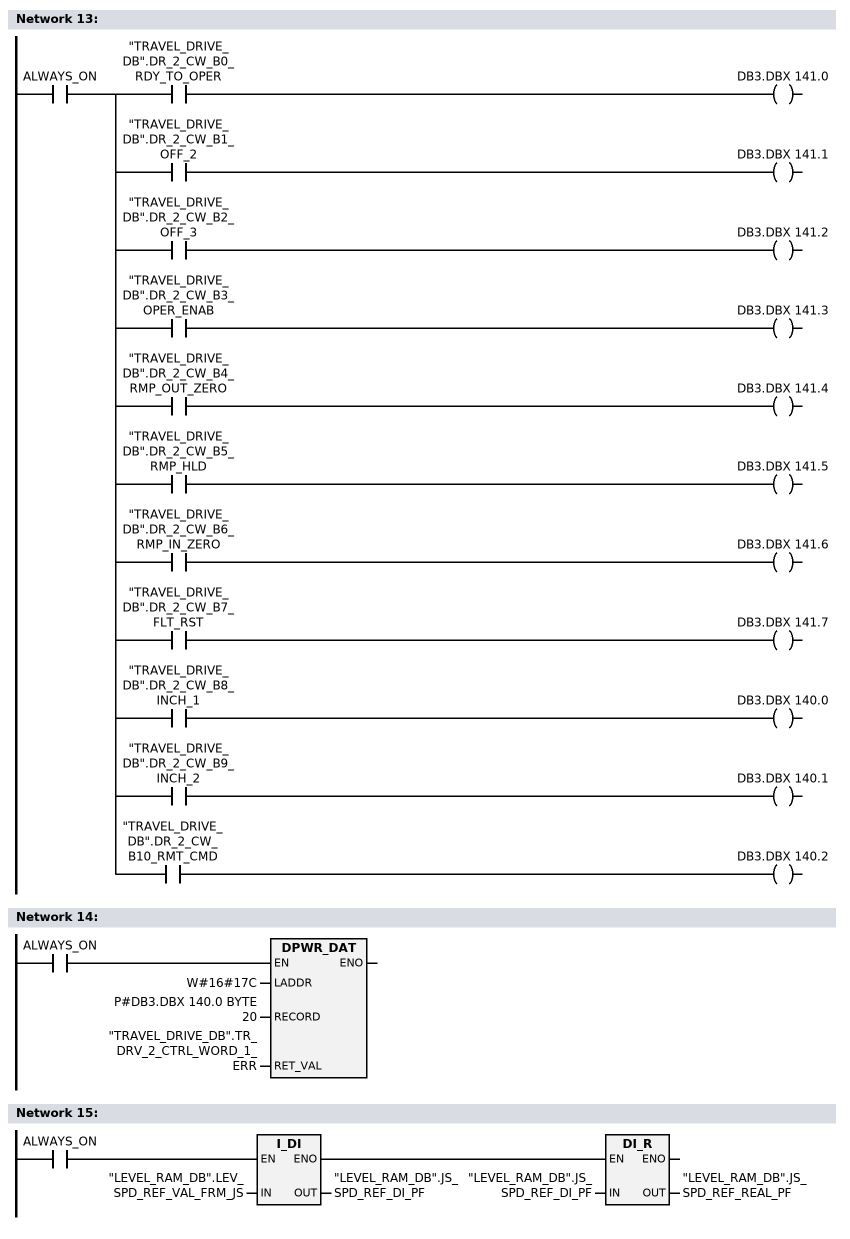
[picture p240: PROFIBUS_COMMUNICATION networks 13-15]
NETWORK
TITLE =
      A     "ALWAYS_ON";
      =     L 0.0;
      A     L 0.0;
      A     "TRAVEL_DRIVE_DB".DR_2_CW_B0_RDY_TO_OPER;
      =     DB3.DBX 141.0;
      A     L 0.0;
      A     "TRAVEL_DRIVE_DB".DR_2_CW_B1_OFF_2;
      =     DB3.DBX 141.1;
      A     L 0.0;
      A     "TRAVEL_DRIVE_DB".DR_2_CW_B2_OFF_3;
      =     DB3.DBX 141.2;
      A     L 0.0;
      A     "TRAVEL_DRIVE_DB".DR_2_CW_B3_OPER_ENAB;
      =     DB3.DBX 141.3;
      A     L 0.0;
      A     "TRAVEL_DRIVE_DB".DR_2_CW_B4_RMP_OUT_ZERO;
      =     DB3.DBX 141.4;
      A     L 0.0;
      A     "TRAVEL_DRIVE_DB".DR_2_CW_B5_RMP_HLD;
      =     DB3.DBX 141.5;
      A     L 0.0;
      A     "TRAVEL_DRIVE_DB".DR_2_CW_B6_RMP_IN_ZERO;
      =     DB3.DBX 141.6;
      A     L 0.0;
      A     "TRAVEL_DRIVE_DB".DR_2_CW_B7_FLT_RST;
      =     DB3.DBX 141.7;
      A     L 0.0;
      A     "TRAVEL_DRIVE_DB".DR_2_CW_B8_INCH_1;
      =     DB3.DBX 140.0;
      A     L 0.0;
      A     "TRAVEL_DRIVE_DB".DR_2_CW_B9_INCH_2;
      =     DB3.DBX 140.1;
      A     L 0.0;
      A     "TRAVEL_DRIVE_DB".DR_2_CW_B10_RMT_CMD;
      =     DB3.DBX 140.2;
NETWORK
TITLE =
      A     "ALWAYS_ON";
      JNB   M011;
      CALL  "DPWR_DAT" (
           LADDR                    := W#16#17C,
           RECORD                   := P#DB3.DBX 140.0 BYTE 20,
           RET_VAL                  := "TRAVEL_DRIVE_DB".TR_DRV_2_CTRL_WORD_1_ERR);
M011: NOP   0;
NETWORK
TITLE =
      A(;
      A     "ALWAYS_ON";
      JNB   M012;
      L     "LEVEL_RAM_DB".LEV_SPD_REF_VAL_FRM_JS;
      ITD;
      T     "LEVEL_RAM_DB".JS_SPD_REF_DI_PF;
      SET;
      SAVE;
      CLR;
M012: A     BR;
      );
      JNB   M013;
      L     "LEVEL_RAM_DB".JS_SPD_REF_DI_PF;
      DTR;
      T     "LEVEL_RAM_DB".JS_SPD_REF_REAL_PF;
M013: NOP   0;
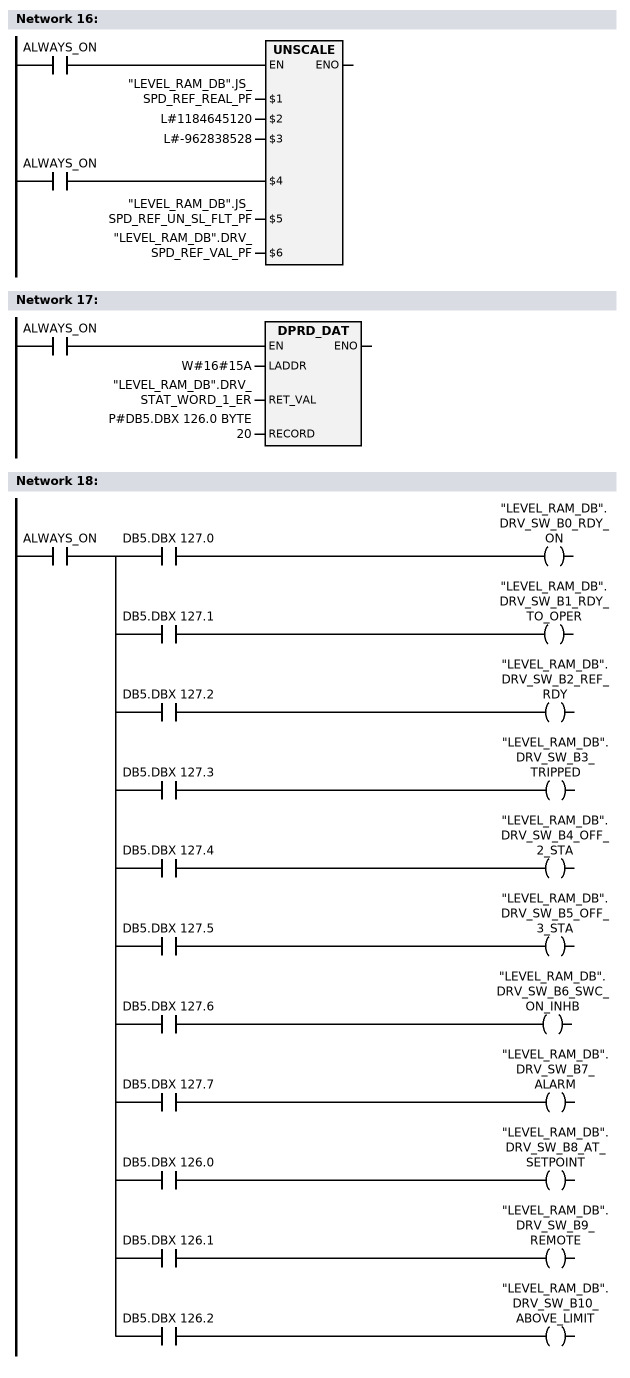
NETWORK
TITLE =
      A     "ALWAYS_ON";
      =     L 0.0;
      BLD   103;
      A     "ALWAYS_ON";
      JNB   M014;
      CALL  "UNSCALE" (
           $1                       := "LEVEL_RAM_DB".JS_SPD_REF_REAL_PF,
           $2                       := L#1184645120,
           $3                       := L#-962838528,
           $4                       := L 0.0,
           $5                       := "LEVEL_RAM_DB".JS_SPD_REF_UN_SL_FLT_PF,
           $6                       := "LEVEL_RAM_DB".DRV_SPD_REF_VAL_PF);
M014: NOP   0;
NETWORK
TITLE =
      A     "ALWAYS_ON";
      JNB   M015;
      CALL  "DPRD_DAT" (
           LADDR                    := W#16#15A,
           RET_VAL                  := "LEVEL_RAM_DB".DRV_STAT_WORD_1_ER,
           RECORD                   := P#DB5.DBX 126.0 BYTE 20);
M015: NOP   0;
NETWORK
TITLE =
      A     "ALWAYS_ON";
      =     L 0.0;
      A     L 0.0;
      A     DB5.DBX 127.0;
      =     "LEVEL_RAM_DB".DRV_SW_B0_RDY_ON;
      A     L 0.0;
      A     DB5.DBX 127.1;
      =     "LEVEL_RAM_DB".DRV_SW_B1_RDY_TO_OPER;
      A     L 0.0;
      A     DB5.DBX 127.2;
      =     "LEVEL_RAM_DB".DRV_SW_B2_REF_RDY;
      A     L 0.0;
      A     DB5.DBX 127.3;
      =     "LEVEL_RAM_DB".DRV_SW_B3_TRIPPED;
      A     L 0.0;
      A     DB5.DBX 127.4;
      =     "LEVEL_RAM_DB".DRV_SW_B4_OFF_2_STA;
      A     L 0.0;
      A     DB5.DBX 127.5;
      =     "LEVEL_RAM_DB".DRV_SW_B5_OFF_3_STA;
      A     L 0.0;
      A     DB5.DBX 127.6;
      =     "LEVEL_RAM_DB".DRV_SW_B6_SWC_ON_INHB;
      A     L 0.0;
      A     DB5.DBX 127.7;
      =     "LEVEL_RAM_DB".DRV_SW_B7_ALARM;
      A     L 0.0;
      A     DB5.DBX 126.0;
      =     "LEVEL_RAM_DB".DRV_SW_B8_AT_SETPOINT;
      A     L 0.0;
      A     DB5.DBX 126.1;
      =     "LEVEL_RAM_DB".DRV_SW_B9_REMOTE;
      A     L 0.0;
      A     DB5.DBX 126.2;
      =     "LEVEL_RAM_DB".DRV_SW_B10_ABOVE_LIMIT;
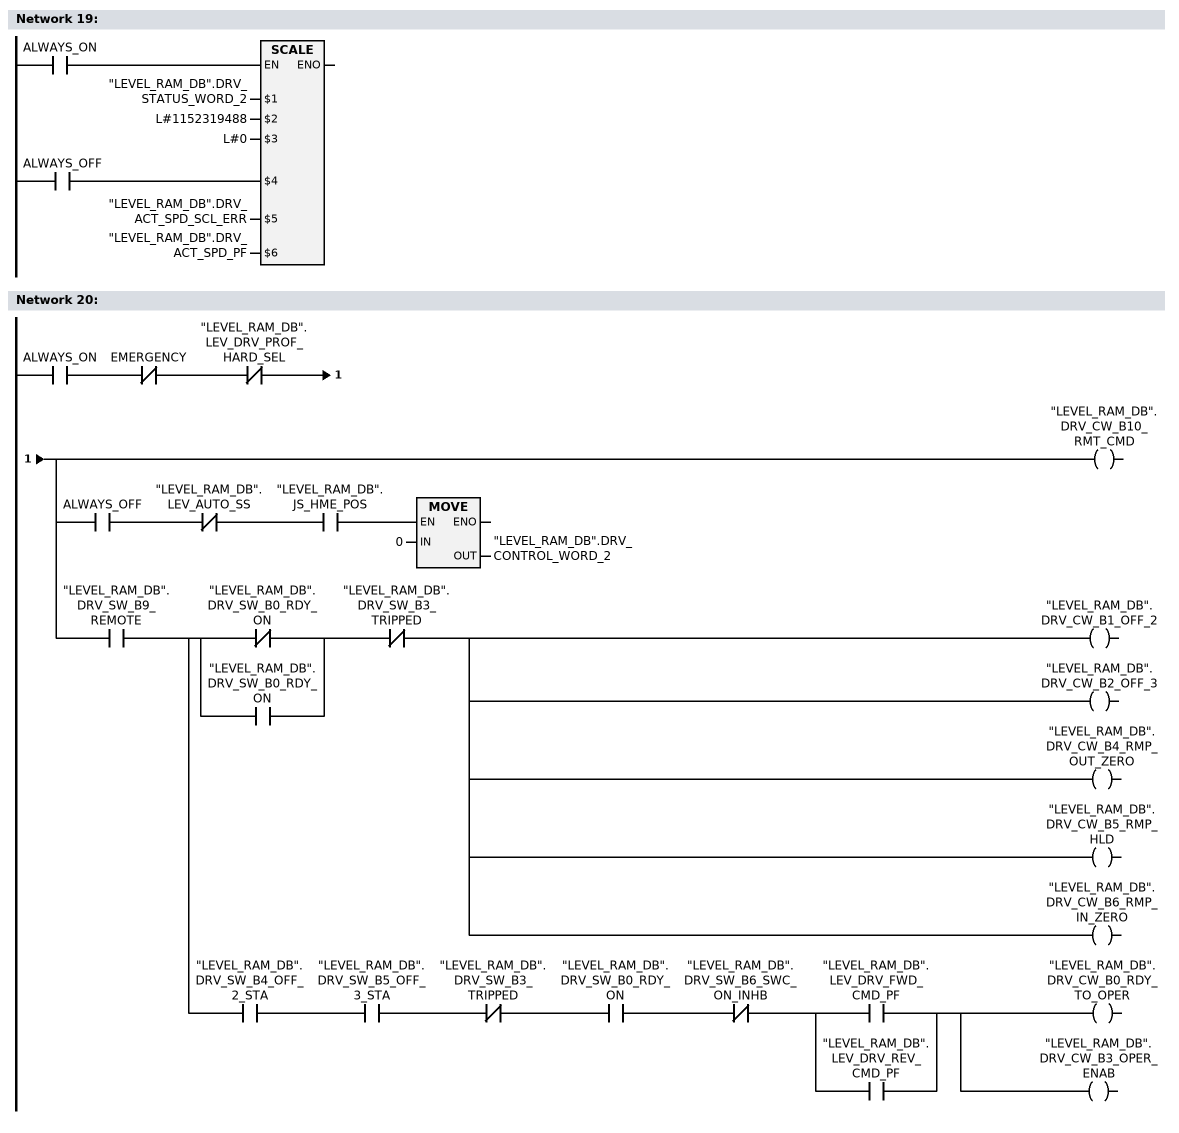
NETWORK
TITLE =
      A     "ALWAYS_OFF";
      =     L 0.0;
      BLD   103;
      A     "ALWAYS_ON";
      JNB   M016;
      CALL  "SCALE" (
           $1                       := "LEVEL_RAM_DB".DRV_STATUS_WORD_2,
           $2                       := L#1152319488,
           $3                       := L#0,
           $4                       := L 0.0,
           $5                       := "LEVEL_RAM_DB".DRV_ACT_SPD_SCL_ERR,
           $6                       := "LEVEL_RAM_DB".DRV_ACT_SPD_PF);
M016: NOP   0;
NETWORK
TITLE =
      A     "ALWAYS_ON";
      AN    "EMERGENCY";
      AN    "LEVEL_RAM_DB".LEV_DRV_PROF_HARD_SEL;
      =     L 0.0;
      A     L 0.0;
      BLD   102;
      =     "LEVEL_RAM_DB".DRV_CW_B10_RMT_CMD;
      A     L 0.0;
      A     "ALWAYS_OFF";
      AN    "LEVEL_RAM_DB".LEV_AUTO_SS;
      A     "LEVEL_RAM_DB".JS_HME_POS;
      JNB   M017;
      L     0;
      T     "LEVEL_RAM_DB".DRV_CONTROL_WORD_2;
M017: NOP   0;
      A     L 0.0;
      A     "LEVEL_RAM_DB".DRV_SW_B9_REMOTE;
      =     L 0.1;
      A     L 0.1;
      A(;
      ON    "LEVEL_RAM_DB".DRV_SW_B0_RDY_ON;
      O     "LEVEL_RAM_DB".DRV_SW_B0_RDY_ON;
      );
      AN    "LEVEL_RAM_DB".DRV_SW_B3_TRIPPED;
      =     "LEVEL_RAM_DB".DRV_CW_B1_OFF_2;
      =     "LEVEL_RAM_DB".DRV_CW_B2_OFF_3;
      =     "LEVEL_RAM_DB".DRV_CW_B4_RMP_OUT_ZERO;
      =     "LEVEL_RAM_DB".DRV_CW_B5_RMP_HLD;
      =     "LEVEL_RAM_DB".DRV_CW_B6_RMP_IN_ZERO;
      A     L 0.1;
      A     "LEVEL_RAM_DB".DRV_SW_B4_OFF_2_STA;
      A     "LEVEL_RAM_DB".DRV_SW_B5_OFF_3_STA;
      AN    "LEVEL_RAM_DB".DRV_SW_B3_TRIPPED;
      A     "LEVEL_RAM_DB".DRV_SW_B0_RDY_ON;
      AN    "LEVEL_RAM_DB".DRV_SW_B6_SWC_ON_INHB;
      A(;
      O     "LEVEL_RAM_DB".LEV_DRV_FWD_CMD_PF;
      O     "LEVEL_RAM_DB".LEV_DRV_REV_CMD_PF;
      );
      =     "LEVEL_RAM_DB".DRV_CW_B0_RDY_TO_OPER;
      =     "LEVEL_RAM_DB".DRV_CW_B3_OPER_ENAB;
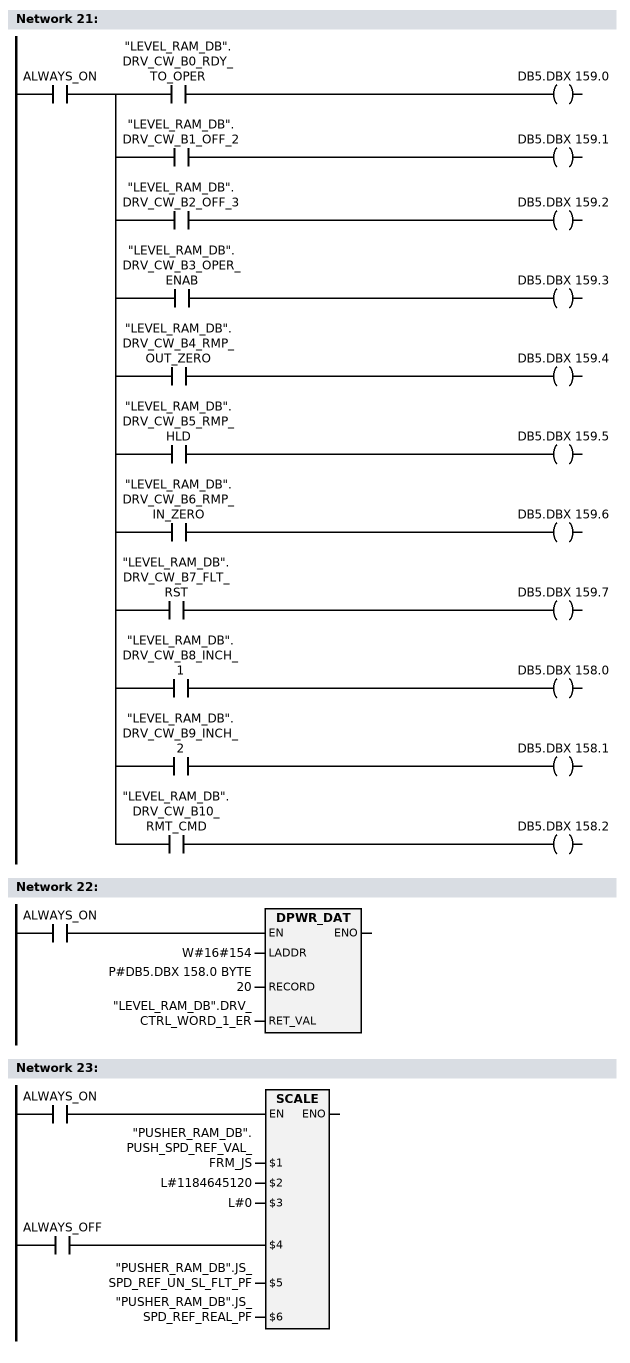
NETWORK
TITLE =
      A     "ALWAYS_ON";
      =     L 0.0;
      A     L 0.0;
      A     "LEVEL_RAM_DB".DRV_CW_B0_RDY_TO_OPER;
      =     DB5.DBX 159.0;
      A     L 0.0;
      A     "LEVEL_RAM_DB".DRV_CW_B1_OFF_2;
      =     DB5.DBX 159.1;
      A     L 0.0;
      A     "LEVEL_RAM_DB".DRV_CW_B2_OFF_3;
      =     DB5.DBX 159.2;
      A     L 0.0;
      A     "LEVEL_RAM_DB".DRV_CW_B3_OPER_ENAB;
      =     DB5.DBX 159.3;
      A     L 0.0;
      A     "LEVEL_RAM_DB".DRV_CW_B4_RMP_OUT_ZERO;
      =     DB5.DBX 159.4;
      A     L 0.0;
      A     "LEVEL_RAM_DB".DRV_CW_B5_RMP_HLD;
      =     DB5.DBX 159.5;
      A     L 0.0;
      A     "LEVEL_RAM_DB".DRV_CW_B6_RMP_IN_ZERO;
      =     DB5.DBX 159.6;
      A     L 0.0;
      A     "LEVEL_RAM_DB".DRV_CW_B7_FLT_RST;
      =     DB5.DBX 159.7;
      A     L 0.0;
      A     "LEVEL_RAM_DB".DRV_CW_B8_INCH_1;
      =     DB5.DBX 158.0;
      A     L 0.0;
      A     "LEVEL_RAM_DB".DRV_CW_B9_INCH_2;
      =     DB5.DBX 158.1;
      A     L 0.0;
      A     "LEVEL_RAM_DB".DRV_CW_B10_RMT_CMD;
      =     DB5.DBX 158.2;
NETWORK
TITLE =
      A     "ALWAYS_ON";
      JNB   M018;
      CALL  "DPWR_DAT" (
           LADDR                    := W#16#154,
           RECORD                   := P#DB5.DBX 158.0 BYTE 20,
           RET_VAL                  := "LEVEL_RAM_DB".DRV_CTRL_WORD_1_ER);
M018: NOP   0;
NETWORK
TITLE =
      A     "ALWAYS_OFF";
      =     L 0.0;
      BLD   103;
      A     "ALWAYS_ON";
      JNB   M019;
      CALL  "SCALE" (
           $1                       := "PUSHER_RAM_DB".PUSH_SPD_REF_VAL_FRM_JS,
           $2                       := L#1184645120,
           $3                       := L#0,
           $4                       := L 0.0,
           $5                       := "PUSHER_RAM_DB".JS_SPD_REF_UN_SL_FLT_PF,
           $6                       := "PUSHER_RAM_DB".JS_SPD_REF_REAL_PF);
M019: NOP   0;
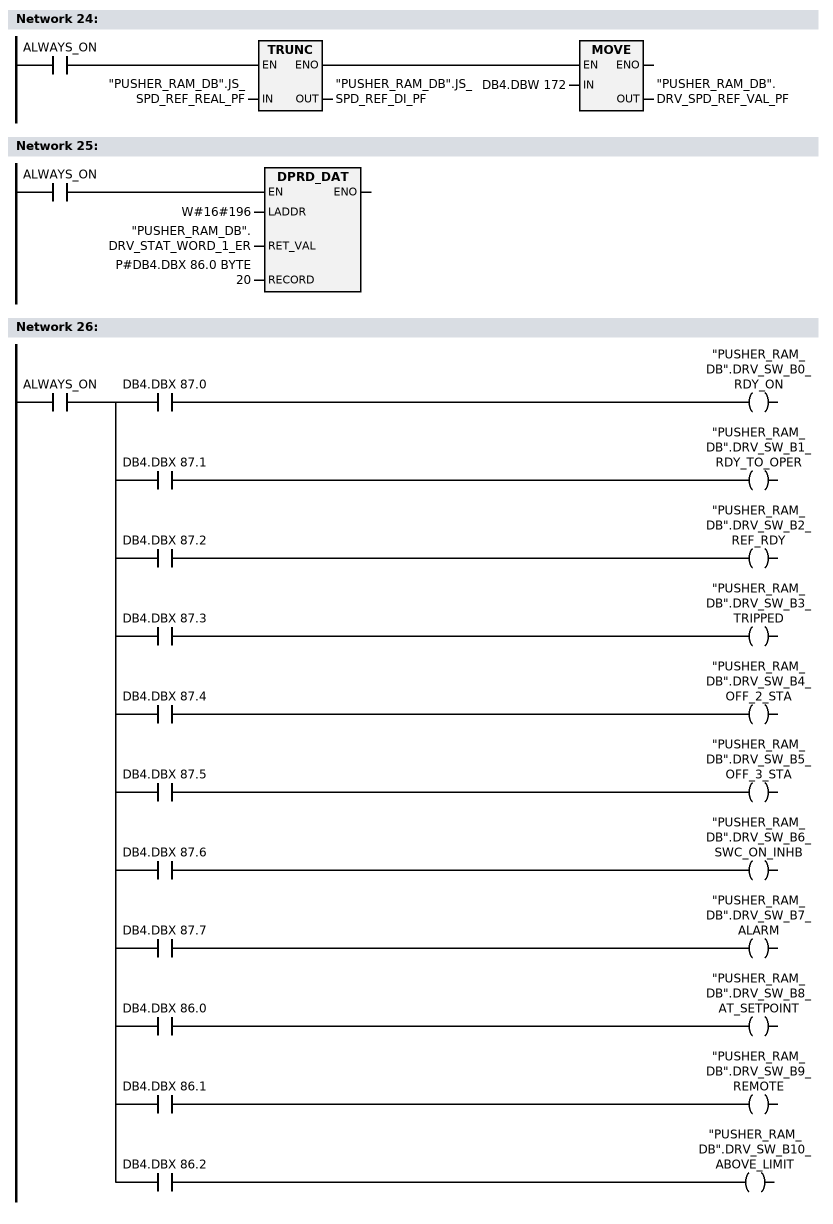
NETWORK
TITLE =
      A(;
      A     "ALWAYS_ON";
      JNB   M020;
      L     "PUSHER_RAM_DB".JS_SPD_REF_REAL_PF;
      TRUNC;
      T     "PUSHER_RAM_DB".JS_SPD_REF_DI_PF;
      AN    OV;
      SAVE;
      CLR;
M020: A     BR;
      );
      JNB   M021;
      L     DB4.DBW 172;
      T     "PUSHER_RAM_DB".DRV_SPD_REF_VAL_PF;
M021: NOP   0;
NETWORK
TITLE =
      A     "ALWAYS_ON";
      JNB   M022;
      CALL  "DPRD_DAT" (
           LADDR                    := W#16#196,
           RET_VAL                  := "PUSHER_RAM_DB".DRV_STAT_WORD_1_ER,
           RECORD                   := P#DB4.DBX 86.0 BYTE 20);
M022: NOP   0;
NETWORK
TITLE =
      A     "ALWAYS_ON";
      =     L 0.0;
      A     L 0.0;
      A     DB4.DBX 87.0;
      =     "PUSHER_RAM_DB".DRV_SW_B0_RDY_ON;
      A     L 0.0;
      A     DB4.DBX 87.1;
      =     "PUSHER_RAM_DB".DRV_SW_B1_RDY_TO_OPER;
      A     L 0.0;
      A     DB4.DBX 87.2;
      =     "PUSHER_RAM_DB".DRV_SW_B2_REF_RDY;
      A     L 0.0;
      A     DB4.DBX 87.3;
      =     "PUSHER_RAM_DB".DRV_SW_B3_TRIPPED;
      A     L 0.0;
      A     DB4.DBX 87.4;
      =     "PUSHER_RAM_DB".DRV_SW_B4_OFF_2_STA;
      A     L 0.0;
      A     DB4.DBX 87.5;
      =     "PUSHER_RAM_DB".DRV_SW_B5_OFF_3_STA;
      A     L 0.0;
      A     DB4.DBX 87.6;
      =     "PUSHER_RAM_DB".DRV_SW_B6_SWC_ON_INHB;
      A     L 0.0;
      A     DB4.DBX 87.7;
      =     "PUSHER_RAM_DB".DRV_SW_B7_ALARM;
      A     L 0.0;
      A     DB4.DBX 86.0;
      =     "PUSHER_RAM_DB".DRV_SW_B8_AT_SETPOINT;
      A     L 0.0;
      A     DB4.DBX 86.1;
      =     "PUSHER_RAM_DB".DRV_SW_B9_REMOTE;
      A     L 0.0;
      A     DB4.DBX 86.2;
      =     "PUSHER_RAM_DB".DRV_SW_B10_ABOVE_LIMIT;
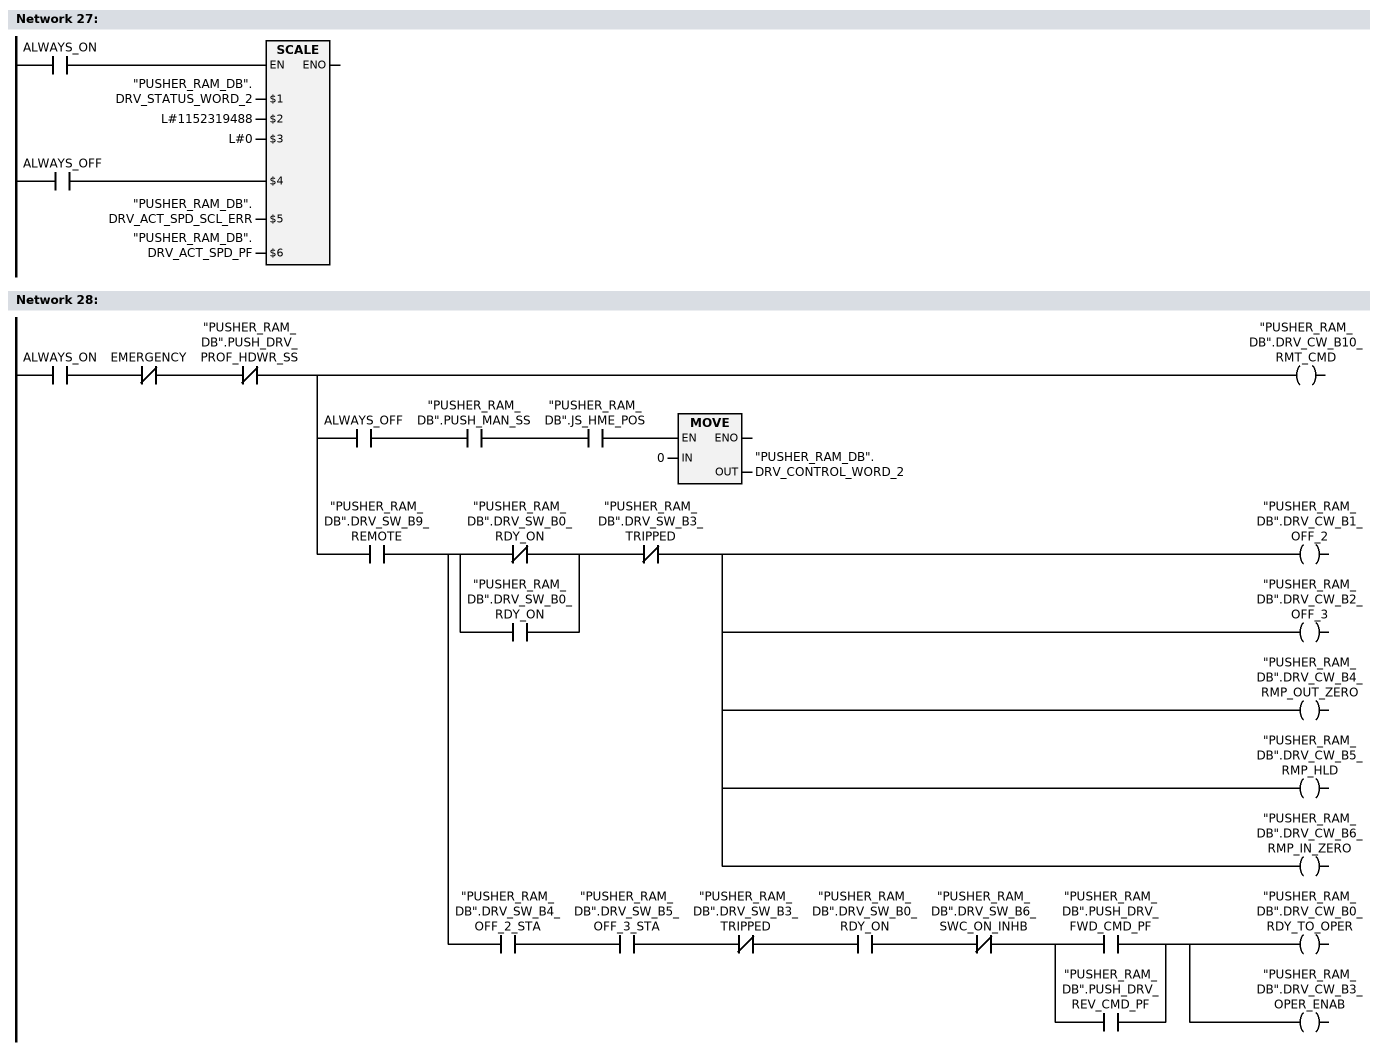
NETWORK
TITLE =
      A     "ALWAYS_OFF";
      =     L 0.0;
      BLD   103;
      A     "ALWAYS_ON";
      JNB   M023;
      CALL  "SCALE" (
           $1                       := "PUSHER_RAM_DB".DRV_STATUS_WORD_2,
           $2                       := L#1152319488,
           $3                       := L#0,
           $4                       := L 0.0,
           $5                       := "PUSHER_RAM_DB".DRV_ACT_SPD_SCL_ERR,
           $6                       := "PUSHER_RAM_DB".DRV_ACT_SPD_PF);
M023: NOP   0;
NETWORK
TITLE =
      A     "ALWAYS_ON";
      AN    "EMERGENCY";
      AN    "PUSHER_RAM_DB".PUSH_DRV_PROF_HDWR_SS;
      =     L 0.0;
      A     L 0.0;
      BLD   102;
      =     "PUSHER_RAM_DB".DRV_CW_B10_RMT_CMD;
      A     L 0.0;
      A     "ALWAYS_OFF";
      A     "PUSHER_RAM_DB".PUSH_MAN_SS;
      A     "PUSHER_RAM_DB".JS_HME_POS;
      JNB   M024;
      L     0;
      T     "PUSHER_RAM_DB".DRV_CONTROL_WORD_2;
M024: NOP   0;
      A     L 0.0;
      A     "PUSHER_RAM_DB".DRV_SW_B9_REMOTE;
      =     L 0.1;
      A     L 0.1;
      A(;
      ON    "PUSHER_RAM_DB".DRV_SW_B0_RDY_ON;
      O     "PUSHER_RAM_DB".DRV_SW_B0_RDY_ON;
      );
      AN    "PUSHER_RAM_DB".DRV_SW_B3_TRIPPED;
      =     "PUSHER_RAM_DB".DRV_CW_B1_OFF_2;
      =     "PUSHER_RAM_DB".DRV_CW_B2_OFF_3;
      =     "PUSHER_RAM_DB".DRV_CW_B4_RMP_OUT_ZERO;
      =     "PUSHER_RAM_DB".DRV_CW_B5_RMP_HLD;
      =     "PUSHER_RAM_DB".DRV_CW_B6_RMP_IN_ZERO;
      A     L 0.1;
      A     "PUSHER_RAM_DB".DRV_SW_B4_OFF_2_STA;
      A     "PUSHER_RAM_DB".DRV_SW_B5_OFF_3_STA;
      AN    "PUSHER_RAM_DB".DRV_SW_B3_TRIPPED;
      A     "PUSHER_RAM_DB".DRV_SW_B0_RDY_ON;
      AN    "PUSHER_RAM_DB".DRV_SW_B6_SWC_ON_INHB;
      A(;
      O     "PUSHER_RAM_DB".PUSH_DRV_FWD_CMD_PF;
      O     "PUSHER_RAM_DB".PUSH_DRV_REV_CMD_PF;
      );
      =     "PUSHER_RAM_DB".DRV_CW_B0_RDY_TO_OPER;
      =     "PUSHER_RAM_DB".DRV_CW_B3_OPER_ENAB;
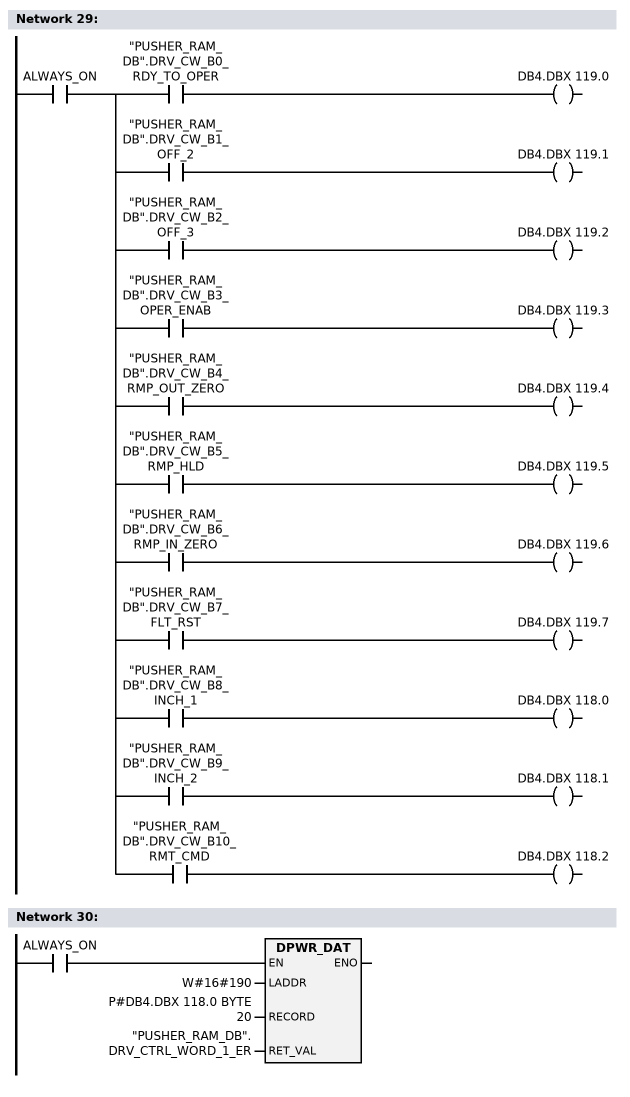
NETWORK
TITLE =
      A     "ALWAYS_ON";
      =     L 0.0;
      A     L 0.0;
      A     "PUSHER_RAM_DB".DRV_CW_B0_RDY_TO_OPER;
      =     DB4.DBX 119.0;
      A     L 0.0;
      A     "PUSHER_RAM_DB".DRV_CW_B1_OFF_2;
      =     DB4.DBX 119.1;
      A     L 0.0;
      A     "PUSHER_RAM_DB".DRV_CW_B2_OFF_3;
      =     DB4.DBX 119.2;
      A     L 0.0;
      A     "PUSHER_RAM_DB".DRV_CW_B3_OPER_ENAB;
      =     DB4.DBX 119.3;
      A     L 0.0;
      A     "PUSHER_RAM_DB".DRV_CW_B4_RMP_OUT_ZERO;
      =     DB4.DBX 119.4;
      A     L 0.0;
      A     "PUSHER_RAM_DB".DRV_CW_B5_RMP_HLD;
      =     DB4.DBX 119.5;
      A     L 0.0;
      A     "PUSHER_RAM_DB".DRV_CW_B6_RMP_IN_ZERO;
      =     DB4.DBX 119.6;
      A     L 0.0;
      A     "PUSHER_RAM_DB".DRV_CW_B7_FLT_RST;
      =     DB4.DBX 119.7;
      A     L 0.0;
      A     "PUSHER_RAM_DB".DRV_CW_B8_INCH_1;
      =     DB4.DBX 118.0;
      A     L 0.0;
      A     "PUSHER_RAM_DB".DRV_CW_B9_INCH_2;
      =     DB4.DBX 118.1;
      A     L 0.0;
      A     "PUSHER_RAM_DB".DRV_CW_B10_RMT_CMD;
      =     DB4.DBX 118.2;
NETWORK
TITLE =
      A     "ALWAYS_ON";
      JNB   M025;
      CALL  "DPWR_DAT" (
           LADDR                    := W#16#190,
           RECORD                   := P#DB4.DBX 118.0 BYTE 20,
           RET_VAL                  := "PUSHER_RAM_DB".DRV_CTRL_WORD_1_ER);
M025: NOP   0;
END_FUNCTION

FUNCTION "TATA_COMMUNICATION" : VOID	// FC 20
AUTHOR : Kamillas
VERSION : 0.1
BEGIN
// (block stored without names or comments; labels and parameter names are numbered)
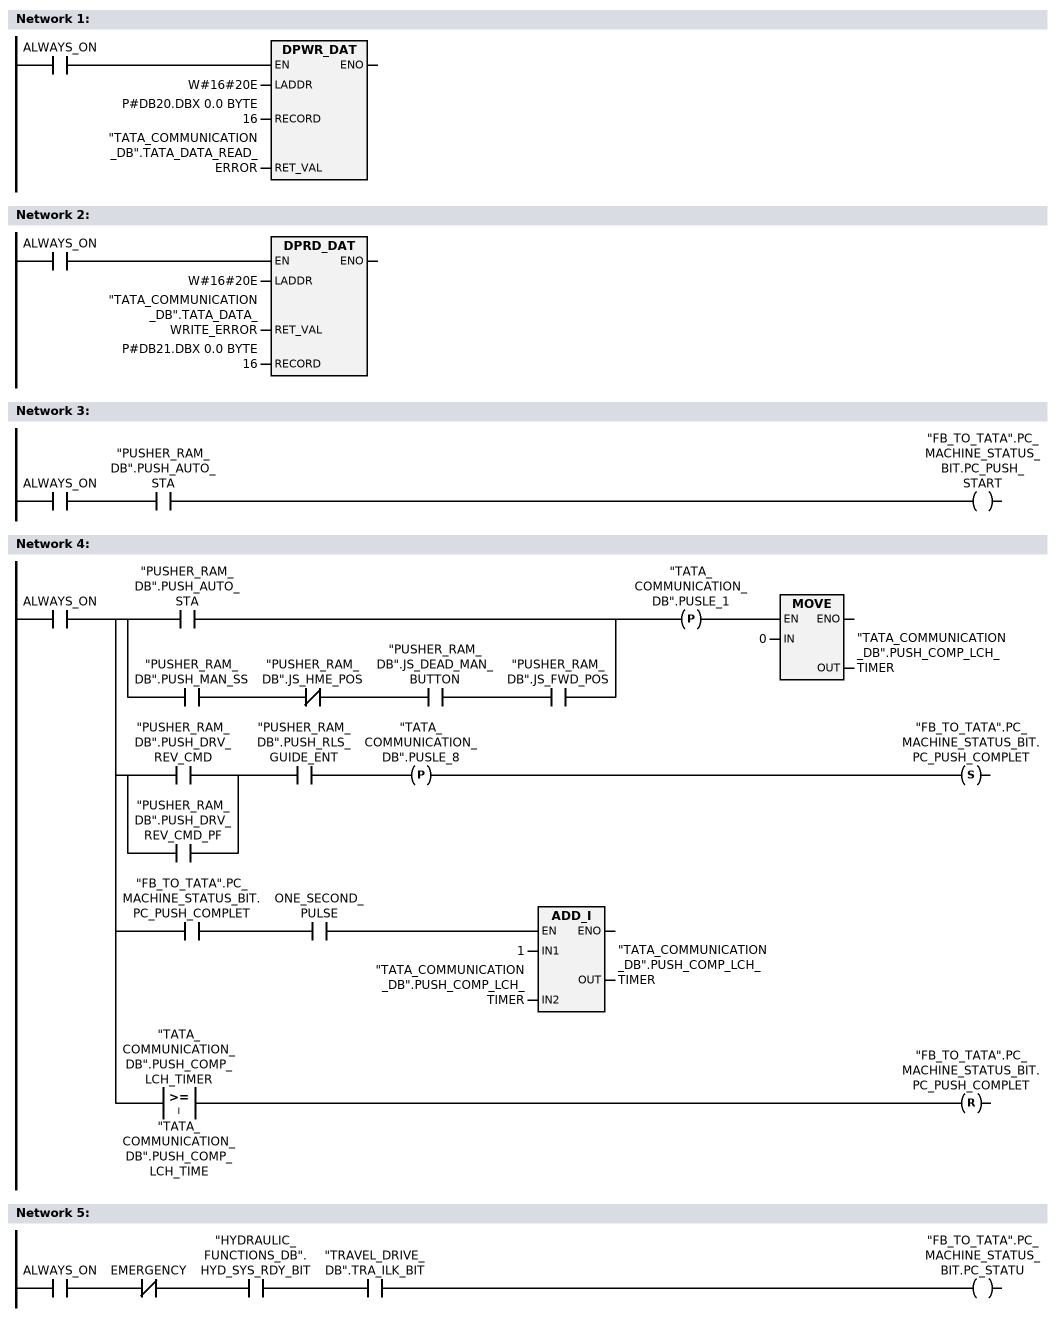
NETWORK
TITLE =
      A     "ALWAYS_ON";
      JNB   M001;
      CALL  "DPWR_DAT" (
           LADDR                    := W#16#20E,
           RECORD                   := P#DB20.DBX 0.0 BYTE 16,
           RET_VAL                  := "TATA_COMMUNICATION_DB".TATA_DATA_READ_ERROR);
M001: NOP   0;
NETWORK
TITLE =
      A     "ALWAYS_ON";
      JNB   M002;
      CALL  "DPRD_DAT" (
           LADDR                    := W#16#20E,
           RET_VAL                  := "TATA_COMMUNICATION_DB".TATA_DATA_WRITE_ERROR,
           RECORD                   := P#DB21.DBX 0.0 BYTE 16);
M002: NOP   0;
NETWORK
TITLE =
      A     "ALWAYS_ON";
      A     "PUSHER_RAM_DB".PUSH_AUTO_STA;
      =     "FB_TO_TATA".PC_MACHINE_STATUS_BIT.PC_PUSH_START;
NETWORK
TITLE =
      A     "ALWAYS_ON";
      =     L 0.0;
      A     L 0.0;
      A(;
      O     "PUSHER_RAM_DB".PUSH_AUTO_STA;
      O;
      A     "PUSHER_RAM_DB".PUSH_MAN_SS;
      AN    "PUSHER_RAM_DB".JS_HME_POS;
      A     "PUSHER_RAM_DB".JS_DEAD_MAN_BUTTON;
      A     "PUSHER_RAM_DB".JS_FWD_POS;
      );
      FP    "TATA_COMMUNICATION_DB".PUSLE_1;
      JNB   M003;
      L     0;
      T     "TATA_COMMUNICATION_DB".PUSH_COMP_LCH_TIMER;
M003: NOP   0;
      A     L 0.0;
      A(;
      O     "PUSHER_RAM_DB".PUSH_DRV_REV_CMD;
      O     "PUSHER_RAM_DB".PUSH_DRV_REV_CMD_PF;
      );
      A     "PUSHER_RAM_DB".PUSH_RLS_GUIDE_ENT;
      FP    "TATA_COMMUNICATION_DB".PUSLE_8;
      S     "FB_TO_TATA".PC_MACHINE_STATUS_BIT.PC_PUSH_COMPLET;
      A     L 0.0;
      A     "FB_TO_TATA".PC_MACHINE_STATUS_BIT.PC_PUSH_COMPLET;
      A     "ONE_SECOND_PULSE";
      JNB   M004;
      L     1;
      L     "TATA_COMMUNICATION_DB".PUSH_COMP_LCH_TIMER;
      +I;
      T     "TATA_COMMUNICATION_DB".PUSH_COMP_LCH_TIMER;
M004: NOP   0;
      A     L 0.0;
      A(;
      L     "TATA_COMMUNICATION_DB".PUSH_COMP_LCH_TIMER;
      L     "TATA_COMMUNICATION_DB".PUSH_COMP_LCH_TIME;
      >=I;
      );
      R     "FB_TO_TATA".PC_MACHINE_STATUS_BIT.PC_PUSH_COMPLET;
NETWORK
TITLE =
      A     "ALWAYS_ON";
      AN    "EMERGENCY";
      A     "HYDRAULIC_FUNCTIONS_DB".HYD_SYS_RDY_BIT;
      A     "TRAVEL_DRIVE_DB".TRA_ILK_BIT;
      =     "FB_TO_TATA".PC_MACHINE_STATUS_BIT.PC_STATU;
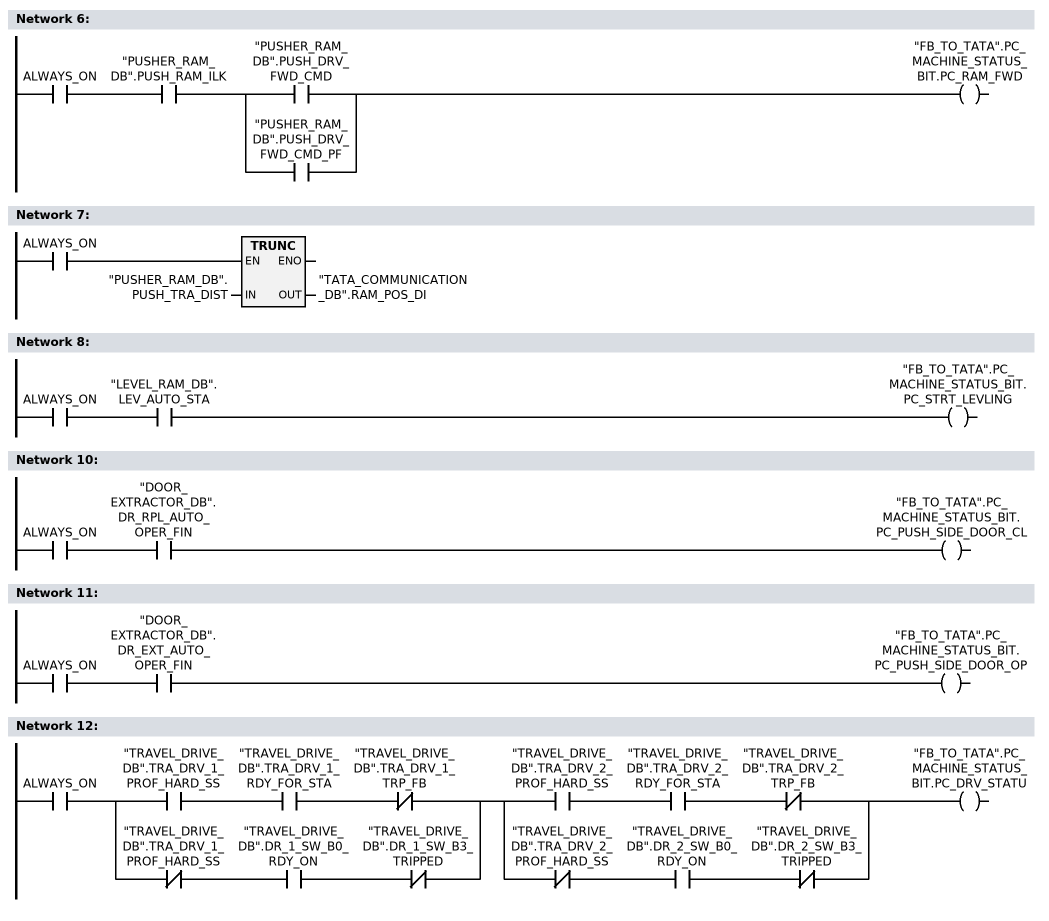
NETWORK
TITLE =
      A     "ALWAYS_ON";
      A     "PUSHER_RAM_DB".PUSH_RAM_ILK;
      A(;
      O     "PUSHER_RAM_DB".PUSH_DRV_FWD_CMD;
      O     "PUSHER_RAM_DB".PUSH_DRV_FWD_CMD_PF;
      );
      =     "FB_TO_TATA".PC_MACHINE_STATUS_BIT.PC_RAM_FWD;
NETWORK
TITLE =
      A     "ALWAYS_ON";
      JNB   M005;
      L     "PUSHER_RAM_DB".PUSH_TRA_DIST;
      TRUNC;
      T     "TATA_COMMUNICATION_DB".RAM_POS_DI;
M005: NOP   0;
NETWORK
TITLE =
      A     "ALWAYS_ON";
      A     "LEVEL_RAM_DB".LEV_AUTO_STA;
      =     "FB_TO_TATA".PC_MACHINE_STATUS_BIT.PC_STRT_LEVLING;
NETWORK
TITLE =
      A     "ALWAYS_ON";
      =     L 0.0;
      A     L 0.0;
      A(;
      O     "LEVEL_RAM_DB".LEV_AUTO_STA;
      O     "LEVEL_RAM_DB".LEV_AUTO_STP_RET;
      );
      =     L 0.1;
      A     L 0.1;
      FP    "TATA_COMMUNICATION_DB".PUSLE_3;
      JNB   M006;
      L     0;
      T     "TATA_COMMUNICATION_DB".LEV_COMP_LCH_TIMER;
M006: NOP   0;
      A(;
      A     L 0.1;
      FN    "TATA_COMMUNICATION_DB".PUSLE_4;
      );
      A     "LEVEL_RAM_DB".LEV_AUTO_SS;
      A(;
      ON    "LEVEL_RAM_DB".LEV_RLS_REV_END;
      ON    "LEVEL_RAM_DB".LEV_END_RET_LS;
      );
      S     "FB_TO_TATA".PC_MACHINE_STATUS_BIT.PC_STOP_LEVLING;
      A     L 0.0;
      A     "FB_TO_TATA".PC_MACHINE_STATUS_BIT.PC_STOP_LEVLING;
      A     "ONE_SECOND_PULSE";
      JNB   M007;
      L     1;
      L     "TATA_COMMUNICATION_DB".LEV_COMP_LCH_TIMER;
      +I;
      T     "TATA_COMMUNICATION_DB".LEV_COMP_LCH_TIMER;
M007: NOP   0;
      A     L 0.0;
      A(;
      L     "TATA_COMMUNICATION_DB".LEV_COMP_LCH_TIMER;
      L     "TATA_COMMUNICATION_DB".LEV_COMP_LCH_TIME;
      >=I;
      );
      R     "FB_TO_TATA".PC_MACHINE_STATUS_BIT.PC_STOP_LEVLING;
NETWORK
TITLE =
      A     "ALWAYS_ON";
      A     "DOOR_EXTRACTOR_DB".DR_RPL_AUTO_OPER_FIN;
      =     "FB_TO_TATA".PC_MACHINE_STATUS_BIT.PC_PUSH_SIDE_DOOR_CL;
NETWORK
TITLE =
      A     "ALWAYS_ON";
      A     "DOOR_EXTRACTOR_DB".DR_EXT_AUTO_OPER_FIN;
      =     "FB_TO_TATA".PC_MACHINE_STATUS_BIT.PC_PUSH_SIDE_DOOR_OP;
NETWORK
TITLE =
      A     "ALWAYS_ON";
      A(;
      A     "TRAVEL_DRIVE_DB".TRA_DRV_1_PROF_HARD_SS;
      A     "TRAVEL_DRIVE_DB".TRA_DRV_1_RDY_FOR_STA;
      AN    "TRAVEL_DRIVE_DB".TRA_DRV_1_TRP_FB;
      O;
      AN    "TRAVEL_DRIVE_DB".TRA_DRV_1_PROF_HARD_SS;
      A     "TRAVEL_DRIVE_DB".DR_1_SW_B0_RDY_ON;
      AN    "TRAVEL_DRIVE_DB".DR_1_SW_B3_TRIPPED;
      );
      A(;
      A     "TRAVEL_DRIVE_DB".TRA_DRV_2_PROF_HARD_SS;
      A     "TRAVEL_DRIVE_DB".TRA_DRV_2_RDY_FOR_STA;
      AN    "TRAVEL_DRIVE_DB".TRA_DRV_2_TRP_FB;
      O;
      AN    "TRAVEL_DRIVE_DB".TRA_DRV_2_PROF_HARD_SS;
      A     "TRAVEL_DRIVE_DB".DR_2_SW_B0_RDY_ON;
      AN    "TRAVEL_DRIVE_DB".DR_2_SW_B3_TRIPPED;
      );
      =     "FB_TO_TATA".PC_MACHINE_STATUS_BIT.PC_DRV_STATU;
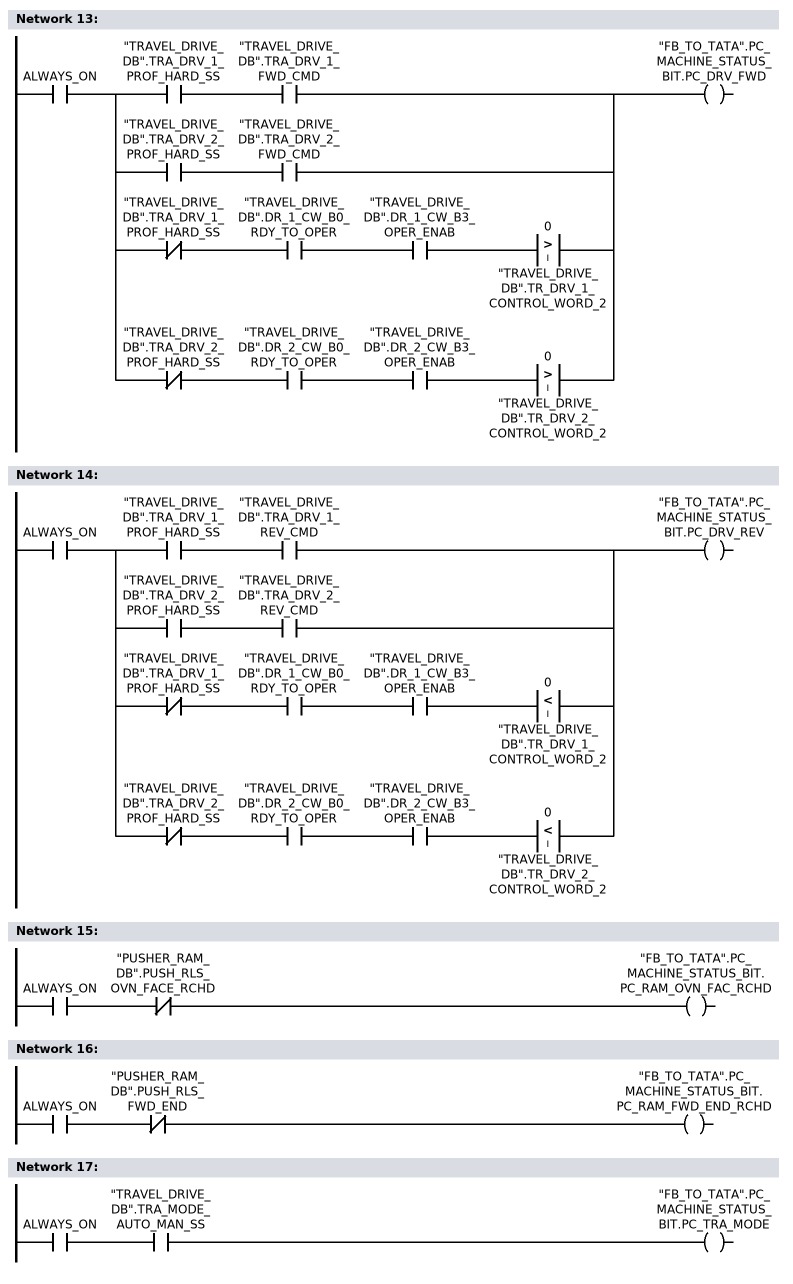
NETWORK
TITLE =
      A     "ALWAYS_ON";
      A(;
      A     "TRAVEL_DRIVE_DB".TRA_DRV_1_PROF_HARD_SS;
      A     "TRAVEL_DRIVE_DB".TRA_DRV_1_FWD_CMD;
      O;
      A     "TRAVEL_DRIVE_DB".TRA_DRV_2_PROF_HARD_SS;
      A     "TRAVEL_DRIVE_DB".TRA_DRV_2_FWD_CMD;
      O;
      AN    "TRAVEL_DRIVE_DB".TRA_DRV_1_PROF_HARD_SS;
      A     "TRAVEL_DRIVE_DB".DR_1_CW_B0_RDY_TO_OPER;
      A     "TRAVEL_DRIVE_DB".DR_1_CW_B3_OPER_ENAB;
      A(;
      L     0;
      L     "TRAVEL_DRIVE_DB".TR_DRV_1_CONTROL_WORD_2;
      >I;
      );
      O;
      AN    "TRAVEL_DRIVE_DB".TRA_DRV_2_PROF_HARD_SS;
      A     "TRAVEL_DRIVE_DB".DR_2_CW_B0_RDY_TO_OPER;
      A     "TRAVEL_DRIVE_DB".DR_2_CW_B3_OPER_ENAB;
      A(;
      L     0;
      L     "TRAVEL_DRIVE_DB".TR_DRV_2_CONTROL_WORD_2;
      >I;
      );
      );
      =     "FB_TO_TATA".PC_MACHINE_STATUS_BIT.PC_DRV_FWD;
NETWORK
TITLE =
      A     "ALWAYS_ON";
      A(;
      A     "TRAVEL_DRIVE_DB".TRA_DRV_1_PROF_HARD_SS;
      A     "TRAVEL_DRIVE_DB".TRA_DRV_1_REV_CMD;
      O;
      A     "TRAVEL_DRIVE_DB".TRA_DRV_2_PROF_HARD_SS;
      A     "TRAVEL_DRIVE_DB".TRA_DRV_2_REV_CMD;
      O;
      AN    "TRAVEL_DRIVE_DB".TRA_DRV_1_PROF_HARD_SS;
      A     "TRAVEL_DRIVE_DB".DR_1_CW_B0_RDY_TO_OPER;
      A     "TRAVEL_DRIVE_DB".DR_1_CW_B3_OPER_ENAB;
      A(;
      L     0;
      L     "TRAVEL_DRIVE_DB".TR_DRV_1_CONTROL_WORD_2;
      <I;
      );
      O;
      AN    "TRAVEL_DRIVE_DB".TRA_DRV_2_PROF_HARD_SS;
      A     "TRAVEL_DRIVE_DB".DR_2_CW_B0_RDY_TO_OPER;
      A     "TRAVEL_DRIVE_DB".DR_2_CW_B3_OPER_ENAB;
      A(;
      L     0;
      L     "TRAVEL_DRIVE_DB".TR_DRV_2_CONTROL_WORD_2;
      <I;
      );
      );
      =     "FB_TO_TATA".PC_MACHINE_STATUS_BIT.PC_DRV_REV;
NETWORK
TITLE =
      A     "ALWAYS_ON";
      AN    "PUSHER_RAM_DB".PUSH_RLS_OVN_FACE_RCHD;
      =     "FB_TO_TATA".PC_MACHINE_STATUS_BIT.PC_RAM_OVN_FAC_RCHD;
NETWORK
TITLE =
      A     "ALWAYS_ON";
      AN    "PUSHER_RAM_DB".PUSH_RLS_FWD_END;
      =     "FB_TO_TATA".PC_MACHINE_STATUS_BIT.PC_RAM_FWD_END_RCHD;
NETWORK
TITLE =
      A     "ALWAYS_ON";
      A     "TRAVEL_DRIVE_DB".TRA_MODE_AUTO_MAN_SS;
      =     "FB_TO_TATA".PC_MACHINE_STATUS_BIT.PC_TRA_MODE;
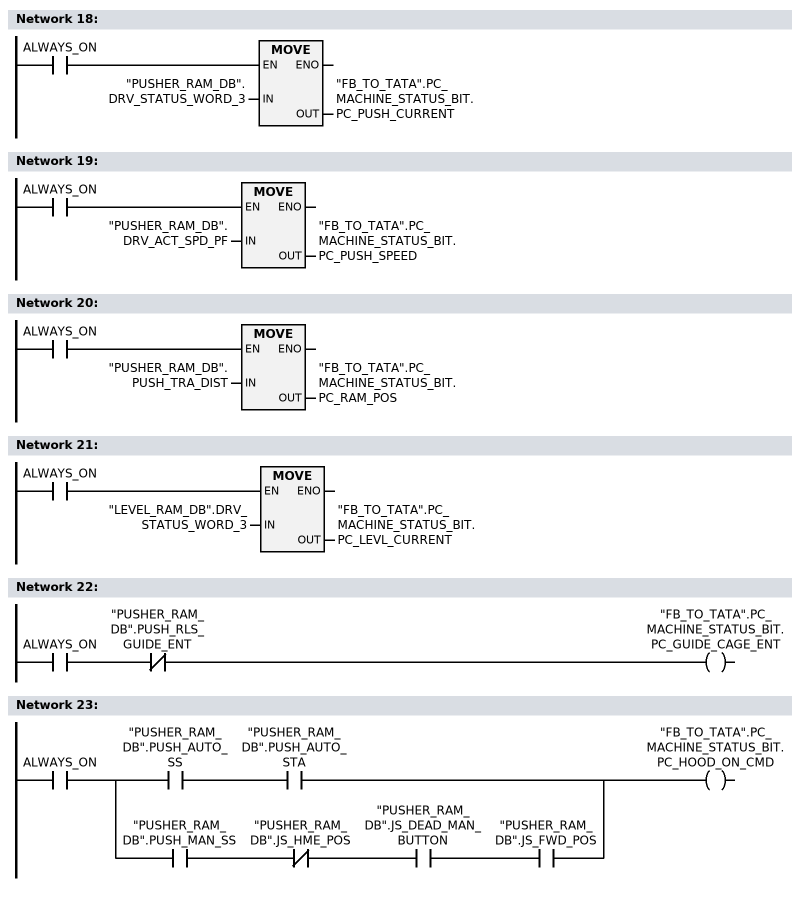
NETWORK
TITLE =
      A     "ALWAYS_ON";
      JNB   M008;
      L     "PUSHER_RAM_DB".DRV_STATUS_WORD_3;
      T     "FB_TO_TATA".PC_MACHINE_STATUS_BIT.PC_PUSH_CURRENT;
M008: NOP   0;
NETWORK
TITLE =
      A     "ALWAYS_ON";
      JNB   M009;
      L     "PUSHER_RAM_DB".DRV_ACT_SPD_PF;
      T     "FB_TO_TATA".PC_MACHINE_STATUS_BIT.PC_PUSH_SPEED;
M009: NOP   0;
NETWORK
TITLE =
      A     "ALWAYS_ON";
      JNB   M010;
      L     "PUSHER_RAM_DB".PUSH_TRA_DIST;
      T     "FB_TO_TATA".PC_MACHINE_STATUS_BIT.PC_RAM_POS;
M010: NOP   0;
NETWORK
TITLE =
      A     "ALWAYS_ON";
      JNB   M011;
      L     "LEVEL_RAM_DB".DRV_STATUS_WORD_3;
      T     "FB_TO_TATA".PC_MACHINE_STATUS_BIT.PC_LEVL_CURRENT;
M011: NOP   0;
NETWORK
TITLE =
      A     "ALWAYS_ON";
      AN    "PUSHER_RAM_DB".PUSH_RLS_GUIDE_ENT;
      =     "FB_TO_TATA".PC_MACHINE_STATUS_BIT.PC_GUIDE_CAGE_ENT;
NETWORK
TITLE =
      A     "ALWAYS_ON";
      A(;
      A     "PUSHER_RAM_DB".PUSH_AUTO_SS;
      A     "PUSHER_RAM_DB".PUSH_AUTO_STA;
      O;
      A     "PUSHER_RAM_DB".PUSH_MAN_SS;
      AN    "PUSHER_RAM_DB".JS_HME_POS;
      A     "PUSHER_RAM_DB".JS_DEAD_MAN_BUTTON;
      A     "PUSHER_RAM_DB".JS_FWD_POS;
      );
      =     "FB_TO_TATA".PC_MACHINE_STATUS_BIT.PC_HOOD_ON_CMD;
END_FUNCTION

FUNCTION FC 21 : VOID
VERSION : 0.1
BEGIN
// (block stored without names or comments; labels and parameter names are numbered)
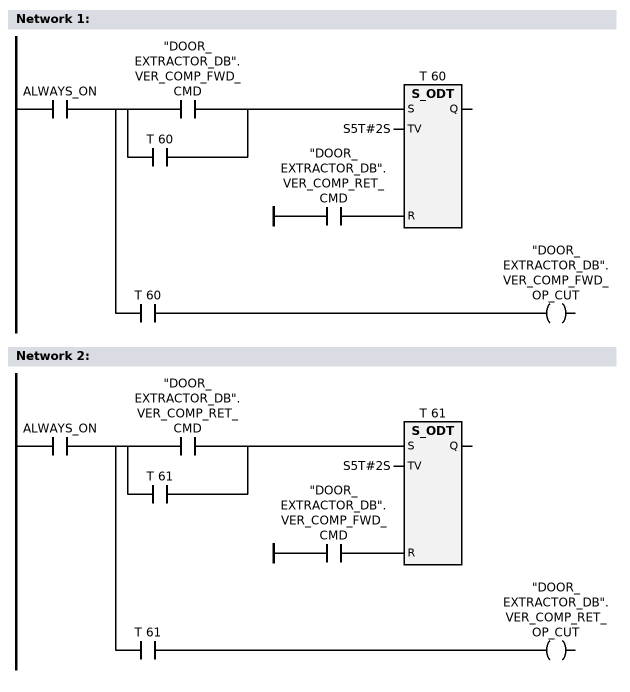
NETWORK
TITLE =
      A     "ALWAYS_ON";
      =     L 0.0;
      A     L 0.0;
      A(;
      O     "DOOR_EXTRACTOR_DB".VER_COMP_FWD_CMD;
      O     T 60;
      );
      L     S5T#2S;
      SD    T 60;
      A     "DOOR_EXTRACTOR_DB".VER_COMP_RET_CMD;
      R     T 60;
      NOP   0;
      NOP   0;
      NOP   0;
      A     L 0.0;
      A     T 60;
      =     "DOOR_EXTRACTOR_DB".VER_COMP_FWD_OP_CUT;
NETWORK
TITLE =
      A     "ALWAYS_ON";
      =     L 0.0;
      A     L 0.0;
      A(;
      O     "DOOR_EXTRACTOR_DB".VER_COMP_RET_CMD;
      O     T 61;
      );
      L     S5T#2S;
      SD    T 61;
      A     "DOOR_EXTRACTOR_DB".VER_COMP_FWD_CMD;
      R     T 61;
      NOP   0;
      NOP   0;
      NOP   0;
      A     L 0.0;
      A     T 61;
      =     "DOOR_EXTRACTOR_DB".VER_COMP_RET_OP_CUT;
END_FUNCTION

// FC 105: know-how protected block, not included

// FC 106: know-how protected block, not included

DATA_BLOCK "MAIN_POWER_DB"	// DB 1
AUTHOR : Kamillas
VERSION : 0.1
  STRUCT
   MAIN_PWR_RDY_FOR_ON : BOOL ;	//MAIN POWER READY FOR ON
   MAIN_PWR_ON_FB : BOOL ;	//MAIN POWER ON FEED BACK
   CTRL_PWR_ON_FB : BOOL ;	//CONTROL POWER ON FEEDBACK
   MAIN_PWR_ON_PB : BOOL ;	//MAIN POWER ON PUSH BUTTON
   MAIN_PWR_OFF_PB : BOOL ;	//MAIN POWER OFF PUSH BUTTON
   LAMP_TEST_PB : BOOL ;	//LAMP TEST PUSH BUTTON
   ALARM_ACK_PB : BOOL ;	//ALARM ACKNOWLEDGE PUSH BUTTON
   MAIN_PWR_ON_CMD : BOOL ;	//MAIN POWER ON COMMAND
   MAIN_PWR_ON_IND : BOOL ;	//MAIN POWER ON INDICATOR
   CTRL_PWR_ON_IND : BOOL ;	//CONTROL POWER ON INDICATOR
   CTRL_SELECTION_CD : BOOL ;	//CONTROL SELECTRION CD
   MAIN_PWR_FLT : BOOL ;	//MAIN POWER FAULT
   CTRL_PWR_FLT : BOOL ;	//CTRL POWER FAULT
   MAIN_PWR_HEALTHY : BOOL ;	//MAIN POWER HEALTHY
   MAIN_PWR_FLT_TIMR : INT ;	//MAIN POWER FAULT TIMER
   MAIN_PWR_FLT_GEN_TIME : INT  := 3;	//MAIN POWER FAULT GENERATION TIME
   PULSE_1 : BOOL ;	//PULSE 1
   PULSE_2 : BOOL ;	//PULSE 2
   CTRL_PWR_FLT_TIMR : INT ;	//CONTROL POWER FAULT TIMER
   CTRL_PWR_FLT_GEN_TIME : INT  := 3;	//CONTROL POWER FAULT GENERATION TIME
  END_STRUCT ;	
BEGIN
   CTRL_PWR_FLT_GEN_TIME := 3;
END_DATA_BLOCK

DATA_BLOCK "HYDRAULIC_FUNCTIONS_DB"	// DB 2
AUTHOR : Kamillas
VERSION : 0.1
  STRUCT
   PUMP_1_RDY_FOR_STA : BOOL ;	//PUMP 1 READY FOR START
   PUMP_1_RUN_FB : BOOL ;	//PUMP 1 RUNNING FEEDBACK
   PUMP_1_OVR_LD_TRIP : BOOL ;	//PUMP 1 OVER LOAD TRIPPED
   PUMP_2_RDY_FOR_STA : BOOL ;	//PUMP 2 READY FOR START
   PUMP_2_RUN_FB : BOOL ;	//PUMP 2 RUNNING FEEDBACK
   PUMP_2_OVR_LD_TRIP : BOOL ;	//PUMP 2 OVER LOAD TRIPPED
   CIR_PUMP_RDY_FOR_STA : BOOL ;	//CIRCULATION PUMP READY FOR START
   CIR_PUMP_RUN_FB : BOOL ;	//CIRCULATION PUMP RUNNING FEEDBACK
   CIR_PUMP_OVR_LD_TRIP : BOOL ;	//CIRCULATION PUMP OVER LOAD TRIPPED
   COLR_FAN_RDY_FOR_STA : BOOL ;	//COOLER FAN READY FOR START
   COLR_FAN_RUN_FB : BOOL ;	//COOLER FAN RUNNING FEEDBACK
   COLR_FAN_OVR_LD_TRIP : BOOL ;	//COOLER FAN OVER LOAD TRIPPED
   CD_LCS_SS : BOOL ;	//CONTROL DESK / LOCAL CONTROL SELECTOR SWITCH
   PUMP_1_2_SS : BOOL ;	//PUMP 1 OR 2 SELECTOR SWITCH
   PUMP_1_STA_PB : BOOL ;	//PUMP 1 START PUSH BUTTON
   PUMP_1_STP_PB : BOOL ;	//PUMP 1 STOP PUSH BUTTON
   PUMP_2_STA_PB : BOOL ;	//PUMP 2 START PUSH BUTTON
   PUMP_2_STP_PB : BOOL ;	//PUMP 2 STOP PUSH BUTTON
   EMERGENCY_STOP_PB : BOOL ;	//EMERGENCY STOP PUSH BUTTON
   PUMP_1_2_SS_LCS : BOOL ;	//PUMP 1 OR 2 SELECTOR SWITCH LCS
   PUMP_1_STA_PB_LCS : BOOL ;	//PUMP 1 START PUSH BUTTON LCS
   PUMP_1_STP_PB_LCS : BOOL ;	//PUMP 1 STOP PUSH BUTTON LCS
   PUMP_2_STA_PB_LCS : BOOL ;	//PUMP 2 START PUSH BUTTON LCS
   PUMP_2_STP_PB_LCS : BOOL ;	//PUMP 2 STOP PUSH BUTTON LCS
   CIR_PUMP_STA_PB_LCS : BOOL ;	//CIRCULATION PUMP START PUSH BUTTON LCS
   CIR_PUMP_STP_PB_LCS : BOOL ;	//CIRCULATION PUMP STOP PUSH BUTTON LCS
   COLR_FAN_STA_PB_LCS : BOOL ;	//COOLER FAN START PUSH BUTTON LCS
   COLR_FAN_STP_PB_LCS : BOOL ;	//COOLER FAN STOP PUSH BUTTON LCS
   LAMP_TEST_PB_LCS_41 : BOOL ;	//LAMP TEST PUSH BUTTON LCS
   EMG_ACCM_STA_PB_LCS : BOOL ;	//EMERGENCY ACCUMULATOR START PB LCS
   EMG_ACCM_STP_PB_LCS : BOOL ;	//EMERGENCY ACCUMULATOR STOP PB LCS
   HTR_STA_PB_LCS : BOOL ;	//HEATER START PUSH BUTTON LCS
   HTR_STP_PB_LCS : BOOL ;	//HEATER STOP PUSH BUTTON LCS
   SHT_OF_VLV_LIN_1_FUL_OPN : BOOL ;	//SHUT OFF VALVE IN LINE 1 - FULLY OPEN
   SHT_OF_VLV_LIN_2_FUL_OPN : BOOL ;	//SHUT OFF VALVE IN LINE 2 - FULLY OPEN
   LOW_OIL_TEMP : BOOL ;	//LOW OIL TEMPERATURE - THERMOSTAT
   HIGH_OIL_TEMP : BOOL ;	//HIGH OIL TEMPERATURE - THERMOSTAT
   MAX_OIL_TEMP : BOOL ;	//MAXIMUM OIL TEMPERATURE - THERMOSTAT
   LOW_OIL_LEVEL : BOOL ;	//LOW OIL LEVEL - FLOAT SWITCH
   MIN_OIL_LEVEL : BOOL ;	//MINIMUM OIL LEVEL - FLOAT SWITCH
   RET_LIN_FLTR_CKD : BOOL ;	//RETURN LINE FILTER CHOKED
   LOW_OIL_PRESS : BOOL ;	//LOW OIL PRESSURE - PRESSURE SWITCH
   HIGH_OIL_PRESS : BOOL ;	//HIGH OIL PRESSURE - PRESSURE SWITCH
   PUMP_1_ON_CMD : BOOL ;	//PUMP 1 ON COMMAND
   PUMP_2_ON_CMD : BOOL ;	//PUMP 2 ON COMMAND
   CIR_PUMP_ON_CMD : BOOL ;	//CIRCULATION PUMP ON COMMAND
   CLR_FAN_ON_CMD : BOOL ;	//COOLER FAN ON COMMAND
   SYSTEM_RDY_IND : BOOL ;	//SYSTEM READY INDICATOR
   PUMP_1_ON_IND : BOOL ;	//PUMP 1 ON INDICATOR
   PUMP_2_ON_IND : BOOL ;	//PUMP 2 ON INDICATOR
   LCS_41_ON_IND_LCS : BOOL ;	//LCS 41 ON INDICATOR
   PUMP_1_ON_IND_LCS : BOOL ;	//PUMP 1 ON INDICATOR LCS
   PUMP_2_ON_IND_LCS : BOOL ;	//PUMP 2 ON INDICATOR LCS
   CIR_PUMP_ON_IND_LCS : BOOL ;	//CIRCULATION PUMP ON INDICATOR LCS
   CLR_FAN_ON_IND_LCS : BOOL ;	//COOLER FAN ON INDICATOR LCS
   HIGH_OIL_TEMP_IND_LCS : BOOL ;	//HIGH OIL TEMPERATURE INDICATOR LCS
   LOW_OIL_LEVEL_IND_LCS : BOOL ;	//LOW OIL LEVEL INDICATOR LCS
   LOW_OIL_TEMP_IND_LCS : BOOL ;	//LOW OIL TEMPERATURE INDICATOR LCS
   HTR_ON_IND_LCS : BOOL ;	//HEATER ON INDICATOR LCS
   FLTR_CHK_IND_LCS : BOOL ;	//FILTER CHOKE INDICATOR LCS
   ACCM_IN_OPER_IND_LCS : BOOL ;	//ACCUMULATOR IN OPERATION INDICATOR
   PRESS_REL_VLV_1_ON_CMD : BOOL ;	//PRESSURE RELIEF VALVE 1 ON COMMAND
   PRESS_REL_VLV_2_ON_CMD : BOOL ;	//PRESSURE RELIEF VALVE 2 ON COMMAND
   EMG_ACCM_ON_CMD : BOOL ;	//EMERGENCY ACCUMULLATOR ON COMMAND
   HYD_SYS_HEALTHY : BOOL ;	//HYDRAULIC SYSTEMS HEALTHY BIT
   PULSE_1 : BOOL ;	//PULSE 1
   PULSE_2 : BOOL ;	//PULSE 2
   PULSE_3 : BOOL ;	//PULSE 3
   PULSE_4 : BOOL ;	//PULSE 4
   PULSE_5 : BOOL ;	//PULSE 5
   PULSE_6 : BOOL ;	//PULSE 6
   HYD_PUMP_1_FLT : BOOL ;	//HYDRAULIC PUMP 1 FAULT
   HYD_PUMP_2_FLT : BOOL ;	//HYDRAULIC PUMP 2 FAULT
   HYD_PUMP_1_FLT_TMR : INT ;	//HYDRAULIC PUMP 1 FAULT TIMER
   HYD_PUMP_1_FLT_GEN_TIME : INT  := 3;	//HYDRAULIC PUMP 1 FAULT GEMERATION TIME
   HYD_PUMP_2_FLT_TMR : INT ;	//HYDRAULIC PUMP 2 FAULT TIMER
   HYD_PUMP_2_FLT_GEN_TIME2 : INT  := 3;	//HYDRAULIC PUMP 2 FAULT GEMERATION TIME
   PRS_REL_VLV_1_OPN_TMR : INT ;	//PRESSURE RELEIF VALVE 1 OPEN TIMER
   PRS_REL_VLV_1_OPN_ST_TIM : INT  := 8;	//PRESSURE RELEIF VALVE 1 OPEN SET TIME
   PRS_REL_VLV_2_OPN_TMR : INT ;	//PRESSURE RELEIF VALVE 2 OPEN TIMER
   PRS_REL_VLV_2_OPN_ST_TIM : INT  := 8;	//PRESSURE RELEIF VALVE 2 OPEN SET TIME
   CIR_PUMP_FLT : BOOL ;	//CIRCULATION PUMP 1 FAULT
   CLR_FAN_FLT : BOOL ;	//COOLER FAN FAULT
   CIR_PUMP_FLT_TMR : INT ;	//CIRCULATION PUMP FAULT TIMER
   CIR_PUMP_FLT_GEN_TIME : INT  := 3;	//CIRCULATION PUMP FAULT GEMERATION TIME
   CLR_FAN_FLT_TMR : INT ;	//HYDRAULIC PUMP 2 FAULT TIMER
   CLR_FAN_FLT_GEN_TIME : INT  := 3;	//COOLER FAN FAULT GEMERATION TIME
   HYD_SYS_RDY_BIT : BOOL ;	//HYDRAULIC SYSTEM READY BIT
   LOW_OIL_LEV_FOR_HMI : BOOL ;	//LOW OIL LEVEL LEVEL CREATED TO DISPLAY IN HMI
  END_STRUCT ;	
BEGIN
   HYD_PUMP_1_FLT_GEN_TIME := 3;
   HYD_PUMP_2_FLT_GEN_TIME2 := 3;
   PRS_REL_VLV_1_OPN_ST_TIM := 3;
   PRS_REL_VLV_2_OPN_ST_TIM := 8;
   CIR_PUMP_FLT_GEN_TIME := 3;
   CLR_FAN_FLT_GEN_TIME := 3;
END_DATA_BLOCK

DATA_BLOCK "TRAVEL_DRIVE_DB"	// DB 3
AUTHOR : Kamillas
VERSION : 0.1
  STRUCT
   TRA_GRP_1_RDY_FOR_STA : BOOL ;	//TRAVEL GROUP 1 READY FOR START
   TRA_GRP_1_RUN_FB : BOOL ;	//TRAVEL GROUP 1 RUNNING FEEDBACK
   TRA_MTR_1_OVLD_TRIP : BOOL ;	//TRAVEL MOTOR 1 OVER LOAD TRIP
   TRA_MTR_2_OVLD_TRIP : BOOL ;	//TRAVEL MOTOR 2 OVER LOAD TRIP
   TRA_MTR_1_ISO_ON_FB : BOOL ;	//TRAVEL MOTOR 1 ISOLATOR ON FEEDBACK
   TRA_MTR_2_ISO_ON_FB : BOOL ;	//TRAVEL MOTOR 2 ISOLATOR ON FEEDBACK
   TRA_GRP_2_RDY_FOR_STA : BOOL ;	//TRAVEL GROUP 2 READY FOR START
   TRA_GRP_2_RUN_FB : BOOL ;	//TRAVEL GROUP 2 RUNNING FEEDBACK
   TRA_MTR_3_OVLD_TRIP : BOOL ;	//TRAVEL MOTOR 3 OVER LOAD TRIP
   TRA_MTR_4_OVLD_TRIP : BOOL ;	//TRAVEL MOTOR 4 OVER LOAD TRIP
   TRA_MTR_3_ISO_ON_FB : BOOL ;	//TRAVEL MOTOR 3 ISOLATOR ON FEEDBACK
   TRA_MTR_4_ISO_ON_FB : BOOL ;	//TRAVEL MOTOR 4 ISOLATOR ON FEEDBACK
   TRA_GRP_1_BRK_RDY_FOR_ST : BOOL ;	//TRAVEL GROUP 1 BREAK READY FOR START
   TRA_GRP_1_BRK_ON_FB : BOOL ;	//TRAVEL GROUP 1 BREAK ON FEEDBACK
   SIR_RDY_FOR_STA : BOOL ;	//SIREN READY FOR START
   SIR_ON_FB : BOOL ;	//SIREN ON FEED BACK
   TRA_GRP_2_BRK_RDY_FOR_ST : BOOL ;	//TRAVEL GROUP 2 BREAK READY FOR START
   TRA_GRP_2_BRK_ON_FB : BOOL ;	//TRAVEL GROUP 2 BREAK ON FEEDBACK
   SIR_OLR_TRIP : BOOL ;	//SIREN ON OVER LOAD TRIP
   TRA_JOY_STK_HME_POS : BOOL ;	//TRAVEL JOY STICK HOME POSITION
   TRA_JOY_STK_DED_MAN_BTN : BOOL ;	//TRAVEL JOY DEAD MAN BUTTON
   TRA_MODE_AUTO_MAN_SS : BOOL ;	//TRAVEL MODE AUTO/MANUAL BUTTON
   AUTO_POS_ACK : BOOL ;	//AUTO POSITION ACKNOWLEDGE
   TRA_DRV_1_PROF_HARD_SS : BOOL ;	//TRAVEL DRIVE 1 PROFIBUS/HARD WIRE SELECTRO SWITCH
   TRA_DRV_1_ON_FB : BOOL ;	//TRAVEL DRIVE 1 ON FEEDBACK
   TRA_DRV_1_RDY_FOR_STA : BOOL ;	//TRAVEL DRIVE 1 READY FOR START
   TRA_DRV_1_TRP_FB : BOOL ;	//TRAVEL DRIVE 1 TRIP FEEDBACK
   TRA_DRV_2_PROF_HARD_SS : BOOL ;	//TRAVEL DRIVE 2 PROFIBUS/HARD WIRE SELECTRO SWITCH
   TRA_DRV_2_ON_FB : BOOL ;	//TRAVEL DRIVE 2 ON FEEDBACK
   TRA_DRV_2_RDY_FOR_STA : BOOL ;	//TRAVEL DRIVE 2 READY FOR START
   TRA_DRV_2_TRP_FB : BOOL ;	//TRAVEL DRIVE 2 TRIP FEEDBACK
   LIMIT_SW_END_FWD_FB : BOOL ;	//LIMIT SWITCH END FORWARD FEEDBACK
   LIMIT_SW_END_REV_FB : BOOL ;	//LIMIT SWITCH END REVERSE FEEDBACK
   TRA_GRP_1_ON_CMD : BOOL ;	//TRAVEL GROUP 1 ON COMMAND
   TRA_GRP_2_ON_CMD : BOOL ;	//TRAVEL GROUP 2 ON COMMAND
   TRA_GRP_1_BRK_ON_CMD : BOOL ;	//TRAVEL GROUP 1 BRAKE ON COMMAND
   SIREN_ON_CMD : BOOL ;	//SIREN ON COMMAND
   TRA_GRP_2_BRK_ON_CMD : BOOL ;	//TRAVEL GROUP 2 BRAKE ON COMMAND
   FLASHER_ON_CMD : BOOL ;	//FLASHER ON COMMAND
   TRA_PER_IND : BOOL ;	//TRAVEL PERMISSION INDICATOR
   AUTO_POS_ON : BOOL ;	//AUTO POSITION ON
   TRA_DRV_1_FWD_CMD : BOOL ;	//TRAVEL DRIVE 1 FORWARD COMMAND
   TRA_DRV_1_REV_CMD : BOOL ;	//TRAVEL DRIVE 1 REVERSE COMMAND
   TRA_DRV_2_FWD_CMD : BOOL ;	//TRAVEL DRIVE 2 FORWARD COMMAND
   TRA_DRV_2_REV_CMD : BOOL ;	//TRAVEL DRIVE 2 REVERSE COMMAND
   TRA_ILK_BIT : BOOL ;	//TRAVEL OPERATIONS INTERLOCK BIT
   TRA_JOY_STK_FWD_POS : BOOL ;	//TRAVEL JOY STICK FOWRWARD POSITION
   TRA_JOY_STK_REV_POS : BOOL ;	//TRAVEL JOY DEAD REVERSE POSITION
   TRA_ILK_INM_BIT_1 : BOOL ;	//TRAVEL INTERLOCK INTERMEDIATE BIT 1
   TRA_ILK_INM_BIT_2 : BOOL ;	//TRAVEL INTERLOCK INTERMEDIATE BIT 2
   TRA_ILK_INM_BIT_3 : BOOL ;	//TRAVEL INTERLOCK INTERMEDIATE BIT 3
   TRA_DRV_1_2_BRK_FLT : BOOL ;	//TRAVEL DRIVE BREAK 1 AND 2 FAULT
   TRA_DRV_1_2_BRK_FLT_TMR : INT ;	//TRAVEL DRIVE BREAK 1 AND 2 FAULT TIMER
   JS_SPD_REF_DI : DINT ;	//JOY STICK SPEED REFERENCE IN DOUBLE INTEGER
   JS_SPD_REF_NEG_RMD : INT ;	//JOY STICK SPEED REFERENCE CONVERTERD TO POSITIVE VALUE
   JS_SPD_REF_REAL : REAL ;	//JOY STICK SPEED REFERENCE IN REAL(FLOATING POINT)
   JS_SPD_REF_UN_SL_FLT : WORD ;	//JOY STICK SPEED REFERENCE UNSCALLING FAULT
   TRA_SPD_REF_VAL : INT ;	//TRAVEL SPEED REFERENCE VALUE
   TRA_SPD_REF_VAL_FRM_JS : INT ;	//TRAVEL SPEED REFERENCE VALUW FROM JOYSTICK
   PULSE_1 : BOOL ;	//PULSE 1
   PULSE_2 : BOOL ;	//PULSE 2
   PULSE_3 : BOOL ;	//PULSE 3
   PULSE_4 : BOOL ;	//PULSE 4
   TR_DRV_1_STATUS_WORD_1 : INT ;	//TRAVEL DRIVE 1 PROFIBUS STATUS WORD 1
   TR_DRV_1_STATUS_WORD_2 : INT ;	//TRAVEL DRIVE 1 PROFIBUS STATUS WORD 2
   TR_DRV_1_STATUS_WORD_3 : INT ;	//TRAVEL DRIVE 1 PROFIBUS STATUS WORD 3
   TR_DRV_1_STATUS_WORD_4 : INT ;	//TRAVEL DRIVE 1 PROFIBUS STATUS WORD 4
   TR_DRV_1_STATUS_WORD_5 : INT ;	//TRAVEL DRIVE 1 PROFIBUS STATUS WORD 5
   TR_DRV_1_STATUS_WORD_6 : INT ;	//TRAVEL DRIVE 1 PROFIBUS STATUS WORD 6
   TR_DRV_1_STATUS_WORD_7 : INT ;	//TRAVEL DRIVE 1 PROFIBUS STATUS WORD 7
   TR_DRV_1_STATUS_WORD_8 : INT ;	//TRAVEL DRIVE 1 PROFIBUS STATUS WORD 8
   TR_DRV_1_STATUS_WORD_9 : INT ;	//TRAVEL DRIVE 1 PROFIBUS STATUS WORD 9
   TR_DRV_1_STATUS_WORD_10 : INT ;	//TRAVEL DRIVE 1 PROFIBUS STATUS WORD 10
   TR_DRV_1_STATUS_WORD_11 : INT ;	//TRAVEL DRIVE 1 PROFIBUS STATUS WORD 11
   TR_DRV_1_STATUS_WORD_12 : INT ;	//TRAVEL DRIVE 1 PROFIBUS STATUS WORD 12
   TR_DRV_1_STATUS_WORD_13 : INT ;	//TRAVEL DRIVE 1 PROFIBUS STATUS WORD 13
   TR_DRV_1_STATUS_WORD_14 : INT ;	//TRAVEL DRIVE 1 PROFIBUS STATUS WORD 14
   TR_DRV_1_STATUS_WORD_15 : INT ;	//TRAVEL DRIVE 1 PROFIBUS STATUS WORD 15
   TR_DRV_1_STATUS_WORD_16 : INT ;	//TRAVEL DRIVE 1 PROFIBUS STATUS WORD 16
   TR_DRV_1_CONTROL_WORD_1 : INT ;	//TRAVEL DRIVE 1 PROFIBUS CONTROL WORD 1
   TR_DRV_1_CONTROL_WORD_2 : INT ;	//TRAVEL DRIVE 1 PROFIBUS CONTROL WORD 2
   TR_DRV_1_CONTROL_WORD_3 : INT ;	//TRAVEL DRIVE 1 PROFIBUS CONTROL WORD 3
   TR_DRV_1_CONTROL_WORD_4 : INT ;	//TRAVEL DRIVE 1 PROFIBUS CONTROL WORD 4
   TR_DRV_1_CONTROL_WORD_5 : INT ;	//TRAVEL DRIVE 1 PROFIBUS CONTROL WORD 5
   TR_DRV_1_CONTROL_WORD_6 : INT ;	//TRAVEL DRIVE 1 PROFIBUS CONTROL WORD 6
   TR_DRV_1_CONTROL_WORD_7 : INT ;	//TRAVEL DRIVE 1 PROFIBUS CONTROL WORD 7
   TR_DRV_1_CONTROL_WORD_8 : INT ;	//TRAVEL DRIVE 1 PROFIBUS CONTROL WORD 8
   TR_DRV_1_CONTROL_WORD_9 : INT ;	//TRAVEL DRIVE 1 PROFIBUS CONTROL WORD 9
   TR_DRV_1_CONTROL_WORD_10 : INT ;	//TRAVEL DRIVE 1 PROFIBUS CONTROL WORD 10
   TR_DRV_1_CONTROL_WORD_11 : INT ;	//TRAVEL DRIVE 1 PROFIBUS CONTROL WORD 11
   TR_DRV_1_CONTROL_WORD_12 : INT ;	//TRAVEL DRIVE 1 PROFIBUS CONTROL WORD 12
   TR_DRV_1_CONTROL_WORD_13 : INT ;	//TRAVEL DRIVE 1 PROFIBUS CONTROL WORD 13
   TR_DRV_1_CONTROL_WORD_14 : INT ;	//TRAVEL DRIVE 1 PROFIBUS CONTROL WORD 14
   TR_DRV_1_CONTROL_WORD_15 : INT ;	//TRAVEL DRIVE 1 PROFIBUS CONTROL WORD 15
   TR_DRV_1_CONTROL_WORD_16 : INT ;	//TRAVEL DRIVE 1 PROFIBUS CONTROL WORD 16
   TR_DRV_1_STAT_WORD_1_ERR : INT ;	//TRAVEL DRIVE 1 DRIVE STATUS WORD 1 READ ERROR
   TR_DRV_1_STAT_WORD_2_ERR : INT ;	//TRAVEL DRIVE 1 DRIVE STATUS WORD 2 READ ERROR
   TR_DRV_1_STAT_WORD_3_ERR : INT ;	//TRAVEL DRIVE 1 DRIVE STATUS WORD 3 READ ERROR
   TR_DRV_1_STAT_WORD_4_ERR : INT ;	//TRAVEL DRIVE 1 DRIVE STATUS WORD 4 READ ERROR
   TR_DRV_1_CTRL_WORD_1_ERR : INT ;	//TRAVEL DRIVE 1 DRIVE CONTROL WORD 1 WRITE ERROR
   TR_DRV_1_CTRL_WORD_2_ERR : INT ;	//TRAVEL DRIVE 1 DRIVE CONTROL WORD 2 WRITE ERROR
   TR_DRV_1_CTRL_WORD_3_ERR : INT ;	//TRAVEL DRIVE 1 DRIVE CONTROL WORD 3 WRITE ERROR
   TR_DRV_1_CTRL_WORD_4_ERR : INT ;	//TRAVEL DRIVE 1 DRIVE CONTROL WORD 4 WRITE ERROR
   TR_DRV_2_STATUS_WORD_1 : INT ;	//TRAVEL DRIVE 2 PROFIBUS STATUS WORD 1
   TR_DRV_2_STATUS_WORD_2 : INT ;	//TRAVEL DRIVE 2 PROFIBUS STATUS WORD 2
   TR_DRV_2_STATUS_WORD_3 : INT ;	//TRAVEL DRIVE 2 PROFIBUS STATUS WORD 3
   TR_DRV_2_STATUS_WORD_4 : INT ;	//TRAVEL DRIVE 2 PROFIBUS STATUS WORD 4
   TR_DRV_2_STATUS_WORD_5 : INT ;	//TRAVEL DRIVE 2 PROFIBUS STATUS WORD 5
   TR_DRV_2_STATUS_WORD_6 : INT ;	//TRAVEL DRIVE 2 PROFIBUS STATUS WORD 6
   TR_DRV_2_STATUS_WORD_7 : INT ;	//TRAVEL DRIVE 2 PROFIBUS STATUS WORD 7
   TR_DRV_2_STATUS_WORD_8 : INT ;	//TRAVEL DRIVE 2 PROFIBUS STATUS WORD 8
   TR_DRV_2_STATUS_WORD_9 : INT ;	//TRAVEL DRIVE 2 PROFIBUS STATUS WORD 9
   TR_DRV_2_STATUS_WORD_10 : INT ;	//TRAVEL DRIVE 2 PROFIBUS STATUS WORD 10
   TR_DRV_2_STATUS_WORD_11 : INT ;	//TRAVEL DRIVE 2 PROFIBUS STATUS WORD 11
   TR_DRV_2_STATUS_WORD_12 : INT ;	//TRAVEL DRIVE 2 PROFIBUS STATUS WORD 12
   TR_DRV_2_STATUS_WORD_13 : INT ;	//TRAVEL DRIVE 2 PROFIBUS STATUS WORD 13
   TR_DRV_2_STATUS_WORD_14 : INT ;	//TRAVEL DRIVE 2 PROFIBUS STATUS WORD 14
   TR_DRV_2_STATUS_WORD_15 : INT ;	//TRAVEL DRIVE 2 PROFIBUS STATUS WORD 15
   TR_DRV_2_STATUS_WORD_16 : INT ;	//TRAVEL DRIVE 2 PROFIBUS STATUS WORD 16
   TR_DRV_2_CONTROL_WORD_1 : INT ;	//TRAVEL DRIVE 2 PROFIBUS CONTROL WORD 1
   TR_DRV_2_CONTROL_WORD_2 : INT ;	//TRAVEL DRIVE 2 PROFIBUS CONTROL WORD 2
   TR_DRV_2_CONTROL_WORD_3 : INT ;	//TRAVEL DRIVE 2 PROFIBUS CONTROL WORD 3
   TR_DRV_2_CONTROL_WORD_4 : INT ;	//TRAVEL DRIVE 2 PROFIBUS CONTROL WORD 4
   TR_DRV_2_CONTROL_WORD_5 : INT ;	//TRAVEL DRIVE 2 PROFIBUS CONTROL WORD 5
   TR_DRV_2_CONTROL_WORD_6 : INT ;	//TRAVEL DRIVE 2 PROFIBUS CONTROL WORD 6
   TR_DRV_2_CONTROL_WORD_7 : INT ;	//TRAVEL DRIVE 2 PROFIBUS CONTROL WORD 7
   TR_DRV_2_CONTROL_WORD_8 : INT ;	//TRAVEL DRIVE 2 PROFIBUS CONTROL WORD 8
   TR_DRV_2_CONTROL_WORD_9 : INT ;	//TRAVEL DRIVE 2 PROFIBUS CONTROL WORD 9
   TR_DRV_2_CONTROL_WORD_10 : INT ;	//TRAVEL DRIVE 2 PROFIBUS CONTROL WORD 10
   TR_DRV_2_CONTROL_WORD_11 : INT ;	//TRAVEL DRIVE 2 PROFIBUS CONTROL WORD 11
   TR_DRV_2_CONTROL_WORD_12 : INT ;	//TRAVEL DRIVE 2 PROFIBUS CONTROL WORD 12
   TR_DRV_2_CONTROL_WORD_13 : INT ;	//TRAVEL DRIVE 2 PROFIBUS CONTROL WORD 13
   TR_DRV_2_CONTROL_WORD_14 : INT ;	//TRAVEL DRIVE 2 PROFIBUS CONTROL WORD 14
   TR_DRV_2_CONTROL_WORD_15 : INT ;	//TRAVEL DRIVE 2 PROFIBUS CONTROL WORD 15
   TR_DRV_2_CONTROL_WORD_16 : INT ;	//TRAVEL DRIVE 2 PROFIBUS CONTROL WORD 16
   TR_DRV_2_STAT_WORD_1_ERR : INT ;	//TRAVEL DRIVE 2 DRIVE STATUS WORD 1 READ ERROR
   TR_DRV_2_STAT_WORD_2_ERR : INT ;	//TRAVEL DRIVE 2 DRIVE STATUS WORD 2 READ ERROR
   TR_DRV_2_STAT_WORD_3_ERR : INT ;	//TRAVEL DRIVE 2 DRIVE STATUS WORD 3 READ ERROR
   TR_DRV_2_STAT_WORD_4_ERR : INT ;	//TRAVEL DRIVE 2 DRIVE STATUS WORD 4 READ ERROR
   TR_DRV_2_CTRL_WORD_1_ERR : INT ;	//TRAVEL DRIVE 2 DRIVE CONTROL WORD 1 WRITE ERROR
   TR_DRV_2_CTRL_WORD_2_ERR : INT ;	//TRAVEL DRIVE 2 DRIVE CONTROL WORD 2 WRITE ERROR
   TR_DRV_2_CTRL_WORD_3_ERR : INT ;	//TRAVEL DRIVE 2 DRIVE CONTROL WORD 3 WRITE ERROR
   TR_DRV_2_CTRL_WORD_4_ERR : INT ;	//TRAVEL DRIVE 2 DRIVE CONTROL WORD 4 WRITE ERROR
   DR_1_CW_B0_RDY_TO_OPER : BOOL ;	//TRAVEL DRIVE 1 CONTROL WORD BIT 0 - READY TO OPERATE - OFF1 - PROFIBUS
   DR_1_CW_B1_OFF_2 : BOOL ;	//TRAVEL DRIVE 1 CONTROL WORD BIT 1 - OFF2 - PROFIBUS
   DR_1_CW_B2_OFF_3 : BOOL ;	//TRAVEL DRIVE 1 CONTROL WORD BIT 2 - OFF3 - PROFIBUS
   DR_1_CW_B3_OPER_ENAB : BOOL ;	//TRAVEL DRIVE 1 CONTROL WORD BIT 3 - OPERATION ENABLE - PROFIBUS
   DR_1_CW_B4_RMP_OUT_ZERO : BOOL ;	//TRAVEL DRIVE 1 CONTROL WORD BIT 4 - RAMP OUT ZERO - PROFIBUS
   DR_1_CW_B5_RMP_HLD : BOOL ;	//TRAVEL DRIVE 1 CONTROL WORD BIT 5 - RAMP HOLD - PROFIBUS
   DR_1_CW_B6_RMP_IN_ZERO : BOOL ;	//TRAVEL DRIVE 1 CONTROL WORD BIT 6 - RAMP IN ZERO - PROFIBUS
   DR_1_CW_B7_FLT_RST : BOOL ;	//TRAVEL DRIVE 1 CONTROL WORD BIT 7 - FAULT RESET - PROFIBUS
   DR_1_CW_B8_INCH_1 : BOOL ;	//TRAVEL DRIVE 1 CONTROL WORD BIT 8 - INCHING 1 - PROFIBUS
   DR_1_CW_B9_INCH_2 : BOOL ;	//TRAVEL DRIVE 1 CONTROL WORD BIT 9 - INCHING 2 - PROFIBUS
   DR_1_CW_B10_RMT_CMD : BOOL ;	//TRAVEL DRIVE 1 CONTROL WORD BIT 10 - REMOTE COMMAND - PROFIBUS
   DR_1_CW_B11 : BOOL ;	//TRAVEL DRIVE 1 CONTROL WORD BIT 11 - DRIVE SPECIFIC - PROFOBUS
   DR_1_CW_B12 : BOOL ;	//TRAVEL DRIVE 1 CONTROL WORD BIT 12 - DRIVE SPECIFIC - PROFOBUS
   DR_1_CW_B13 : BOOL ;	//TRAVEL DRIVE 1 CONTROL WORD BIT 13 - DRIVE SPECIFIC - PROFOBUS
   DR_1_CW_B14 : BOOL ;	//TRAVEL DRIVE 1 CONTROL WORD BIT 14 - DRIVE SPECIFIC - PROFOBUS
   DR_1_CW_B15 : BOOL ;	//TRAVEL DRIVE 1 CONTROL WORD BIT 15 - DRIVE SPECIFIC - PROFOBUS
   DR_1_SW_B0_RDY_ON : BOOL ;	//TRAVEL DRIVE 1 STATUS WORD BIT 0 - READY TO OPERATE - OFF1 - PROFIBUS
   DR_1_SW_B1_RDY_TO_OPER : BOOL ;	//TRAVEL DRIVE 1 STATUS WORD BIT 1 - REDY TO OPERATE - PROFIBUS
   DR_1_SW_B2_REF_RDY : BOOL ;	//TRAVEL DRIVE 1 STATUS WORD BIT 2 - ENABEL OPERATION - PROFIBUS
   DR_1_SW_B3_TRIPPED : BOOL ;	//TRAVEL DRIVE 1 STATUS WORD BIT 3 - FAULT - PROFIBUS
   DR_1_SW_B4_OFF_2_STA : BOOL ;	//TRAVEL DRIVE 1 STATUS WORD BIT 4 - OFF 2 STATUS - PROFIBUS
   DR_1_SW_B5_OFF_3_STA : BOOL ;	//TRAVEL DRIVE 1 STATUS WORD BIT 5 - OFF 3 STATUS - PROFIBUS
   DR_1_SW_B6_SWC_ON_INHB : BOOL ;	//TRAVEL DRIVE 1 STATUS WORD BIT 6 - SWITCH ON INHIBIT - PROFIBUS
   DR_1_SW_B7_ALARM : BOOL ;	//TRAVEL DRIVE 1 STATUS WORD BIT 7 - WARNING/ALARM - PROFIBUS
   DR_1_SW_B8_AT_SETPOINT : BOOL ;	//TRAVEL DRIVE 1 STATUS WORD BIT 8 - OPERATING - PROFIBUS
   DR_1_SW_B9_REMOTE : BOOL ;	//TRAVEL DRIVE 1 STATUS WORD BIT 9 - DRIVE CONTROL REMOTE\LOCAL - PROFIBUS
   DR_1_SW_B10_ABOVE_LIMIT : BOOL ;	//TRAVEL DRIVE 1 STATUS WORD BIT 10 - SPEED ABOVE LIMIT - PROFIBUS
   DR_1_SW_B11 : BOOL ;	//TRAVEL DRIVE 1 STATUS WORD BIT 11 - DRIVE SPECIFIC - PROFOBUS
   DR_1_SW_B12 : BOOL ;	//TRAVEL DRIVE 1 STATUS WORD BIT 12 - DRIVE SPECIFIC - PROFOBUS
   DR_1_SW_B13 : BOOL ;	//TRAVEL DRIVE 1 STATUS WORD BIT 13 - DRIVE SPECIFIC - PROFOBUS
   DR_1_SW_B14 : BOOL ;	//TRAVEL DRIVE 1 STATUS WORD BIT 14 - DRIVE SPECIFIC - PROFOBUS
   DR_1_SW_B15 : BOOL ;	//TRAVEL DRIVE 1 STATUS WORD BIT 15 - DRIVE SPECIFIC - PROFOBUS
   JS_SPD_REF_DI_PF : DINT ;	//JOY STICK SPEED REFERENCE IN DOUBLE INTEGER
   JS_SPD_REF_REAL_PF : REAL ;	//JOY STICK SPEED REFERENCE IN REAL(FLOATING POINT)
   JS_SPD_REF_UN_SL_FLT_PF : WORD ;	//JOY STICK SPEED REFERENCE UNSCALLING FAULT
   TRA_SPD_REF_VAL_PF : INT ;	//TRAVEL SPEED REFERENCE VALUE
   DR_2_CW_B0_RDY_TO_OPER : BOOL ;	//TRAVEL DRIVE 2 CONTROL WORD BIT 0 - READY TO OPERATE - OFF1 - PROFIBUS
   DR_2_CW_B1_OFF_2 : BOOL ;	//TRAVEL DRIVE 2 CONTROL WORD BIT 1 - OFF2 - PROFIBUS
   DR_2_CW_B2_OFF_3 : BOOL ;	//TRAVEL DRIVE 2 CONTROL WORD BIT 2 - OFF3 - PROFIBUS
   DR_2_CW_B3_OPER_ENAB : BOOL ;	//TRAVEL DRIVE 2 CONTROL WORD BIT 3 - OPERATION ENABLE - PROFIBUS
   DR_2_CW_B4_RMP_OUT_ZERO : BOOL ;	//TRAVEL DRIVE 2 CONTROL WORD BIT 4 - RAMP OUT ZERO - PROFIBUS
   DR_2_CW_B5_RMP_HLD : BOOL ;	//TRAVEL DRIVE 2 CONTROL WORD BIT 5 - RAMP HOLD - PROFIBUS
   DR_2_CW_B6_RMP_IN_ZERO : BOOL ;	//TRAVEL DRIVE 2 CONTROL WORD BIT 6 - RAMP IN ZERO - PROFIBUS
   DR_2_CW_B7_FLT_RST : BOOL ;	//TRAVEL DRIVE 2 CONTROL WORD BIT 7 - FAULT RESET - PROFIBUS
   DR_2_CW_B8_INCH_1 : BOOL ;	//TRAVEL DRIVE 2 CONTROL WORD BIT 8 - INCHING 1 - PROFIBUS
   DR_2_CW_B9_INCH_2 : BOOL ;	//TRAVEL DRIVE 2 CONTROL WORD BIT 9 - INCHING 2 - PROFIBUS
   DR_2_CW_B10_RMT_CMD : BOOL ;	//TRAVEL DRIVE 2 CONTROL WORD BIT 10 - REMOTE COMMAND - PROFIBUS
   DR_2_CW_B11 : BOOL ;	//TRAVEL DRIVE 2 CONTROL WORD BIT 11 - DRIVE SPECIFIC - PROFOBUS
   DR_2_CW_B12 : BOOL ;	//TRAVEL DRIVE 2 CONTROL WORD BIT 12 - DRIVE SPECIFIC - PROFOBUS
   DR_2_CW_B13 : BOOL ;	//TRAVEL DRIVE 2 CONTROL WORD BIT 13 - DRIVE SPECIFIC - PROFOBUS
   DR_2_CW_B14 : BOOL ;	//TRAVEL DRIVE 2 CONTROL WORD BIT 14 - DRIVE SPECIFIC - PROFOBUS
   DR_2_CW_B15 : BOOL ;	//TRAVEL DRIVE 2 CONTROL WORD BIT 15 - DRIVE SPECIFIC - PROFOBUS
   DR_2_SW_B0_RDY_ON : BOOL ;	//TRAVEL DRIVE 2 STATUS WORD BIT 0 - READY TO OPERATE - OFF1 - PROFIBUS
   DR_2_SW_B1_RDY_TO_OPER : BOOL ;	//TRAVEL DRIVE 2 STATUS WORD BIT 1 - REDY TO OPERATE - PROFIBUS
   DR_2_SW_B2_REF_RDY : BOOL ;	//TRAVEL DRIVE 2 STATUS WORD BIT 2 - ENABEL OPERATION - PROFIBUS
   DR_2_SW_B3_TRIPPED : BOOL ;	//TRAVEL DRIVE 2 STATUS WORD BIT 3 - FAULT - PROFIBUS
   DR_2_SW_B4_OFF_2_STA : BOOL ;	//TRAVEL DRIVE 2 STATUS WORD BIT 4 - OFF 2 STATUS - PROFIBUS
   DR_2_SW_B5_OFF_3_STA : BOOL ;	//TRAVEL DRIVE 2 STATUS WORD BIT 5 - OFF 3 STATUS - PROFIBUS
   DR_2_SW_B6_SWC_ON_INHB : BOOL ;	//TRAVEL DRIVE 2 STATUS WORD BIT 6 - SWITCH ON INHIBIT - PROFIBUS
   DR_2_SW_B7_ALARM : BOOL ;	//TRAVEL DRIVE 2 STATUS WORD BIT 7 - WARNING/ALARM - PROFIBUS
   DR_2_SW_B8_AT_SETPOINT : BOOL ;	//TRAVEL DRIVE 2 STATUS WORD BIT 8 - OPERATING - PROFIBUS
   DR_2_SW_B9_REMOTE : BOOL ;	//TRAVEL DRIVE 2 STATUS WORD BIT 9 - DRIVE CONTROL REMOTE\LOCAL - PROFIBUS
   DR_2_SW_B10_ABOVE_LIMIT : BOOL ;	//TRAVEL DRIVE 2 STATUS WORD BIT 10 - SPEED ABOVE LIMIT - PROFIBUS
   DR_2_SW_B11 : BOOL ;	//TRAVEL DRIVE 2 STATUS WORD BIT 11 - DRIVE SPECIFIC - PROFOBUS
   DR_2_SW_B12 : BOOL ;	//TRAVEL DRIVE 2 STATUS WORD BIT 12 - DRIVE SPECIFIC - PROFOBUS
   DR_2_SW_B13 : BOOL ;	//TRAVEL DRIVE 2 STATUS WORD BIT 13 - DRIVE SPECIFIC - PROFOBUS
   DR_2_SW_B14 : BOOL ;	//TRAVEL DRIVE 2 STATUS WORD BIT 14 - DRIVE SPECIFIC - PROFOBUS
   DR_2_SW_B15 : BOOL ;	//TRAVEL DRIVE 2 STATUS WORD BIT 15 - DRIVE SPECIFIC - PROFOBUS
   DR_1_ACT_SPD_PF : REAL ;	//TRAVEL DRIVE 1 ACTUAL SPEED - PROFIBUS
   DR_1_ACT_SPD_SCL_ERR : WORD ;	//TRAVEL DRIVE 1 ACTUAL SPEED SCALING ERROR - PROFIBUS
   DR_2_ACT_SPD_PF : REAL ;	//TRAVEL DRIVE 2 ACTUAL SPEED - PROFIBUS
   DR_2_ACT_SPD_SCL_ERR : WORD ;	//TRAVEL DRIVE 2 ACTUAL SPEED SCALING ERROR - PROFIBUS
   TRA_DRV_1_FWD_CMD_PF : BOOL ;	//TRAVEL DRIVE 1 FORWARD COMMAND THROUGH PROFIBUS
   TRA_DRV_1_REV_CMD_PF : BOOL ;	//TRAVEL DRIVE 1 REVERSE COMMAND THROUGH PROFIBUS
   TRA_DRV_2_FWD_CMD_PF : BOOL ;	//TRAVEL DRIVE 2 FORWARD COMMAND THROUGH PROFIBUS
   TRA_DRV_2_REV_CMD_PF : BOOL ;	//TRAVEL DRIVE 2 REVERSE COMMAND THROUGH PROFIBUS
   TRA_FWD_CHNG_OVR_DEL : BOOL ;	//TRAVEL DRIVE FORWARD CHANGE OVER DELAY
   TRA_REV_CHNG_OVR_DEL : BOOL ;	//TRAVEL DRIVE REVERSE CHANGE OVER DELAY
   TRA_DRV_MAN_JS_ANA_IN : INT ;	//TRAVEL DRIVE MANUAL MODE JOYSTICK ANALOG INPPUT
   TRA_DRV_ATUO_PF_ANA_IN : INT ;	//TRAVEL DRIVE AUTO MODE ANALOG INPUT THROUGH PROFIBUS FROM TATA PLC
   TRA_DRV_SPD_REF_HW_OUT : INT ;	//TRAVEL DRIVE SPEED REFERENCE THROUGH ANALOG OUTPUT
   TRA_DRV_SPD_REF_PF_OUT : INT ;	//TRAVEL DRIVE SPEED REFERENCE THROUGH PROFIBUS OUTPUT
   TRA_AUTO_POS_ACK_SET : BOOL ;	//TRAVEL AUTO POSITIONING ACKNOWLEDGE
   TRA_SIREN_ON_PB : BOOL ;	//TRAVEL SIREN PUSH BUTTON
   TRA_SIREN_ON_COMMAND : BOOL ;	//TRAVEL SIREN ON COMMAND
  END_STRUCT ;	
BEGIN
END_DATA_BLOCK

DATA_BLOCK "PUSHER_RAM_DB"	// DB 4
AUTHOR : Kamillas
VERSION : 0.1
  STRUCT
   PUSH_BRK_RDY_FOR_STA : BOOL ;	//PUSHER BRAKE READY FOR START
   PUSH_MTR_BRK_ON_FB : BOOL ;	//PUSHER MOTOR BRAKE ON FEEDBCAK
   PUSH_RAM_STP_PB : BOOL ;	//PUSHER RAM STOP PUSH BUTTON
   PUSH_MAN_SS : BOOL ;	//PUSHER MANUAL SELECTOR SWTICH
   PUSH_AUTO_SS : BOOL ;	//PUSHER AUTO SELECTOR SWITCH
   PUSH_DRV_PROF_HDWR_SS : BOOL ;	//PUSHER DRIVE PROFIBUS/HARDWIRE SELECTOR SWITCH
   PUSH_DRV_ON_FB : BOOL ;	//PUSHER DRIVE ON FEED BACK
   PUSH_DRV_RDY_FOR_STA : BOOL ;	//PUSHER DRIVE READY FOR START
   PUSH_DRV_TRP_FB : BOOL ;	//PUSHER DRIVE TRIP FEED BACK
   PUSH_RLS_OVN_FACE_RCHD : BOOL ;	//PUSHER RLS OVEN FACE REACHED
   PUSH_RLS_GUIDE_ENT : BOOL ;	//PUSHER RLS GUIDE ENTRY
   PUSH_RLS_FWD_END : BOOL ;	//PUSHER RLS FORWARD END
   PUSH_RLS_STND_PIPE : BOOL ;	//PUSHER RLS STAND PIPE
   PUSH_RLS_REV_END : BOOL ;	//PUSHER RLS REVERSE END
   PUSH_EM_DRV_ENG : BOOL ;	//PUSHER EMERGENCY DRIVE ENGAGE
   PUSH_EM_DRV_DIS_ENG : BOOL ;	//PUSHER EMERGENCY DRIVE DISENGAGE
   EMERGENCY_PB_LCS_15 : BOOL ;	//EMERGENCY PUSH BUTTON
   RAM_EMG_DRV_DIS_ENG : BOOL ;	//RAM EMERGENCY DRIVE DISENGAGE
   RAM_END_FWD_LS : BOOL ;	//RAM END FORWARD LIMIT SWITCH
   RAM_END_RET_LS : BOOL ;	//RAM END RETRACT LIMIT SWITCH
   PUSH_RAM_BRK_ON_CMD : BOOL ;	//PUSHER RAM BREAK ON COMMAND
   PREP_FOR_PUSH_IND : BOOL ;	//PREPARE FOR PUSHING INDICATOR
   PUSH_DRV_FWD_CMD : BOOL ;	//PUSHER DRIVE FORWARD COMMAND
   PUSH_DRV_REV_CMD : BOOL ;	//PUSHER DRIVE REVERSE COMMAND
   LOCAL_SEL_IND_LCS_15 : BOOL ;	//LOCAL SELECTION INDICATOR LCS-15
   PUSH_RAM_ILK_1 : BOOL ;	//PUSHER RAM INTERLOCK BIT 1
   PUSH_RAM_ILK : BOOL ;	//PUSHER RAM INTERLOCK BIT
   JS_HME_POS : BOOL ;	//JOYSTICK HOME POSITION
   JS_FWD_POS : BOOL ;	//JOYSTICK FORWARD POSITION
   JS_REV_POS : BOOL ;	//JOYSTICK REVERSE POSITION
   JS_DEAD_MAN_BUTTON : BOOL ;	//JOYSTICK DEAD MAN BUTTON
   JS_SPD_REF_DI : DINT ;	//JOY STICK SPEED REFERENCE IN DOUBLE INTEGER
   JS_SPD_REF_NEG_RMD : INT ;	//JOY STICK SPEED REFERENCE CONVERTERD TO POSITIVE VALUE
   JS_SPD_REF_REAL : REAL ;	//JOY STICK SPEED REFERENCE IN REAL(FLOATING POINT)
   JS_SPD_REF_UN_SL_FLT : WORD ;	//JOY STICK SPEED REFERENCE UNSCALLING FAULT
   PUSH_SPD_REF_VAL : INT ;	//PUSHER SPEED REFERENCE VALUE
   PUSH_DRV_BRK_FLT : BOOL ;	//PUSHER DRIVE BREAK FAULT
   PUSH_DRV_BRK_FLT_TMR : INT ;	//PUSHER DRIVE BREAK FAULT TIMER
   PUSH_ILK_BYPASS : BOOL ;	//PUSHER RAM INTERLOCK BYPASS INPUT
   PUSH_RAM_REV_END_IND : BOOL ;	//PUSHER RAM REVERSE END INDICATOR
   PUSH_PERM_IND : BOOL ;	//PUSHER PERMISION INDICATION
   PUSH_DRV_STATUS_WORD_1 : INT ;	//PUSHER PROFIBUS STATUS WORD 1
   PUSH_DRV_STATUS_WORD_2 : INT ;	//PUSHER PROFIBUS STATUS WORD 2
   PUSH_DRV_STATUS_WORD_3 : INT ;	//PUSHER PROFIBUS STATUS WORD 3
   PUSH_DRV_STATUS_WORD_4 : INT ;	//PUSHER PROFIBUS STATUS WORD 4
   PUSH_DRV_CONTROL_WORD_1 : INT ;	//PUSHER PROFIBUS CONTROL WORD 1
   PUSH_DRV_CONTROL_WORD_2 : INT ;	//PUSHER PROFIBUS CONTROL WORD 2
   PUSH_DRV_CONTROL_WORD_3 : INT ;	//PUSHER PROFIBUS CONTROL WORD 3
   PUSH_DRV_CONTROL_WORD_4 : INT ;	//PUSHER PROFIBUS CONTROL WORD 4
   PUSH_DRV_STAT_WORD_1_ERR : INT ;	//PUSHER DRIVE STATUS WORD 1 READ ERROR
   PUSH_DRV_STAT_WORD_2_ERR : INT ;	//PUSHER DRIVE STATUS WORD 2 READ ERROR
   PUSH_DRV_STAT_WORD_3_ERR : INT ;	//PUSHER DRIVE STATUS WORD 3 READ ERROR
   PUSH_DRV_STAT_WORD_4_ERR : INT ;	//PUSHER DRIVE STATUS WORD 4 READ ERROR
   PUSH_DRV_CTRL_WORD_1_ERR : INT ;	//PUSHER DRIVE CONTROL WORD 1 WRITE ERROR
   PUSH_DRV_CTRL_WORD_2_ERR : INT ;	//PUSHER DRIVE CONTROL WORD 2 WRITE ERROR
   PUSH_DRV_CTRL_WORD_3_ERR : INT ;	//PUSHER DRIVE CONTROL WORD 3 WRITE ERROR
   PUSH_DRV_CTRL_WORD_4_ERR : INT ;	//PUSHER DRIVE CONTROL WORD 4 WRITE ERROR
   PUSH_FWD_REV_COUNT : INT ;	//PUSHER FORWARD REVERSE COUNT
   PUSH_FWD_REV_COUNT_SET : INT  := 3;	//PUSHER FORWARD REVERSE COUNT SET POINT
   PUSH_AUTO_CNT_RCHD : BOOL ;	//PUSHER AUTO COUNT REACHED
   PUSH_FST_TIM_FWD_END_RCH : BOOL ;	//PUSHER REACHED THE FORWARD END FOR FIRST TIME
   PUSH_AUTO_STA_PB : BOOL ;	//PUSHER AUTO START PUSH BUTTON
   PUSH_AUTO_STP_RET_PB : BOOL ;	//PUSHER AUTO STOP AND RETRACT PUSH BUTTON
   PUSH_AUTO_STA : BOOL ;	//PUSHER AUTO START
   PUSH_AUTO_STP_RET : BOOL ;	//PUSHER AUTO STOP AND RETRACT
   PULSE_1 : BOOL ;	//PULSE 1
   PULSE_2 : BOOL ;	//PULSE 2
   PULSE_3 : BOOL ;	//PULSE 3
   PULSE_4 : BOOL ;	//PULSE 4
   STA_PUSH_IND : BOOL ;	//START PUSHING INDICATION IN AUTO MODE
   PUSH_SPD_REF_VAL_FRM_JS : INT ;	//PUSHER SPEED REFERENCE VALUW FROM JOYSTICK
   PUSH_DE_CARB_VLV : BOOL ;	//PUSHER RAM DECARBONISING VALVE
   PUSH_RACK_TEETH_VLV : BOOL ;	//PSUHER RAM RACK TEETH VALVE
   PUSH_TRA_DIST : REAL ;	//PUSHER TRAVELED DISTANCE
   PUSH_ENC_VAL : INT ;	//PUSHER ENCODER VALUE THROUGH PROFIBUS
   PUSH_ENC_VAL_DI : DINT ;	//PUSHER ENCODER VALUE IN DOUBLE INT FORMAR
   PUSH_ENC_VAL_REAL : REAL ;	//PUSHER ENCODER VALUE IN REAL FORMAT
   PUSH_ENC_NO_OF_REV : REAL ;	//PUSHER ENCODER NO OF REVOLUTIONS
   PUSH_ENC_VAL_RST : BOOL ;	//PUSHER ENCODER VALUE RESET
   DRV_STATUS_WORD_1 : INT ;	//PUSHER DRIVE PROFIBUS STATUS WORD 1
   DRV_STATUS_WORD_2 : INT ;	//PUSHER DRIVE PROFIBUS STATUS WORD 2
   DRV_STATUS_WORD_3 : INT ;	//PUSHER DRIVE PROFIBUS STATUS WORD 3
   DRV_STATUS_WORD_4 : INT ;	//PUSHER DRIVE PROFIBUS STATUS WORD 4
   DRV_STATUS_WORD_5 : INT ;	//PUSHER DRIVE PROFIBUS STATUS WORD 5
   DRV_STATUS_WORD_6 : INT ;	//PUSHER DRIVE PROFIBUS STATUS WORD 6
   DRV_STATUS_WORD_7 : INT ;	//PUSHER DRIVE PROFIBUS STATUS WORD 7
   DRV_STATUS_WORD_8 : INT ;	//PUSHER DRIVE PROFIBUS STATUS WORD 8
   DRV_STATUS_WORD_9 : INT ;	//PUSHER DRIVE PROFIBUS STATUS WORD 9
   DRV_STATUS_WORD_10 : INT ;	//PUSHER DRIVE PROFIBUS STATUS WORD 10
   DRV_STATUS_WORD_11 : INT ;	//PUSHER DRIVE PROFIBUS STATUS WORD 11
   DRV_STATUS_WORD_12 : INT ;	//PUSHER DRIVE PROFIBUS STATUS WORD 12
   DRV_STATUS_WORD_13 : INT ;	//PUSHER DRIVE PROFIBUS STATUS WORD 13
   DRV_STATUS_WORD_14 : INT ;	//PUSHER DRIVE PROFIBUS STATUS WORD 14
   DRV_STATUS_WORD_15 : INT ;	//PUSHER DRIVE PROFIBUS STATUS WORD 15
   DRV_STATUS_WORD_16 : INT ;	//PUSHER DRIVE PROFIBUS STATUS WORD 16
   DRV_CONTROL_WORD_1 : INT ;	//PUSHER DRIVE PROFIBUS CONTROL WORD 1
   DRV_CONTROL_WORD_2 : INT ;	//PUSHER DRIVE PROFIBUS CONTROL WORD 2
   DRV_CONTROL_WORD_3 : INT ;	//PUSHER DRIVE PROFIBUS CONTROL WORD 3
   DRV_CONTROL_WORD_4 : INT ;	//PUSHER DRIVE PROFIBUS CONTROL WORD 4
   DRV_CONTROL_WORD_5 : INT ;	//PUSHER DRIVE PROFIBUS CONTROL WORD 5
   DRV_CONTROL_WORD_6 : INT ;	//PUSHER DRIVE PROFIBUS CONTROL WORD 6
   DRV_CONTROL_WORD_7 : INT ;	//PUSHER DRIVE PROFIBUS CONTROL WORD 7
   DRV_CONTROL_WORD_8 : INT ;	//PUSHER DRIVE PROFIBUS CONTROL WORD 8
   DRV_CONTROL_WORD_9 : INT ;	//PUSHER DRIVE PROFIBUS CONTROL WORD 9
   DRV_CONTROL_WORD_10 : INT ;	//PUSHER DRIVE PROFIBUS CONTROL WORD 10
   DRV_CONTROL_WORD_11 : INT ;	//PUSHER DRIVE PROFIBUS CONTROL WORD 11
   DRV_CONTROL_WORD_12 : INT ;	//PUSHER DRIVE PROFIBUS CONTROL WORD 12
   DRV_CONTROL_WORD_13 : INT ;	//PUSHER DRIVE PROFIBUS CONTROL WORD 13
   DRV_CONTROL_WORD_14 : INT ;	//PUSHER DRIVE PROFIBUS CONTROL WORD 14
   DRV_CONTROL_WORD_15 : INT ;	//PUSHER DRIVE PROFIBUS CONTROL WORD 15
   DRV_CONTROL_WORD_16 : INT ;	//PUSHER DRIVE PROFIBUS CONTROL WORD 16
   DRV_STAT_WORD_1_ER : INT ;	//PUSHER DRIVE DRIVE STATUS WORD 1 READ ERROR
   DRV_STAT_WORD_2_ER : INT ;	//PUSHER DRIVE DRIVE STATUS WORD 2 READ ERROR
   DRV_STAT_WORD_3_ER : INT ;	//PUSHER DRIVE DRIVE STATUS WORD 3 READ ERROR
   DRV_STAT_WORD_4_ER : INT ;	//PUSHER DRIVE DRIVE STATUS WORD 4 READ ERROR
   DRV_CTRL_WORD_1_ER : INT ;	//PUSHER DRIVE DRIVE CONTROL WORD 1 WRITE ERROR
   DRV_CTRL_WORD_2_ER : INT ;	//PUSHER DRIVE DRIVE CONTROL WORD 2 WRITE ERROR
   DRV_CTRL_WORD_3_ER : INT ;	//PUSHER DRIVE DRIVE CONTROL WORD 3 WRITE ERROR
   DRV_CTRL_WORD_4_ER : INT ;	//PUSHER DRIVE DRIVE CONTROL WORD 4 WRITE ERROR
   DRV_CW_B0_RDY_TO_OPER : BOOL ;	//PUSHER DRIVE CONTROL WORD BIT 0 - READY TO OPERATE - OFF1 - PROFIBUS
   DRV_CW_B1_OFF_2 : BOOL ;	//PUSHER DRIVE CONTROL WORD BIT 1 - OFF2 - PROFIBUS
   DRV_CW_B2_OFF_3 : BOOL ;	//PUSHER DRIVE CONTROL WORD BIT 2 - OFF3 - PROFIBUS
   DRV_CW_B3_OPER_ENAB : BOOL ;	//PUSHER DRIVE CONTROL WORD BIT 3 - OPERATION ENABLE - PROFIBUS
   DRV_CW_B4_RMP_OUT_ZERO : BOOL ;	//PUSHER DRIVE CONTROL WORD BIT 4 - RAMP OUT ZERO - PROFIBUS
   DRV_CW_B5_RMP_HLD : BOOL ;	//PUSHER DRIVE CONTROL WORD BIT 5 - RAMP HOLD - PROFIBUS
   DRV_CW_B6_RMP_IN_ZERO : BOOL ;	//PUSHER DRIVE CONTROL WORD BIT 6 - RAMP IN ZERO - PROFIBUS
   DRV_CW_B7_FLT_RST : BOOL ;	//PUSHER DRIVE CONTROL WORD BIT 7 - FAULT RESET - PROFIBUS
   DRV_CW_B8_INCH_1 : BOOL ;	//PUSHER DRIVE CONTROL WORD BIT 8 - INCHING 1 - PROFIBUS
   DRV_CW_B9_INCH_2 : BOOL ;	//PUSHER DRIVE CONTROL WORD BIT 9 - INCHING 2 - PROFIBUS
   DRV_CW_B10_RMT_CMD : BOOL ;	//PUSHER DRIVE CONTROL WORD BIT 10 - REMOTE COMMAND - PROFIBUS
   DRV_CW_B11 : BOOL ;	//PUSHER DRIVE CONTROL WORD BIT 11 - DRIVE SPECIFIC - PROFOBUS
   DRV_CW_B12 : BOOL ;	//PUSHER DRIVE CONTROL WORD BIT 12 - DRIVE SPECIFIC - PROFOBUS
   DRV_CW_B13 : BOOL ;	//PUSHER DRIVE CONTROL WORD BIT 13 - DRIVE SPECIFIC - PROFOBUS
   DRV_CW_B14 : BOOL ;	//PUSHER DRIVE CONTROL WORD BIT 14 - DRIVE SPECIFIC - PROFOBUS
   DRV_CW_B15 : BOOL ;	//PUSHER DRIVE CONTROL WORD BIT 15 - DRIVE SPECIFIC - PROFOBUS
   DRV_SW_B0_RDY_ON : BOOL ;	//PUSHER DRIVE STATUS WORD BIT 0 - READY TO OPERATE - OFF1 - PROFIBUS
   DRV_SW_B1_RDY_TO_OPER : BOOL ;	//PUSHER DRIVE STATUS WORD BIT 1 - REDY TO OPERATE - PROFIBUS
   DRV_SW_B2_REF_RDY : BOOL ;	//PUSHER DRIVE STATUS WORD BIT 2 - ENABEL OPERATION - PROFIBUS
   DRV_SW_B3_TRIPPED : BOOL ;	//PUSHER DRIVE STATUS WORD BIT 3 - FAULT - PROFIBUS
   DRV_SW_B4_OFF_2_STA : BOOL ;	//PUSHER DRIVE STATUS WORD BIT 4 - OFF 2 STATUS - PROFIBUS
   DRV_SW_B5_OFF_3_STA : BOOL ;	//PUSHER DRIVE STATUS WORD BIT 5 - OFF 3 STATUS - PROFIBUS
   DRV_SW_B6_SWC_ON_INHB : BOOL ;	//PUSHER DRIVE STATUS WORD BIT 6 - SWITCH ON INHIBIT - PROFIBUS
   DRV_SW_B7_ALARM : BOOL ;	//PUSHER DRIVE STATUS WORD BIT 7 - WARNING/ALARM - PROFIBUS
   DRV_SW_B8_AT_SETPOINT : BOOL ;	//PUSHER DRIVE STATUS WORD BIT 8 - OPERATING - PROFIBUS
   DRV_SW_B9_REMOTE : BOOL ;	//PUSHER DRIVE STATUS WORD BIT 9 - DRIVE CONTROL REMOTE\LOCAL - PROFIBUS
   DRV_SW_B10_ABOVE_LIMIT : BOOL ;	//PUSHER DRIVE STATUS WORD BIT 10 - SPEED ABOVE LIMIT - PROFIBUS
   DRV_SW_B11 : BOOL ;	//PUSHER DRIVE STATUS WORD BIT 11 - DRIVE SPECIFIC - PROFOBUS
   DRV_SW_B12 : BOOL ;	//PUSHER DRIVE STATUS WORD BIT 12 - DRIVE SPECIFIC - PROFOBUS
   DRV_SW_B13 : BOOL ;	//PUSHER DRIVE STATUS WORD BIT 13 - DRIVE SPECIFIC - PROFOBUS
   DRV_SW_B14 : BOOL ;	//PUSHER DRIVE STATUS WORD BIT 14 - DRIVE SPECIFIC - PROFOBUS
   DRV_SW_B15 : BOOL ;	//PUSHER DRIVE STATUS WORD BIT 15 - DRIVE SPECIFIC - PROFOBUS
   JS_SPD_REF_DI_PF : DINT ;	//JOY STICK SPEED REFERENCE IN DOUBLE INTEGER
   JS_SPD_REF_REAL_PF : REAL ;	//JOY STICK SPEED REFERENCE IN REAL(FLOATING POINT)
   JS_SPD_REF_UN_SL_FLT_PF : WORD ;	//JOY STICK SPEED REFERENCE UNSCALLING FAULT
   DRV_SPD_REF_VAL_PF : INT ;	//PUSHER DRIVE SPEED REFERENCE VALUE
   DRV_ACT_SPD_PF : REAL ;	//PUSHER DRIVE ACTUAL SPEED - PROFIBUS
   DRV_ACT_SPD_SCL_ERR : WORD ;	//PUSHER DRIVE ACTUAL SPEED SCALING ERROR - PROFIBUS
   PUSH_DRV_FWD_CMD_PF : BOOL ;	//PUSHER DRIVE FORWARD COMMAND OVER PROFIBUS
   PUSH_DRV_REV_CMD_PF : BOOL ;	//PUSHER DRIVE REVERSE COMMAND OVER PROFIBUS
   PUSH_FWD_CHNG_OVR_DEL : BOOL ;	//PUSHER DRIVE FORWARD CHANGE OVER DELAY
   PUSH_REV_CHNG_OVR_DEL : BOOL ;	//PUSHER DRIVE REVERSE CHANGE OVER DELAY
   PUSH_RAM_AUTO_FWD_STOP : BOOL ;	//PUSHER DRIVE AUTO FORWARD STOP
   PUSH_RAM_AUTO_RET_STOP : BOOL ;	//PUSHER DRIVE AUTO RETRACT STOP
   PULSE_5 : BOOL ;	//PULSE 5
   PULSE_6 : BOOL ;	//PULSE 6
   PULSE_7 : BOOL ;	//PULSE 7
   PULSE_8 : BOOL ;	//PULSE 8
   PULSE_9 : BOOL ;	//PULSE 9
   PULSE_10 : BOOL ;	//PULSE 10
   PULSE_11 : BOOL ;	//PULSE 11
   PULSE_12 : BOOL ;	//PULSE 12
   PUSH_AUTO_FWD_OVR : BOOL ;	//PUSHER AUTO FORWARD OVER
   PUSH_RAM_HOOT : BOOL ;	//PUSHER RAM HOOTER
  END_STRUCT ;	
BEGIN
   PUSH_FWD_REV_COUNT_SET := 3;
END_DATA_BLOCK

DATA_BLOCK "LEVEL_RAM_DB"	// DB 5
AUTHOR : Kamillas
VERSION : 0.1
  STRUCT
   LEV_BRK_RDY_FOR_STA : BOOL ;	//LEVELER BRAKE READY FOR START
   LEV_BRK_ON_FB : BOOL ;	//MOTOR BRAKE ON FEED BACK
   LEV_STP_PB : BOOL ;	//LEVELER STOP PUSH BUTTON
   LEV_MANUAL_SS : BOOL ;	//MANUAL SELECTOR SWITCH
   LEV_AUTO_SS : BOOL ;	//AUTOMATIC SELECTOR SWITCH
   JS_HME_POS : BOOL ;	//JOYSTICK HOME POSITION
   JS_FWD_POS : BOOL ;	//JOYSTICK FORWARD POSITION
   JS_REV_POS : BOOL ;	//JOYSTICK REVERSE POSITION
   JS_DEAD_MAN_BUTTON : BOOL ;	//JOYSTICK DEAD MAN BUTTON
   LEV_DRV_PROF_HARD_SEL : BOOL ;	//LEVELER DRIVE PROFIBUS / HARD WIRE CONNECTION
   LEV_DRV_ON_FB : BOOL ;	//LEVELER DRIVE ON FEED BACK
   LEV_DRV_RDY_FOR_STA : BOOL ;	//LEVELER DRIVE READY FOR START
   LEV_DRV_TRP_FB : BOOL ;	//LEVELER DRIVE TRIP FEED BACK
   LEV_RLS_OVN_FAC_RCHD : BOOL ;	//LEVELER RLS OVEN FACE REACHED
   LEV_RLS_FWD_END : BOOL ;	//LEVELER RLS FORWARD END
   LEV_RLS_REV_STK_FB : BOOL ;	//LEVELER RLS REVERSE STROKE FEED BACK
   LEV_RLS_REV_END : BOOL ;	//LEVELER RLS REVERSE END
   EMG_PB_LCS_16 : BOOL ;	//EMERGENCY PUSH BUTTON LCS 16
   LEV_EM_DRV_ENG_LCS : BOOL ;	//LEVELER EMERGENCY DRIVE ENGAGE LCS
   LEV_EM_DRV_DIS_ENG_LCS : BOOL ;	//LEVELER EMERGENCY DRIVE DISENGAGE LCS
   LEV_EM_DRV_DIS_ENG : BOOL ;	//LEVELER EMERGENCY DRIVE DISENGAGE
   LEV_END_FWD_LS : BOOL ;	//LEVELER END FORWARD LIMIT SWITCH
   LEV_END_RET_LS : BOOL ;	//LEVELER END RETRACT LIMIT SWITCH
   LEV_RAM_BRK_ON_CMD : BOOL ;	//LEVELER RAM BRAKE ON COMMAND
   PREP_FOR_LEV_IND : BOOL ;	//PREPARE FOR LEVELING INDICATION
   LEV_DRV_FWD_CMD : BOOL ;	//LEVELER DRIVE FORWARD COMMAND
   LEV_DRV_REV_CMD : BOOL ;	//LEVELER DRIVE REVERSE COMMAND
   LEV_DRV_ENG_IND : BOOL ;	//LEVELER DRIVE ENGAGE INDICATION
   LEV_RAM_ILK_1 : BOOL ;	//LEVELER RAM INTERLOCK BIT 1
   LEV_RAM_ILK : BOOL ;	//LEVELER RAM INTERLOCK BIT
   JS_SPD_REF_DI : DINT ;	//JOY STICK SPEED REFERENCE IN DOUBLE INTEGER
   JS_SPD_REF_NEG_RMD : INT ;	//JOY STICK SPEED REFERENCE CONVERTERD TO POSITIVE VALUE
   JS_SPD_REF_REAL : REAL ;	//JOY STICK SPEED REFERENCE IN REAL(FLOATING POINT)
   JS_SPD_REF_UN_SL_FLT : WORD ;	//JOY STICK SPEED REFERENCE UNSCALLING FAULT
   LEV_SPD_REF_VAL : INT ;	//LEVELER SPEED REFERENCE VALUE
   LEV_DRV_BRK_FLT : BOOL ;	//LEVELER DRIVE BREAK FAULT
   LEV_DRV_BRK_FLT_TMR : INT ;	//LEVELER DRIVE BREAK FAULT TIMER
   LEV_ILK_BYPASS : BOOL ;	//LEVELER RAM INTERLOCK BYPASS INPUT
   LEV_RAM_REV_END_IND : BOOL ;	//LEVELER RAM REVERSE END INDICATOR
   LEV_PERM_IND : BOOL ;	//LEVELER PERMISION INDICATION
   LEV_DRV_STATUS_WORD_1 : INT ;	//LEVELER PROFIBUS STATUS WORD 1
   LEV_DRV_STATUS_WORD_2 : INT ;	//LEVELER PROFIBUS STATUS WORD 2
   LEV_DRV_STATUS_WORD_3 : INT ;	//LEVELER PROFIBUS STATUS WORD 3
   LEV_DRV_STATUS_WORD_4 : INT ;	//LEVELER PROFIBUS STATUS WORD 4
   LEV_DRV_CONTROL_WORD_1 : INT ;	//LEVELER PROFIBUS CONTROL WORD 1
   LEV_DRV_CONTROL_WORD_2 : INT ;	//LEVELER PROFIBUS CONTROL WORD 2
   LEV_DRV_CONTROL_WORD_3 : INT ;	//LEVELER PROFIBUS CONTROL WORD 3
   LEV_DRV_CONTROL_WORD_4 : INT ;	//LEVELER PROFIBUS CONTROL WORD 4
   LEV_DRV_STAT_WORD_1_ERR : INT ;	//LEVELER DRIVE STATUS WORD 1 READ ERROR
   LEV_DRV_STAT_WORD_2_ERR : INT ;	//LEVELER DRIVE STATUS WORD 2 READ ERROR
   LEV_DRV_STAT_WORD_3_ERR : INT ;	//LEVELER DRIVE STATUS WORD 3 READ ERROR
   LEV_DRV_STAT_WORD_4_ERR : INT ;	//LEVELER DRIVE STATUS WORD 4 READ ERROR
   LEV_DRV_CTRL_WORD_1_ERR : INT ;	//LEVELER DRIVE CONTROL WORD 1 WRITE ERROR
   LEV_DRV_CTRL_WORD_2_ERR : INT ;	//LEVELER DRIVE CONTROL WORD 2 WRITE ERROR
   LEV_DRV_CTRL_WORD_3_ERR : INT ;	//LEVELER DRIVE CONTROL WORD 3 WRITE ERROR
   LEV_DRV_CTRL_WORD_4_ERR : INT ;	//LEVELER DRIVE CONTROL WORD 4 WRITE ERROR
   LEV_FWD_REV_COUNT : INT ;	//LEVELER FORWARD REVERSE COUNT
   LEV_FWD_REV_COUNT_SET : INT ;	//LEVELER FORWARD REVERSE COUNT SET POINT
   LEV_AUTO_CNT_RCHD : BOOL ;	//LEVELER AUTO COUNT REACHED
   LEV_FST_TIM_FWD_END_RCHD : BOOL ;	//LEVELER REACHED THE FORWARD END FOR FIRST TIME
   LEV_AUTO_STA_PB : BOOL ;	//LEVELER AUTO START PUSH BUTTON
   LEV_AUTO_STP_RET_PB : BOOL ;	//LEVELER AUTO STOP AND RETRACT PUSH BUTTON
   LEV_AUTO_STA : BOOL ;	//LEVELER AUTO START
   LEV_AUTO_STP_RET : BOOL ;	//LEVELER AUTO STOP AND RETRACT
   PULSE_1 : BOOL ;	//PULSE 1
   PULSE_2 : BOOL ;	//PULSE 2
   PULSE_3 : BOOL ;	//PULSE 3
   PULSE_4 : BOOL ;	//PULSE 4
   STA_LEV_IND : BOOL ;	//START LEVELING INDIACTION IN AUTO MODE
   LEV_MAN_STOP : BOOL ;	//LEVELER MANUAL STOP
   PULSE_5 : BOOL ;	//PULSE 5
   PULSE_6 : BOOL ;	//PULSE 6
   PULSE_7 : BOOL ;	//PULSE 7
   PULSE_8 : BOOL ;	//PULSE 8
   LEV_MAN_STP_PB : BOOL ;	//LEVELER MANUAL STOP PUSH BUTTON
   LEV_SPD_REF_VAL_FRM_JS : INT ;	//LEVELER SPEED REFERENCE VALUW FROM JOYSTICK
   LEV_DRV_STATUS_WORD_5 : INT ;	//LEVELER PROFIBUS STATUS WORD 5
   LEV_DRV_STATUS_WORD_6 : INT ;	//LEVELER PROFIBUS STATUS WORD 6
   LEV_DRV_STATUS_WORD_7 : INT ;	//LEVELER PROFIBUS STATUS WORD 7
   LEV_DRV_STATUS_WORD_8 : INT ;	//LEVELER PROFIBUS STATUS WORD 8
   LEV_DRV_STATUS_WORD_9 : INT ;	//LEVELER PROFIBUS STATUS WORD 9
   LEV_DRV_STATUS_WORD_10 : INT ;	//LEVELER PROFIBUS STATUS WORD 10
   LEV_DRV_STATUS_WORD_11 : INT ;	//LEVELER PROFIBUS STATUS WORD 11
   LEV_DRV_STATUS_WORD_12 : INT ;	//LEVELER PROFIBUS STATUS WORD 12
   LEV_DRV_STATUS_WORD_13 : INT ;	//LEVELER PROFIBUS STATUS WORD 13
   LEV_DRV_STATUS_WORD_14 : INT ;	//LEVELER PROFIBUS STATUS WORD 14
   LEV_DRV_CONTROL_WORD_5 : INT ;	//LEVELER PROFIBUS CONTROL WORD 5
   LEV_DRV_CONTROL_WORD_6 : INT ;	//LEVELER PROFIBUS CONTROL WORD 6
   LEV_DRV_CONTROL_WORD_7 : INT ;	//LEVELER PROFIBUS CONTROL WORD 7
   LEV_DRV_CONTROL_WORD_8 : INT ;	//LEVELER PROFIBUS CONTROL WORD 8
   LEV_DRV_CONTROL_WORD_9 : INT ;	//LEVELER PROFIBUS CONTROL WORD 9
   LEV_DRV_CONTROL_WORD_10 : INT ;	//LEVELER PROFIBUS CONTROL WORD 10
   LEV_DRV_CONTROL_WORD_11 : INT ;	//LEVELER PROFIBUS CONTROL WORD 11
   LEV_DRV_CONTROL_WORD_12 : INT ;	//LEVELER PROFIBUS CONTROL WORD 12
   LEV_DRV_CONTROL_WORD_13 : INT ;	//LEVELER PROFIBUS CONTROL WORD 13
   LEV_DRV_CONTROL_WORD_14 : INT ;	//LEVELER PROFIBUS CONTROL WORD 14
   LEV_TRA_DIST : REAL ;	//LEVELER TRAVELED DISTANCE
   LEV_ENC_VAL : INT ;	//LEVELER ENCODER VALUE THROUGH PROFIBUS
   LEV_ENC_VAL_DI : DINT ;	//LEVELER ENCODER VALUE IN DOUBLE INT FORMAR
   LEV_ENC_VAL_REAL : REAL ;	//LEVELER ENCODER VALUE IN REAL FORMAT
   LEV_ENC_NO_OF_REV : REAL ;	//LEVELER ENCODER NO OF REVOLUTIONS
   LEV_ENC_VAL_RST : BOOL ;	//LEVELER ENCODER VALUE RESET
   DRV_STATUS_WORD_1 : INT ;	//LEVELER DRIVE PROFIBUS STATUS WORD 1
   DRV_STATUS_WORD_2 : INT ;	//LEVELER DRIVE PROFIBUS STATUS WORD 2
   DRV_STATUS_WORD_3 : INT ;	//LEVELER DRIVE PROFIBUS STATUS WORD 3
   DRV_STATUS_WORD_4 : INT ;	//LEVELER DRIVE PROFIBUS STATUS WORD 4 (Fault WORD 1)
   DRV_STATUS_WORD_5 : INT ;	//LEVELER DRIVE PROFIBUS STATUS WORD 5 (Fault WORD 2)
   DRV_STATUS_WORD_6 : INT ;	//LEVELER DRIVE PROFIBUS STATUS WORD 6 (Fault WORD 4)
   DRV_STATUS_WORD_7 : INT ;	//LEVELER DRIVE PROFIBUS STATUS WORD 7 (LAST FAULT)
   DRV_STATUS_WORD_8 : INT ;	//LEVELER DRIVE PROFIBUS STATUS WORD 8
   DRV_STATUS_WORD_9 : INT ;	//LEVELER DRIVE PROFIBUS STATUS WORD 9
   DRV_STATUS_WORD_10 : INT ;	//LEVELER DRIVE PROFIBUS STATUS WORD 10
   DRV_STATUS_WORD_11 : INT ;	//LEVELER DRIVE PROFIBUS STATUS WORD 11
   DRV_STATUS_WORD_12 : INT ;	//LEVELER DRIVE PROFIBUS STATUS WORD 12
   DRV_STATUS_WORD_13 : INT ;	//LEVELER DRIVE PROFIBUS STATUS WORD 13
   DRV_STATUS_WORD_14 : INT ;	//LEVELER DRIVE PROFIBUS STATUS WORD 14
   DRV_STATUS_WORD_15 : INT ;	//LEVELER DRIVE PROFIBUS STATUS WORD 15
   DRV_STATUS_WORD_16 : INT ;	//LEVELER DRIVE PROFIBUS STATUS WORD 16
   DRV_CONTROL_WORD_1 : INT ;	//LEVELER DRIVE PROFIBUS CONTROL WORD 1
   DRV_CONTROL_WORD_2 : INT ;	//LEVELER DRIVE PROFIBUS CONTROL WORD 2
   DRV_CONTROL_WORD_3 : INT ;	//LEVELER DRIVE PROFIBUS CONTROL WORD 3
   DRV_CONTROL_WORD_4 : INT ;	//LEVELER DRIVE PROFIBUS CONTROL WORD 4
   DRV_CONTROL_WORD_5 : INT ;	//LEVELER DRIVE PROFIBUS CONTROL WORD 5
   DRV_CONTROL_WORD_6 : INT ;	//LEVELER DRIVE PROFIBUS CONTROL WORD 6
   DRV_CONTROL_WORD_7 : INT ;	//LEVELER DRIVE PROFIBUS CONTROL WORD 7
   DRV_CONTROL_WORD_8 : INT ;	//LEVELER DRIVE PROFIBUS CONTROL WORD 8
   DRV_CONTROL_WORD_9 : INT ;	//LEVELER DRIVE PROFIBUS CONTROL WORD 9
   DRV_CONTROL_WORD_10 : INT ;	//LEVELER DRIVE PROFIBUS CONTROL WORD 10
   DRV_CONTROL_WORD_11 : INT ;	//LEVELER DRIVE PROFIBUS CONTROL WORD 11
   DRV_CONTROL_WORD_12 : INT ;	//LEVELER DRIVE PROFIBUS CONTROL WORD 12
   DRV_CONTROL_WORD_13 : INT ;	//LEVELER DRIVE PROFIBUS CONTROL WORD 13
   DRV_CONTROL_WORD_14 : INT ;	//LEVELER DRIVE PROFIBUS CONTROL WORD 14
   DRV_CONTROL_WORD_15 : INT ;	//LEVELER DRIVE PROFIBUS CONTROL WORD 15
   DRV_CONTROL_WORD_16 : INT ;	//LEVELER DRIVE PROFIBUS CONTROL WORD 16
   DRV_STAT_WORD_1_ER : INT ;	//LEVELER DRIVE DRIVE STATUS WORD 1 READ ERROR
   DRV_STAT_WORD_2_ER : INT ;	//LEVELER DRIVE DRIVE STATUS WORD 2 READ ERROR
   DRV_STAT_WORD_3_ER : INT ;	//LEVELER DRIVE DRIVE STATUS WORD 3 READ ERROR
   DRV_STAT_WORD_4_ER : INT ;	//LEVELER DRIVE DRIVE STATUS WORD 4 READ ERROR
   DRV_CTRL_WORD_1_ER : INT ;	//LEVELER DRIVE DRIVE CONTROL WORD 1 WRITE ERROR
   DRV_CTRL_WORD_2_ER : INT ;	//LEVELER DRIVE DRIVE CONTROL WORD 2 WRITE ERROR
   DRV_CTRL_WORD_3_ER : INT ;	//LEVELER DRIVE DRIVE CONTROL WORD 3 WRITE ERROR
   DRV_CTRL_WORD_4_ER : INT ;	//LEVELER DRIVE DRIVE CONTROL WORD 4 WRITE ERROR
   DRV_CW_B0_RDY_TO_OPER : BOOL ;	//LEVELER DRIVE CONTROL WORD BIT 0 - READY TO OPERATE - OFF1 - PROFIBUS
   DRV_CW_B1_OFF_2 : BOOL ;	//LEVELER DRIVE CONTROL WORD BIT 1 - OFF2 - PROFIBUS
   DRV_CW_B2_OFF_3 : BOOL ;	//LEVELER DRIVE CONTROL WORD BIT 2 - OFF3 - PROFIBUS
   DRV_CW_B3_OPER_ENAB : BOOL ;	//LEVELER DRIVE CONTROL WORD BIT 3 - OPERATION ENABLE - PROFIBUS
   DRV_CW_B4_RMP_OUT_ZERO : BOOL ;	//LEVELER DRIVE CONTROL WORD BIT 4 - RAMP OUT ZERO - PROFIBUS
   DRV_CW_B5_RMP_HLD : BOOL ;	//LEVELER DRIVE CONTROL WORD BIT 5 - RAMP HOLD - PROFIBUS
   DRV_CW_B6_RMP_IN_ZERO : BOOL ;	//LEVELER DRIVE CONTROL WORD BIT 6 - RAMP IN ZERO - PROFIBUS
   DRV_CW_B7_FLT_RST : BOOL ;	//LEVELER DRIVE CONTROL WORD BIT 7 - FAULT RESET - PROFIBUS
   DRV_CW_B8_INCH_1 : BOOL ;	//LEVELER DRIVE CONTROL WORD BIT 8 - INCHING 1 - PROFIBUS
   DRV_CW_B9_INCH_2 : BOOL ;	//LEVELER DRIVE CONTROL WORD BIT 9 - INCHING 2 - PROFIBUS
   DRV_CW_B10_RMT_CMD : BOOL ;	//LEVELER DRIVE CONTROL WORD BIT 10 - REMOTE COMMAND - PROFIBUS
   DRV_CW_B11 : BOOL ;	//LEVELER DRIVE CONTROL WORD BIT 11 - DRIVE SPECIFIC - PROFOBUS
   DRV_CW_B12 : BOOL ;	//LEVELER DRIVE CONTROL WORD BIT 12 - DRIVE SPECIFIC - PROFOBUS
   DRV_CW_B13 : BOOL ;	//LEVELER DRIVE CONTROL WORD BIT 13 - DRIVE SPECIFIC - PROFOBUS
   DRV_CW_B14 : BOOL ;	//LEVELER DRIVE CONTROL WORD BIT 14 - DRIVE SPECIFIC - PROFOBUS
   DRV_CW_B15 : BOOL ;	//LEVELER DRIVE CONTROL WORD BIT 15 - DRIVE SPECIFIC - PROFOBUS
   DRV_SW_B0_RDY_ON : BOOL ;	//LEVELER DRIVE STATUS WORD BIT 0 - READY TO OPERATE - OFF1 - PROFIBUS
   DRV_SW_B1_RDY_TO_OPER : BOOL ;	//LEVELER DRIVE STATUS WORD BIT 1 - REDY TO OPERATE - PROFIBUS
   DRV_SW_B2_REF_RDY : BOOL ;	//LEVELER DRIVE STATUS WORD BIT 2 - ENABEL OPERATION - PROFIBUS
   DRV_SW_B3_TRIPPED : BOOL ;	//LEVELER DRIVE STATUS WORD BIT 3 - FAULT - PROFIBUS
   DRV_SW_B4_OFF_2_STA : BOOL ;	//LEVELER DRIVE STATUS WORD BIT 4 - OFF 2 STATUS - PROFIBUS
   DRV_SW_B5_OFF_3_STA : BOOL ;	//LEVELER DRIVE STATUS WORD BIT 5 - OFF 3 STATUS - PROFIBUS
   DRV_SW_B6_SWC_ON_INHB : BOOL ;	//LEVELER DRIVE STATUS WORD BIT 6 - SWITCH ON INHIBIT - PROFIBUS
   DRV_SW_B7_ALARM : BOOL ;	//LEVELER DRIVE STATUS WORD BIT 7 - WARNING/ALARM - PROFIBUS
   DRV_SW_B8_AT_SETPOINT : BOOL ;	//LEVELER DRIVE STATUS WORD BIT 8 - OPERATING - PROFIBUS
   DRV_SW_B9_REMOTE : BOOL ;	//LEVELER DRIVE STATUS WORD BIT 9 - DRIVE CONTROL REMOTE\LOCAL - PROFIBUS
   DRV_SW_B10_ABOVE_LIMIT : BOOL ;	//LEVELER DRIVE STATUS WORD BIT 10 - SPEED ABOVE LIMIT - PROFIBUS
   DRV_SW_B11 : BOOL ;	//LEVELER DRIVE STATUS WORD BIT 11 - DRIVE SPECIFIC - PROFOBUS
   DRV_SW_B12 : BOOL ;	//LEVELER DRIVE STATUS WORD BIT 12 - DRIVE SPECIFIC - PROFOBUS
   DRV_SW_B13 : BOOL ;	//LEVELER DRIVE STATUS WORD BIT 13 - DRIVE SPECIFIC - PROFOBUS
   DRV_SW_B14 : BOOL ;	//LEVELER DRIVE STATUS WORD BIT 14 - DRIVE SPECIFIC - PROFOBUS
   DRV_SW_B15 : BOOL ;	//LEVELER DRIVE STATUS WORD BIT 15 - DRIVE SPECIFIC - PROFOBUS
   JS_SPD_REF_DI_PF : DINT ;	//JOY STICK SPEED REFERENCE IN DOUBLE INTEGER
   JS_SPD_REF_REAL_PF : REAL ;	//JOY STICK SPEED REFERENCE IN REAL(FLOATING POINT)
   JS_SPD_REF_UN_SL_FLT_PF : WORD ;	//JOY STICK SPEED REFERENCE UNSCALLING FAULT
   DRV_SPD_REF_VAL_PF : INT ;	//LEVELER DRIVE SPEED REFERENCE VALUE
   DRV_ACT_SPD_PF : REAL ;	//LEVELER DRIVE ACTUAL SPEED - PROFIBUS
   DRV_ACT_SPD_SCL_ERR : WORD ;	//LEVELER DRIVE ACTUAL SPEED SCALING ERROR - PROFIBUS
   LEV_DRV_FWD_CMD_PF : BOOL ;	//LEVELER DRIVE FORWARD COMMAND OVER PROFIBUS
   LEV_DRV_REV_CMD_PF : BOOL ;	//LEVELER DRIVE REVERSE COMMAND OVER PROFIBUS
   LEV_FWD_CHNG_OVR_DEL : BOOL ;	//LEVELER DRIVE FORWARD CHANGE OVER DELAY
   LEV_REV_CHNG_OVR_DEL : BOOL ;	//LEVELER DRIVE REVERSE CHANGE OVER DELAY
  END_STRUCT ;	
BEGIN
   LEV_FWD_REV_COUNT_SET := 4;
END_DATA_BLOCK

DATA_BLOCK "AIR_COMPRESSOR_DB"	// DB 6
AUTHOR : Kamillas
VERSION : 0.1
  STRUCT
   MRT_1_RDY_FOR_STA : BOOL ;	//MOTOR 1 READY FOR START
   MTR_1_RUN_FB : BOOL ;	//MOTOR 1 RUN FEEDBACK
   MTR_1_OLR_TRP : BOOL ;	//MOTOR 1 OVER LOAD TRIP
   MRT_2_RDY_FOR_STA : BOOL ;	//MOTOR 2 READY FOR START
   MTR_2_RUN_FB : BOOL ;	//MOTOR 2 RUN FEEDBACK
   MTR_2_OLR_TRP : BOOL ;	//MOTOR 2 OVER LOAD TRIP
   CD_LCS_SS : BOOL ;	//CONTROL DESK/LOCAL CONTROL SELECTOR SWITCH
   MTR_1_2_SS : BOOL ;	//MOTOR 1/2 SELECTION
   MTR_1_STA_PB : BOOL ;	//MOTOR 1 START PUSH BUTTON
   MTR_1_STP_PB : BOOL ;	//MOTOR 1 STOP PUSH BUTTON
   MTR_2_STA_PB : BOOL ;	//MOTOR 2 START PUSH BUTTON
   MTR_2_STP_PB : BOOL ;	//MOTOR 2 STOP PUSH BUTTON
   MTR_1_2_SS_LCS : BOOL ;	//MOTOR 1/2 SELECTION LCS
   MTR_1_STA_PB_LCS : BOOL ;	//MOTOR 1 START PUSH BUTTON LCS
   MTR_1_STP_PB_LCS : BOOL ;	//MOTOR 1 STOP PUSH BUTTON LCS
   MTR_2_STA_PB_LCS : BOOL ;	//MOTOR 2 START PUSH BUTTON LCS
   MTR_2_STP_PB_LCS : BOOL ;	//MOTOR 2 STOP PUSH BUTTON LCS
   LCS_24_EMERGENCY_STOP_PB : BOOL ;	//LCS-24 EMERGENCY STOP PUSH BUTTON
   PRESSURE_SW_FB : BOOL ;	//PRESSURE SWITCH FEEDBACK
   MTR_1_ON_CMD : BOOL ;	//MOTOR 1 ON COMMAND
   MTR_2_ON_CMD : BOOL ;	//MOTOR 2 ON COMMAND
   MTR_1_ON_IND : BOOL ;	//MOTOR 1 ON INDICATOR
   MTR_2_ON_IND : BOOL ;	//MOTOR 2 ON INDICATOR
   MTR_1_ON_IND_LCS : BOOL ;	//MOTOR 1 ON INDICATOR LCS
   MTR_2_ON_IND_LCS : BOOL ;	//MOTOR 2 ON INDICATOR LCS
   LCS_24_ON_IND_LCS : BOOL ;	//LCS-24 ON INDICATOR LCS
   MTR_1_FLT : BOOL ;	//AIR COMPRESEOR MOTOR 1 FAULT
   MTR_1_FLT_TMR : INT ;	//AIR COMPRESEOR MOTOR 1 FAULT TIMER
   MTR_1_FLT_GEN_TIME : INT  := 3;	//AIR COMPRESEOR MOTOR 1 FAULT GEMERATION TIME
   MTR_2_FLT : BOOL ;	//AIR COMPRESEOR MOTOR 2 FAULT
   MTR_2_FLT_TMR : INT ;	//AIR COMPRESEOR MOTOR 2 FAULT TIMER
   MTR_2_FLT_GEN_TIME : INT  := 3;	//AIR COMPRESEOR MOTOR 2 FAULT GEMERATION TIME
   PULSE_1 : BOOL ;	//PULSE 1
   PULSE_2 : BOOL ;	//PULSE 2
   PULSE_3 : BOOL ;	//PULSE 3
   PULSE_4 : BOOL ;	//PULSE 4
   PULSE_5 : BOOL ;	//PULSE 5
   PULSE_6 : BOOL ;	//PULSE 6
   PULSE_7 : BOOL ;	//PULSE 7
   PULSE_8 : BOOL ;	//PULSE 8
   MTR_1_ON_CMD_BIT : BOOL ;	//AIR COMPRESSOR MOTOR 1 ON COMMAND WITHOUT PRESSURE SWITCH INTERLOCK
   MTR_2_ON_CMD_BIT : BOOL ;	//AIR COMPRESSOR MOTOR 2 ON COMMAND WITHOUT PRESSURE SWITCH INTERLOCK
  END_STRUCT ;	
BEGIN
   MTR_1_FLT_GEN_TIME := 3;
   MTR_2_FLT_GEN_TIME := 3;
END_DATA_BLOCK

DATA_BLOCK "DOOR_AND_JAMB_DB"	// DB 7
AUTHOR : Kamillas
VERSION : 0.1
  STRUCT
   VIB_DOR_CLNR_RDY_FOR_STA : BOOL ;	//VIBRATOR - DOOR CLEANER READY FOR START
   VIB_DOR_CLNR_RUN_FB : BOOL ;	//VIBRATOR - DOOR CLEANER RUN FEEDBACK
   VIB_DOR_CLNR_OLR_TRP : BOOL ;	//VIBRATOR - DOOR CLEANER OVERLOAD TRIP
   VIB_JMB_CLNR_RDY_FOR_STA : BOOL ;	//VIBRATOR - JAMB CLEANER READY FOR START
   VIB_JMB_CLNR_RUN_FB : BOOL ;	//VIBRATOR - JAMB CLEANER RUN FEEDBACK
   VIB_JMB_CLNR_OLR_TRP : BOOL ;	//VIBRATOR - JAMB CLEANER OVERLOAD TRIP
   VIB_DOR_CLNR_STA_PB : BOOL ;	//VIBRATOR - DOOR CLEANER START PUSH BUTTON
   VIB_DOR_CLNR_STP_PB : BOOL ;	//VIBRATOR - DOOR CLEANER STOP PUSH BUTTON
   VIB_JMB_CLNR_STA_PB : BOOL ;	//VIBRATOR - JAMB CLEANER START PUSH BUTTON
   VIB_JMB_CLNR_STP_PB : BOOL ;	//VIBRATOR - JAMB CLEANER STOP PUSH BUTTON
   VIB_DOR_CLNR_STA_PB_LCS : BOOL ;	//VIBRATOR - DOOR CLEANER START PUSH BUTTON LCS
   VIB_DOR_CLNR_STP_PB_LCS : BOOL ;	//VIBRATOR - DOOR CLEANER STOP PUSH BUTTON LCS
   VIB_JMB_CLNR_STA_PB_LCS : BOOL ;	//VIBRATOR - JAMB CLEANER START PUSH BUTTON LCS
   VIB_JMB_CLNR_STP_PB_LCS : BOOL ;	//VIBRATOR - JAMB CLEANER STOP PUSH BUTTON LCS
   VIB_DOR_CLNR_ON_CMD : BOOL ;	//VIBRATOR - DOOR CLEANER ON COMMAND
   VIB_JMB_CLNR_ON_CMD : BOOL ;	//VIBRATOR - JAMB CLEANER ON COMMAND
   VIB_DOR_CLNR_ON_IND : BOOL ;	//VIBRATOR - DOOR CLEANER ON INDICATOR
   VIB_JMB_CLNR_ON_IND : BOOL ;	//VIBRATOR - JAMB CLEANER ON INDICATOR
   VIB_DOR_CLNR_ON_IND_LCS : BOOL ;	//VIBRATOR - DOOR CLEANER ON INDICATOR LCS
   VIB_JMB_CLNR_ON_IND_LCS : BOOL ;	//VIBRATOR - JAMB CLEANER ON INDICATOR LCS
   PULSE_1 : BOOL ;	//PULSE 1
   PULSE_2 : BOOL ;	//PULSE 2
   PULSE_3 : BOOL ;	//PULSE 3
   PULSE_4 : BOOL ;	//PULSE 4
   PULSE_5 : BOOL ;	//PULSE 5
   PULSE_6 : BOOL ;	//PULSE 6
   PULSE_7 : BOOL ;	//PULSE 7
   PULSE_8 : BOOL ;	//PULSE 8
   VIB_DOR_CLNR_FLT : BOOL ;	//VIBRATOR - DOOR CLEANER FAULT
   VIB_DOR_CLNR_FLT_TMR : INT ;	//VIBRATOR - DOOR CLEANER FAULT TIMER
   VIB_DOR_CLN_FLT_GEN_TIME : INT  := 3;	//VIBRATOR - DOOR CLEANER FAULT GEMERATION TIME
   VIB_JMB_CLNR_FLT : BOOL ;	//VIBRATOR - JAMB CLEANER FAULT
   VIB_JMB_CLNR_FLT_TMR : INT ;	//VIBRATOR - JAMB CLEANER FAULT TIMER
   VIB_JMB_CLN_FLT_GEN_TIME : INT  := 3;	//VIBRATOR - JAMB CLEANER FAULT GEMERATION TIME
  END_STRUCT ;	
BEGIN
   VIB_DOR_CLN_FLT_GEN_TIME := 3;
   VIB_JMB_CLN_FLT_GEN_TIME := 3;
END_DATA_BLOCK

DATA_BLOCK "LEVELER_BLOWER_DB"	// DB 8
AUTHOR : Kamillas
VERSION : 0.1
  STRUCT
   LEV_BLOW_MTR_RDY_FOR_STA : BOOL ;	//LEVELER BLOWER READY FOR START
   LEV_BLOW_MTR_RUN_FB : BOOL ;	//LEVELER BLOWER RUNNING FEED BACK
   LEV_BLOW_MTR_OLR_TRP : BOOL ;	//LEVELER BLOWER TRIP FEED BACK
   LEV_BLOW_MTR_STA_PB : BOOL ;	//LEVELER BLOWER START PUSH BUTTON
   LEV_BLOW_MTR_STP_PB : BOOL ;	//LEVELER BLOWER STOP PUSH BUTTON
   LEV_BLOW_MTR_STA_PB_LCS : BOOL ;	//LEVELER BLOWER START PUSH BUTTON LCS
   LEV_BLOW_MTR_STP_PB_LCS : BOOL ;	//LEVELER BLOWER STOP PUSH BUTTON LCS
   LEV_BLOW_MTR_ON_CMD : BOOL ;	//LEVELER BLOWER MOTOR ON COMMAND
   LEV_BLOW_MTR_ON_IND : BOOL ;	//LEVELER BLOWER MOTOR ON INDICATOR
   LEV_BLOW_MTR_ON_IND_LCS : BOOL ;	//LEVELER BLOWER MOTOR ON INDICATOR
   LEV_BLOW_MTR_FLT : BOOL ;	//VIBRATOR - JAMB CLEANER FAULT
   LEV_BLOW_MTR_FLT_TMR : INT ;	//VIBRATOR - JAMB CLEANER FAULT TIMER
   LEV_BLO_MTR_FLT_GEN_TIME : INT  := 3;	//VIBRATOR - JAMB CLEANER FAULT GEMERATION TIME
   PULSE_1 : BOOL ;	//PULSE 1
   PULSE_2 : BOOL ;	//PULSE 2
   PULSE_3 : BOOL ;	//PULSE 3
   PULSE_4 : BOOL ;	//PULSE 4
   PULSE_5 : BOOL ;	//PULSE 5
   PULSE_6 : BOOL ;	//PULSE 6
   PULSE_7 : BOOL ;	//PULSE 7
   PULSE_8 : BOOL ;	//PULSE 8
  END_STRUCT ;	
BEGIN
   LEV_BLO_MTR_FLT_GEN_TIME := 3;
END_DATA_BLOCK

DATA_BLOCK "LIFTING_PLATFORM_DB"	// DB 9
AUTHOR : Kamillas
VERSION : 0.1
  STRUCT
   LIFT_PF_MRT_RDY_FOR_STA : BOOL ;	//LIFT PLATFORM READY FOR START
   LIFT_PF_MTR_UP_ON_FB : BOOL ;	//LIFT PLATFORM UP ON FEEDBCAK
   LIFT_PF_MTR_DN_ON_FB : BOOL ;	//LIFT PLATFORM DOWN ON FEEDBCAK
   LIFT_PF_MTR_OLR_TRP : BOOL ;	//LIFT MOTOR OVERLOAD TRIP
   LIFT_PF_MTR_UP_PB : BOOL ;	//LIFT PLATFORM UP PUSH BUTTON
   LIFT_PF_MTR_DN_PB : BOOL ;	//LIFT PLATFORM DOWN PUSH BUTTON
   EMERGENCY_PB_LCS_19 : BOOL ;	//LCS-19 EMERGENCY PUSH BUTTON
   LIFT_PF_MTR_UP_LS : BOOL ;	//LIFT PLATFORM UP LIMIT SWITCH
   LIFT_PF_MTR_DN_LS : BOOL ;	//LIFT PLATFORM DOWN LIMIT SWITCH
   LIFT_PF_MTR_UP_ON_CMD : BOOL ;	//LIFT PLATFORM UP ON COMMAND
   LIFT_PF_MTR_DN_ON_CMD : BOOL ;	//LIFT PLATFORM DOWN ON COMMAND
   LIFT_PF_MTR_FLT : BOOL ;	//LIFT PLATFORM FAULT
   LIFT_PF_MTR_FLT_TMR : INT ;	//LIFT PLATFORM CLEANER FAULT TIMER
   LIFT_PF_MTR_FLT_GEN_TIME : INT  := 3;	//LIFT PLATFORM CLEANER FAULT GEMERATION TIME
   PULSE_1 : BOOL ;	//PULSE 1
   PULSE_2 : BOOL ;	//PULSE 2
   PULSE_3 : BOOL ;	//PULSE 3
   PULSE_4 : BOOL ;	//PULSE 4
   PULSE_5 : BOOL ;	//PULSE 5
   PULSE_6 : BOOL ;	//PULSE 6
   PULSE_7 : BOOL ;	//PULSE 7
   PULSE_8 : BOOL ;	//PULSE 8
  END_STRUCT ;	
BEGIN
   LIFT_PF_MTR_FLT_GEN_TIME := 3;
END_DATA_BLOCK

DATA_BLOCK "LEVELER_DOOR_DB"	// DB 10
AUTHOR : Kamillas
VERSION : 0.1
  STRUCT
   LEV_DOOR_LOCAL_SS : BOOL ;	//LEVELER DOOR LOCAL SELECTOR SWITCH
   LEV_DOOR_MAN_SS : BOOL ;	//LEVELER DOOR MANUAL SELECTOR SWITCH
   LEV_DOOR_AUTO_SS : BOOL ;	//LEVELER DOOR AUTO SELECTOR SWITCH
   LEV_DOOR_STP_PB : BOOL ;	//LEVELER DOOR STOP PUSH BUTTON
   ACT_GRP_FWD_STA_PB : BOOL ;	//ACTUATING GRIP FORWARD START PUSH BUTTON
   ACT_GRP_RET_STA_PB : BOOL ;	//ACTUATING GRIP RETRACT START PUSH BUTTON
   SLW_RK_SP_1_FWD_STA : BOOL ;	//SLEAVING RACK STEP 1 FORWARD START PUSH BUTTON
   SLW_RK_SP_1_RET_STA : BOOL ;	//SLEAVING RACK STEP 1 RETRACT START PUSH BUTTON
   SLW_RK_SP_2_FWD_STA : BOOL ;	//SLEAVING RACK STEP 2 FORWARD START PUSH BUTTON
   SLW_RK_SP_2_RET_STA : BOOL ;	//SLEAVING RACK STEP 2 RETRACT START PUSH BUTTON
   LEV_WN_CLR_UP_STA_PB : BOOL ;	//LEVELER WINDOW FRAME CLEANER UP START PUSH BUTTON
   LEV_WN_CLR_DN_STA_PB : BOOL ;	//LEVELER WINDOW FRAME CLEANER DOWN START PUSH BUTTON
   SMK_SLVE_FWD_STA_PB : BOOL ;	//SMOKE SLEEVE FORWARD START PUSH BUTTON
   SMK_SLVE_RET_STA_PB : BOOL ;	//SMOKE SLEEVE RETRACT START PUSH BUTTON
   EMG_STOP_PB_LCS_61 : BOOL ;	//EMERGENCY STOP PUSH BUTTON LCS 61
   ACT_GRP_FWD_STA_PB_LCS : BOOL ;	//ACTUATING GRIP FORWARD START PUSH BUTTON LCS
   ACT_GRP_RET_STA_PB_LCS : BOOL ;	//ACTUATING GRIP RETRACT START PUSH BUTTON LCS
   SLW_RK_SP_1_FWD_STA_LCS : BOOL ;	//SLEAVING RACK STEP 1 FORWARD START PUSH BUTTON LCS
   SLW_RK_SP_1_RET_STA_LCS : BOOL ;	//SLEAVING RACK STEP 1 RETRACT START PUSH BUTTON LCS
   SLW_RK_SP_2_FWD_STA_LCS : BOOL ;	//SLEAVING RACK STEP 2 FORWARD START PUSH BUTTON LCS
   SLW_RK_SP_2_RET_STA_LCS : BOOL ;	//SLEAVING RACK STEP 2 RETRACT START PUSH BUTTON LCS
   LEV_WN_CLR_UP_STA_LCS : BOOL ;	//LEVELER WINDOW FRAME CLEANER UP START PUSH BUTTON LCS
   LEV_WN_CLR_DN_STA_LCS : BOOL ;	//LEVELER WINDOW FRAME CLEANER DOWN START PUSH BUTTON LCS
   SMK_SLVE_FWD_STA_PB_LCS : BOOL ;	//SMOKE SLEEVE FORWARD START PUSH BUTTON LCS
   SMK_SLVE_RET_STA_PB_LCS : BOOL ;	//SMOKE SLEEVE RETRACT START PUSH BUTTON LCS
   TEST_LAMP_PB_LCS_61 : BOOL ;	//TEST LAMP PUSH BUTTON LCS 61
   ACT_GRP_FWD_LS : BOOL ;	//ACTUATING GRIP FORWARD START LIMIT SWITCH
   ACT_GRP_RET_LS : BOOL ;	//ACTUATING GRIP RETRACT START LIMIT SWITCH
   SLW_RK_SP_1_FWD_LS : BOOL ;	//SLEAVING RACK STEP 1 FORWARD LIMIT SWITCH
   SLW_RK_SP_1_RET_LS : BOOL ;	//SLEAVING RACK STEP 1 RETRACT LIMIT SWITCH
   SLW_RK_SP_2_FWD_LS : BOOL ;	//SLEAVING RACK STEP 2 FORWARD LIMIT SWITCH
   SLW_RK_SP_2_RET_LS : BOOL ;	//SLEAVING RACK STEP 2 RETRACT LIMIT SWITCH
   LEV_WN_CLR_UP_LS : BOOL ;	//LEVELER WINDOW FRAME CLEANER UP LIMIT SWITCH
   LEV_WN_CLR_DN_LS : BOOL ;	//LEVELER WINDOW FRAME CLEANER DOWN LIMIT SWITCH
   SMK_SLVE_FWD_LS : BOOL ;	//SMOKE SLEEVE FORWARD LIMIT SWITCH
   SMK_SLVE_SLOW_FWD_LS : BOOL ;	//SMOKE SLEEVE SLOW FORWARD LIMIT SWITCH
   SMK_SLVE_REV_LS : BOOL ;	//SMOKE SLEEVE RETRACT LIMIT SWITCH
   ACT_GRP_FWD_CMD : BOOL ;	//ACTUATING GRIP FORWARD START COMMAND
   ACT_GRP_RET_CMD : BOOL ;	//ACTUATING GRIP RETRACT START COMMAND
   SLW_RK_SP_1_FWD_CMD : BOOL ;	//SLEAVING RACK STEP 1 FORWARD COMMAND
   SLW_RK_SP_1_RET_CMD : BOOL ;	//SLEAVING RACK STEP 1 RETRACT COMMAND
   SLW_RK_SP_2_FWD_CMD : BOOL ;	//SLEAVING RACK STEP 2 FORWARD COMMAND
   SLW_RK_SP_2_RET_CMD : BOOL ;	//SLEAVING RACK STEP 2 RETRACT COMMAND
   LEV_WN_CLR_UP_CMD : BOOL ;	//LEVELER WINDOW FRAME CLEANER UP COMMAND
   LEV_WN_CLR_DN_CMD : BOOL ;	//LEVELER WINDOW FRAME CLEANER DOWN COMMAND
   SMK_SLVE_SLOW_FWD_CMD : BOOL ;	//SMOKE SLEEVE SLOW FORWARD COMMAND
   SMK_SLVE_SLOW_REV_CMD : BOOL ;	//SMOKE SLEEVE SLOW RETRACT COMMAND
   SMK_SLVE_NORM_FWD_CMD : BOOL ;	//SMOKE SLEEVE NORMAL FORWARD COMMAND
   SMK_SLVE_NORM_REV_CMD : BOOL ;	//SMOKE SLEEVE NORMAL RETRACT COMMAND
   ACT_GRP_FWD_IND : BOOL ;	//ACTUATING GRIP FORWARD INDICATOR
   ACT_GRP_RET_IND : BOOL ;	//ACTUATING GRIP RETRACT INDICATOR
   SLW_RK_SP_1_FWD_IND : BOOL ;	//SLEAVING RACK STEP 1 FORWARD INDICATOR
   SLW_RK_SP_1_RET_IND : BOOL ;	//SLEAVING RACK STEP 1 RETRACT INDICATOR
   SLW_RK_SP_2_FWD_IND : BOOL ;	//SLEAVING RACK STEP 2 FORWARD INDICATOR
   SLW_RK_SP_2_RET_IND : BOOL ;	//SLEAVING RACK STEP 2 RETRACT INDICATOR
   LEV_WN_CLR_UP_IND : BOOL ;	//LEVELER WINDOW FRAME CLEANER UP INDICATOR
   LEV_WN_CLR_DN_IND : BOOL ;	//LEVELER WINDOW FRAME CLEANER DOWN INDICATOR
   SMK_SLVE_FWD_IND : BOOL ;	//SMOKE SLEEVE FORWARD INDICATOR
   SMK_SLVE_RET_IND : BOOL ;	//SMOKE SLEEVE RETRACT INDICATOR
   ACT_GRP_FWD_IND_LCS : BOOL ;	//ACTUATING GRIP FORWARD INDICATOR LCS
   ACT_GRP_RET_IND_LCS : BOOL ;	//ACTUATING GRIP RETRACT INDICATOR LCS
   SLW_RK_SP_1_FWD_IND_LCS : BOOL ;	//SLEAVING RACK STEP 1 FORWARD INDICATOR LCS
   SLW_RK_SP_1_RET_IND_LCS : BOOL ;	//SLEAVING RACK STEP 1 RETRACT INDICATOR LCS
   SLW_RK_SP_2_FWD_IND_LCS : BOOL ;	//SLEAVING RACK STEP 2 FORWARD INDICATOR LCS
   SLW_RK_SP_2_RET_IND_LCS : BOOL ;	//SLEAVING RACK STEP 2 RETRACT INDICATOR LCS
   LEV_WN_CLR_UP_IND_LCS : BOOL ;	//LEVELER WINDOW FRAME CLEANER UP INDICATOR LCS
   LEV_WN_CLR_DN_IND_LCS : BOOL ;	//LEVELER WINDOW FRAME CLEANER DOWN INDICATOR LCS
   SMK_SLVE_FWD_IND_LCS : BOOL ;	//SMOKE SLEEVE FORWARD INDICATOR LCS
   SMK_SLVE_RET_IND_LCS : BOOL ;	//SMOKE SLEEVE RETRACT INDICATOR LCS
   LCS_61_ON_INDICATOR : BOOL ;	//LCS 61 ON INDICATOR
   ACT_GRP_DOOR_ON_HOOK : BOOL ;	//ACTUATOR GRIP DOOR ON HOOK
   ACT_GRP_DOOR_ON_HOOK_LCS : BOOL ;	//ACTUATOR GRIP DOOR ON HOOK LCS
   PREP_LEV_ILK_BIT : BOOL ;	//PREPARE LEVELER INTERLOCK BIT
   PREP_LEV_AUTO_STA_BIT : BOOL ;	//PREPARE FOR LEVELING AUTO START BIT
   FIN_LEV_OPER_COMP_BIT : BOOL ;	//FINISH LEVELING OPERATION COMPLETED BIT
   PREP_LEV_OPER_COMP_BIT : BOOL ;	//PREPARE LEVELING OPERATION COMPLETED BIT
   PREP_LEV_RDY_BIT : BOOL ;	//PREPARE LEVELER READY BIT
   PREP_LEV_AUTO_STA_BIT1 : BOOL ;	//PREPARE LEVELER AUTO START BIT
   PREP_FOR_LEV_STA_PB : BOOL ;	//PREPARE FOR LEVELLING START PUSH BUTTON
   PREP_FOR_LEV_STP_PB : BOOL ;	//PREPARE FOR LEVELLING STOP PUSH BUTTON
   SLW_RK_SP_1_FWD_OPU_CUT : BOOL ;	//SLEWING RACK STEP 1 FORWARD OUTPUT CUT
   SLW_RK_SP_1_FWD_FLT_TMR : INT ;	//SLEWING RACK STEP 1 FORWARD FAULT TIMER
   SLW_RK_SP_1_FWD_FLT_GEN : INT  := 8;	//SLEWING RACK STEP 1 FORWARD FAULT GENERATION TIME
   SLW_RK_SP_1_FWD_OP_CT_TM : INT ;	//SLEWING RACK STEP 1 FORWARD OUTPUT CUT TIMER
   SLW_RK_SP_1_FWD_FLT : BOOL ;	//SLEWING RACK STEP 1 FORWARD FAULT
   SLW_RK_SP_1_AUTO_FWD_OVR : BOOL ;	//SLEWING RACK STEP 1 AUTO FORWARD OVER
   SLW_RK_SP_1_AUTO_FWD_DEL : INT  := 3;	//SLEWING RACK STEP 1 AUTO FORWARD OVER DELAY
   SLW_RK_SP_1_ATO_FWD_DL_T : INT ;	//SLEWING RACK STEP 1 AUTO FORWARD OVER DELAY TIMER
   PULSE_1 : BOOL ;	//PULSE 1
   PULSE_2 : BOOL ;	//PULSE 2
   PULSE_3 : BOOL ;	//PULSE 3
   PULSE_4 : BOOL ;	//PULSE 4
   PULSE_5 : BOOL ;	//PULSE 5
   PULSE_6 : BOOL ;	//PULSE 6
   PULSE_7 : BOOL ;	//PULSE 7
   PULSE_8 : BOOL ;	//PULSE 8
   PULSE_9 : BOOL ;	//PULSE 9
   PULSE_10 : BOOL ;	//PULSE 10
   PULSE_11 : BOOL ;	//PULSE 11
   PULSE_12 : BOOL ;	//PULSE 12
   PULSE_13 : BOOL ;	//PULSE 13
   PULSE_14 : BOOL ;	//PULSE 14
   PULSE_15 : BOOL ;	//PULSE 15
   PULSE_16 : BOOL ;	//PULSE 16
   SLW_RK_SP_2_FWD_OPU_CUT : BOOL ;	//SLEWING RACK STEP 2 FORWARD OUTPUT CUT
   SLW_RK_SP_2_FWD_FLT_TMR : INT ;	//SLEWING RACK STEP 2 FORWARD FAULT TIMER
   SLW_RK_SP_2_FWD_FLT_GEN : INT  := 8;	//SLEWING RACK STEP 2 FORWARD FAULT GENERATION TIME
   SLW_RK_SP_2_FWD_OP_CT_TM : INT ;	//SLEWING RACK STEP 2 FORWARD OUTPUT CUT TIMER
   SLW_RK_SP_2_FWD_FLT : BOOL ;	//SLEWING RACK STEP 2 FORWARD FAULT
   SLW_RK_SP_2_AUTO_FWD_OVR : BOOL ;	//SLEWING RACK STEP 2 AUTO FORWARD OVER
   SLW_RK_SP_2_AUTO_FWD_DEL : INT  := 3;	//SLEWING RACK STEP 2 AUTO FORWARD OVER DELAY
   SLW_RK_SP_2_ATO_FWD_DL_T : INT ;	//SLEWING RACK STEP 2 AUTO FORWARD OVER DELAY TIMER
   SLW_RK_SP_1_RET_OPU_CUT : BOOL ;	//SLEWING RACK STEP 1 RETRACT OUTPUT CUT
   SLW_RK_SP_1_RET_FLT_TMR : INT ;	//SLEWING RACK STEP 1 RETRACT FAULT TIMER
   SLW_RK_SP_1_RET_FLT_GEN : INT  := 8;	//SLEWING RACK STEP 1 RETRACT FAULT GENERATION TIME
   SLW_RK_SP_1_RET_OP_CT_TM : INT ;	//SLEWING RACK STEP 1 RETRACT OUTPUT CUT TIMER
   SLW_RK_SP_1_RET_FLT : BOOL ;	//SLEWING RACK STEP 1 RETRACT FAULT
   SLW_RK_SP_1_AUTO_RET_OVR : BOOL ;	//SLEWING RACK STEP 1 AUTO RETRACT OVER
   SLW_RK_SP_1_AUTO_RET_DEL : INT  := 3;	//SLEWING RACK STEP 1 AUTO RETRACT OVER DELAY
   SLW_RK_SP_1_ATO_RET_DL_T : INT ;	//SLEWING RACK STEP 1 AUTO RETRACT OVER DELAY TIMER
   SLW_RK_SP_2_RET_OPU_CUT : BOOL ;	//SLEWING RACK STEP 2 RETRACT OUTPUT CUT
   SLW_RK_SP_2_RET_FLT_TMR : INT ;	//SLEWING RACK STEP 2 RETRACT FAULT TIMER
   SLW_RK_SP_2_RET_FLT_GEN : INT  := 8;	//SLEWING RACK STEP 2 RETRACT FAULT GENERATION TIME
   SLW_RK_SP_2_RET_OP_CT_TM : INT ;	//SLEWING RACK STEP 2 RETRACT OUTPUT CUT TIMER
   SLW_RK_SP_2_RET_FLT : BOOL ;	//SLEWING RACK STEP 2 RETRACT FAULT
   SLW_RK_SP_2_AUTO_RET_OVR : BOOL ;	//SLEWING RACK STEP 2 AUTO RETRACT OVER
   SLW_RK_SP_2_AUTO_RET_DEL : INT  := 3;	//SLEWING RACK STEP 2 AUTO RETRACT OVER DELAY
   SLW_RK_SP_2_ATO_RET_DL_T : INT ;	//SLEWING RACK STEP 2 AUTO RETRACT OVER DELAY TIMER
   ACT_GRP_FWD_OP_CUT : BOOL ;	//ACTUAROT GRIPPER FORWARD OUTPUT CUT
   ACT_GRP_FWD_FLT_TMR : INT ;	//ACTUAROT GRIPPER FORWARD FAULT TIMER
   ACT_GRP_FWD_FLT_GEN : INT  := 8;	//ACTUAROT GRIPPER FORWARD FAULT GENERATION TIME
   ACT_GRP_FWD_OP_CT_TM : INT ;	//ACTUAROT GRIPPER FORWARD RETRACT OUTPUT CUT TIMER
   ACT_GRP_FWD_FLT : BOOL ;	//ACTUAROT GRIPPER FORWARD RETRACT FAULT
   ACT_GRP_AUTO_FWD_OVR : BOOL ;	//ACTUAROT GRIPPER FORWARD AUTO RETRACT OVER
   ACT_GRP_AUTO_FWD_DEL : INT  := 3;	//ACTUAROT GRIPPER FORWARD AUTO RETRACT OVER DELAY
   ACT_GRP_ATO_FWD_DL_T : INT ;	//ACTUAROT GRIPPER FORWARD AUTO RETRACT OVER DELAY TIMER
   ACT_GRP_RET_OP_CUT : BOOL ;	//ACTUAROT GRIPPER RETRACT OUTPUT CUT
   ACT_GRP_RET_FLT_TMR : INT ;	//ACTUAROT GRIPPER RETRACT FAULT TIMER
   ACT_GRP_RET_FLT_GEN : INT  := 8;	//ACTUAROT GRIPPER RETRACT FAULT GENERATION TIME
   ACT_GRP_RET_OP_CT_TM : INT ;	//ACTUAROT GRIPPER RETRACT RETRACT OUTPUT CUT TIMER
   ACT_GRP_RET_FLT : BOOL ;	//ACTUAROT GRIPPER RETRACT RETRACT FAULT
   ACT_GRP_AUTO_RET_OVR : BOOL ;	//ACTUAROT GRIPPER RETRACT AUTO RETRACT OVER
   ACT_GRP_AUTO_RET_DEL : INT  := 3;	//ACTUAROT GRIPPER RETRACT AUTO RETRACT OVER DELAY
   ACT_GRP_ATO_RET_DL_T : INT ;	//ACTUAROT GRIPPER RETRACT AUTO RETRACT OVER DELAY TIMER
   LEV_WN_CLR_UP_OP_CUT : BOOL ;	//LEVELER WINDOW FRAME CLEANER UP OUTPUT CUT
   LEV_WN_CLR_UP_FLT_TMR : INT ;	//LEVELER WINDOW FRAME CLEANER UP FAULT TIMER
   LEV_WN_CLR_UP_FLT_GEN : INT  := 8;	//LEVELER WINDOW FRAME CLEANER UP FAULT GENERATION TIME
   LEV_WN_CLR_UP_OP_CT_TM : INT ;	//LEVELER WINDOW FRAME CLEANER UP RETRACT OUTPUT CUT TIMER
   LEV_WN_CLR_UP_FLT : BOOL ;	//LEVELER WINDOW FRAME CLEANER UP RETRACT FAULT
   LEV_WN_CLR_AUTO_UP_OVR : BOOL ;	//LEVELER WINDOW FRAME CLEANER AUTO UP OVER
   LEV_WN_CLR_AUTO_UP_DEL : INT  := 3;	//LEVELER WINDOW FRAME CLEANER AUTO UP OVER DELAY
   LEV_WN_CLR_ATO_UP_DL_T : INT ;	//LEVELER WINDOW FRAME CLEANER AUTO UP OVER DELAY TIMER
   LEV_WN_CLR_DN_OP_CUT : BOOL ;	//LEVELER WINDOW FRAME CLEANER DOWN OUTPUT CUT
   LEV_WN_CLR_DN_FLT_TMR : INT ;	//LEVELER WINDOW FRAME CLEANER DOWN FAULT TIMER
   LEV_WN_CLR_DN_FLT_GEN : INT  := 8;	//LEVELER WINDOW FRAME CLEANER DOWN FAULT GENERATION TIME
   LEV_WN_CLR_DN_OP_CT_TM : INT ;	//LEVELER WINDOW FRAME CLEANER DOWN OUTPUT CUT TIMER
   LEV_WN_CLR_DN_FLT : BOOL ;	//LEVELER WINDOW FRAME CLEANER DOWN FAULT
   LEV_WN_CLR_AUTO_DN_OVR : BOOL ;	//LEVELER WINDOW FRAME CLEANER AUTO DOWN OVER
   LEV_WN_CLR_AUTO_DN_DEL : INT  := 3;	//LEVELER WINDOW FRAME CLEANER AUTO DOWN OVER DELAY
   LEV_WN_CLR_ATO_DN_DL_T : INT ;	//LEVELER WINDOW FRAME CLEANER AUTO DOWN OVER DELAY TIMER
   SMK_SLVE_FWD_OP_CUT : BOOL ;	//SMOKE SLEEVE FORWARD OUTPUT CUT
   SMK_SLVE_FWD_FLT_TMR : INT ;	//SMOKE SLEEVE FORWARD FAULT TIMER
   SMK_SLVE_FWD_FLT_GEN : INT  := 8;	//SMOKE SLEEVE FORWARD FAULT GENERATION TIME
   SMK_SLVE_FWD_OP_CT_TM : INT ;	//SMOKE SLEEVE FORWARD OUTPUT CUT TIMER
   SMK_SLVE_FWD_FLT : BOOL ;	//SMOKE SLEEVE FORWARD FAULT
   SMK_SLVE_AUTO_FWD_OVR : BOOL ;	//SMOKE SLEEVE AUTO FORWARD OVER
   SMK_SLVE_AUTO_FWD_DEL : INT  := 3;	//SMOKE SLEEVE AUTO FORWARD OVER DELAY
   SMK_SLVE_ATO_FWD_DL_T : INT ;	//SMOKE SLEEVE AUTO FORWARD OVER DELAY TIMER
   SMK_SLVE_RET_OP_CUT : BOOL ;	//SMOKE SLEEVE RETRACT OUTPUT CUT
   SMK_SLVE_RET_FLT_TMR : INT ;	//SMOKE SLEEVE RETRACT FAULT TIMER
   SMK_SLVE_RET_FLT_GEN : INT  := 8;	//SMOKE SLEEVE RETRACT FAULT GENERATION TIME
   SMK_SLVE_RET_OP_CT_TM : INT ;	//SMOKE SLEEVE RETRACT OUTPUT CUT TIMER
   SMK_SLVE_RET_FLT : BOOL ;	//SMOKE SLEEVE RETRACT FAULT
   SMK_SLVE_AUTO_RET_OVR : BOOL ;	//SMOKE SLEEVE AUTO RETRACT OVER
   SMK_SLVE_AUTO_RET_DEL : INT  := 3;	//SMOKE SLEEVE AUTO RETRACT OVER DELAY
   SMK_SLVE_ATO_RET_DL_T : INT ;	//SMOKE SLEEVE AUTO RETRACT OVER DELAY TIMER
   ACT_GRIP_DOOR_HOOK_IND : BOOL ;	//ACTUATING GRIP DOOR ON HOOK INDICATION
   ACT_GRIP_DR_HOOK_IND_LCS : BOOL ;	//ACTUATING GRIP DOOR ON HOOK INDICATION LCS
   SMK_SLVE_SL_FWD_OP_CUT : BOOL ;	//SMOKE SLEEVE SLOW FORWARD OUTPUT CUT
   SMK_SLVE_SL_FWD_FLT_TMR : INT ;	//SMOKE SLEEVE SLOW FORWARD FAULT TIMER
   SMK_SLVE_SL_FWD_FLT_GEN : INT  := 8;	//SMOKE SLEEVE SLOW FORWARD FAULT GENERATION TIME
   SMK_SLVE_SL_FWD_OP_CT_TM : INT ;	//SMOKE SLEEVE SLOW FORWARD OUTPUT CUT TIMER
   SMK_SLVE_SL_FWD_FLT : BOOL ;	//SMOKE SLEEVE SLOW FORWARD FAULT
   SMK_SLVE_SL_AUTO_FWD_OVR : BOOL ;	//SMOKE SLEEVE SLOW AUTO FORWARD OVER
   SMK_SLVE_SL_AUTO_FWD_DEL : INT  := 3;	//SMOKE SLEEVE SLOW AUTO FORWARD OVER DELAY
   SMK_SLVE_SL_ATO_FWD_DL_T : INT ;	//SMOKE SLEEVE SLOW AUTO FORWARD OVER DELAY TIMER
   SMK_SLV_SLOW_FWD_BIT : BOOL ;	//SMOKE SLEEVEL SLOW FORWARD BIT
   FIN_LEV_DOOR_OPER_STA_PB : BOOL ;	//FINISH LEVELING DOOR OPERATIONS START PUSH BUTTON
   FIN_LEV_OPER_AUTO_START : BOOL ;	//FINISH LEVELING OPERATIONS AUTO START
   LEV_FR_CL_CLN_CYL_CNT : INT ;	//LEVELER FRAME CLEANER CLEAN CYCLE COUNT
   LEV_FR_CL_CLN_CYL_CNT_SE : INT  := 3;	//LEVELER FRAME CLEANER CLEAN CYCLE COUNT SET POINT
   LEV_FR_CL_CLN_CYL_CMP : BOOL ;	//LEVELER FRAME CLEANER CLEAN CYCLE COMPLETED
   FIN_LEV_PERM_IND : BOOL ;	//FINISH LEVELING PERMISSION INDICATOR
   SLW_RK_SP_1_RET_FST : BOOL ;	//SLEWING RACK STEP 1 FIRST RETRACT IN AUTO MODE
   SLW_RK_SP_1_RET_SND : BOOL ;	//SLEWING RACK STEP 1 SECONFD RETRACE IN AUTO MODE
   FIN_LEV_RDY_TO_STA : BOOL ;	//FINISH LEVELING READY TO START
  END_STRUCT ;	
BEGIN
   SLW_RK_SP_1_FWD_FLT_GEN := 8;
   SLW_RK_SP_1_AUTO_FWD_DEL := 3;
   SLW_RK_SP_2_FWD_FLT_GEN := 8;
   SLW_RK_SP_2_AUTO_FWD_DEL := 3;
   SLW_RK_SP_1_RET_FLT_GEN := 8;
   SLW_RK_SP_1_AUTO_RET_DEL := 3;
   SLW_RK_SP_2_RET_FLT_GEN := 8;
   SLW_RK_SP_2_AUTO_RET_DEL := 3;
   ACT_GRP_FWD_FLT_GEN := 8;
   ACT_GRP_AUTO_FWD_DEL := 3;
   ACT_GRP_RET_FLT_GEN := 8;
   ACT_GRP_AUTO_RET_DEL := 3;
   LEV_WN_CLR_UP_FLT_GEN := 8;
   LEV_WN_CLR_AUTO_UP_DEL := 3;
   LEV_WN_CLR_DN_FLT_GEN := 8;
   LEV_WN_CLR_AUTO_DN_DEL := 3;
   SMK_SLVE_FWD_FLT_GEN := 8;
   SMK_SLVE_AUTO_FWD_DEL := 3;
   SMK_SLVE_RET_FLT_GEN := 8;
   SMK_SLVE_AUTO_RET_DEL := 3;
   SMK_SLVE_SL_FWD_FLT_GEN := 8;
   SMK_SLVE_SL_AUTO_FWD_DEL := 3;
END_DATA_BLOCK

DATA_BLOCK "LEVELER_MUFF_DB"	// DB 11
AUTHOR : Kamillas
VERSION : 0.1
  STRUCT
   RAM_EM_DRV_ENG_LCS_15 : BOOL ;	//RAM EMERGENCY DRIVE ENGAGE LCS-15
   RAM_EM_DRV_DENG_LCS_15 : BOOL ;	//RAM EMERGENCY DRIVE DISENGAGE LCS-15
   EMERGENCY_PB_LCS_15 : BOOL ;	//LCS-15 EMERGENCY PUSH BUTTON
   LEV_EM_DRV_ENG_LCS_16 : BOOL ;	//LEVELER EMERGENCY DRIVE ENGAGE LCS-16
   LEV_EM_DRV_DENG_LCS_16 : BOOL ;	//LEVELER EMERGENCY DRIVE DISENGAGE LCS-16
   EMERGENCY_PB_LCS_16 : BOOL ;	//LCS-16 EMERGENCY PUSH BUTTON
   RAM_EM_DRV_ENG_IND_LC_15 : BOOL ;	//RAM EMERGENCY DRIVE ENGAGE INDICATOR LCS-15
   RAM_PNEU_DRV_ENG_UP_CMD : BOOL ;	//PNEUMATIC EMERGENCY DRIVE LEVEL UP COMMAND
   RAM_PNEU_DRV_ENG_DN_CMD : BOOL ;	//PNEUMATIC EMERGENCY DRIVE LEVEL DOWN COMMAND
   LOCAL_LCS_16_IND : BOOL ;	//LOCAL SELECTED LCS-16 INDICATOR
   LEV_PNEU_DRV_ENG_UP_CMD : BOOL ;	//LEVELER EMERGENCY PNEUMATIC DRIVE PUSH UP COMMAND
   LEV_PNEU_DRV_ENG_DN_CMD : BOOL ;	//LEVELER EMERGENCY PNEUMATIC DRIVE PUSH DOWN COMMAND
   LEV_EM_DRV_ENG_LS : BOOL ;	//LEVELER EMERGENCY DRIVE ENGAGED LIMIT SWITCH
   RAM_EM_DRV_ENG_LS : BOOL ;	//PUSHER EMERGENCY DRIVE ENGAGED LIMIT SWITCH
  END_STRUCT ;	
BEGIN
END_DATA_BLOCK

